// TIA Portal project "MSE_Mubea_AsitYikama" (V15.1)

(* hardware
DEVICE "S7-1200 station_1"  S7-1200 Station
   slot 0: "Rack_0"  S7-1200 Rack  Rack  V1.0
   slot 1: "PLC_1"  CPU 1215C DC/DC/DC  6ES7 215-1AG40-0XB0  V4.1
   slot 2: "DI16/DQ16 x 24VDC"  6ES7 223-1BL32-0XB0  V2.0
DEVICE "HMI_1"  KTP400 Basic color PN
   slot 0: "HMI_1"  KTP400 Basic color PN  6AV6 647-0AK11-3AX0  12.0.0.0
   slot 1: "HMI_RT_1"  KTP400 Basic color PN  6AV6 647-0AK11-3AX0  12.0.0.0
   slot 5: "HMI_1.IE_CP_1"  PROFINET Interface  12.0.0.0
      slot 1: "PROFINET Interface_1"  PROFINET Interface
         slot 1: "Port_1"  Port
*)

// ===== PLC "PLC_1"  CPU 1215C DC/DC/DC =====

VAR_GLOBAL   // PLC tag table "Default tag table"
   "Clock_Byte" AT %MB0 : Byte;
   "Clock_10Hz" AT %M0.0 : Bool;
   "Clock_5Hz" AT %M0.1 : Bool;
   "Clock_2.5Hz" AT %M0.2 : Bool;
   "Clock_2Hz" AT %M0.3 : Bool;
   "Clock_1.25Hz" AT %M0.4 : Bool;
   "Clock_1Hz" AT %M0.5 : Bool;
   "Clock_0.625Hz" AT %M0.6 : Bool;
   "Clock_0.5Hz" AT %M0.7 : Bool;
   "HmiSirkVana_Ac_Mem" AT %M1.0 : Bool;   // Sirkulasyon vanasini ac
   "HmiSirkVana_Kapat_Mem" AT %M1.1 : Bool;
   "HmiDolumVana_Ac_Mem" AT %M1.2 : Bool;
   "HmiDolumVana_Kapat_Mem" AT %M1.3 : Bool;
   "HmiAsitTahVana_Ac_Mem" AT %M1.4 : Bool;
   "HmiAsitTahVana_Kapat_Mem" AT %M1.5 : Bool;
   "HmiUcYolluVana_Ac_Mem" AT %M1.6 : Bool;
   "HmiUcYolluVana_Kapat_Mem" AT %M1.7 : Bool;
   "HmiKuyuVana_Ac_Mem" AT %M2.0 : Bool;
   "HmiKuyuVana_Kapat_Mem" AT %M2.1 : Bool;
   "HmiIBCVana_Ac_Mem" AT %M2.2 : Bool;
   "HmiIBCVana_Kapat_Mem" AT %M2.3 : Bool;
   "HmiAnaPompa_Run" AT %M2.4 : Bool;
   "HmiIBCPopmpa_Run" AT %M2.5 : Bool;
   "AsitDoldur_Started" AT %M2.6 : Bool;
   "AsitDoldurSeq_UcYolVana_Ac" AT %M2.7 : Bool;
   "AsitDoldurSeq_DolumVana_Ac" AT %M3.0 : Bool;
   "AsitDoldurSeq_SirVana_Kapat" AT %M3.1 : Bool;
   "AsitDoldurSeq_TahVana_Kapat" AT %M3.2 : Bool;
   "AsitDoldurSeq_KuyuVana_Kapat" AT %M3.3 : Bool;
   "AsitDoldurSeq_IBCVana_Kapat" AT %M3.4 : Bool;
   "AsitDoldurSeq_AnaPompa_Run" AT %M3.5 : Bool;
   "AsitSirkulas_Started" AT %M3.6 : Bool;
   "AsitSirkulas_SirkVana_Ac" AT %M3.7 : Bool;
   "AsitSirkulas_DolumVana_Kapat" AT %M4.0 : Bool;
   "AsitSirkulas_TahVana_Kapat" AT %M4.1 : Bool;
   "AsitSirkulas_UcYolVana_Kapat" AT %M4.2 : Bool;
   "AsitSirkulas_KuyuVana_Kapat" AT %M4.3 : Bool;
   "AsitSirkulas_IBCVana_Kapat" AT %M4.4 : Bool;
   "AsitSirkulas_AnaPompa_Run" AT %M4.5 : Bool;
   "AsitSirkTimerReset_Mem" AT %M4.6 : Bool;
   "AsitTahliyesi_Started" AT %M4.7 : Bool;
   "AsitTahliyesi_SirkVana_Kapat" AT %M5.0 : Bool;
   "AsitTahliyesi_DolumVana_Kapat" AT %M5.1 : Bool;
   "AsitTahliyesi_TahVana_Ac" AT %M5.2 : Bool;
   "AsitTahliyesi_UcYolVana_Kapat" AT %M5.3 : Bool;
   "AsitTahliyesi_KuyuTahVana_Kapat" AT %M5.4 : Bool;
   "AsitTahliyesi_IBCVana_Kapat" AT %M5.5 : Bool;
   "AsitTahliyesi_Pompa_Run" AT %M5.6 : Bool;
   "SuSirkulasyon_Started" AT %M5.7 : Bool;
   "SuSirkulasyonTimer_Reset" AT %M6.0 : Bool;
   "SuSirkulasyon_SirkVana_Ac" AT %M6.1 : Bool;
   "SuSirkulasyon_DolumVana_Kapat" AT %M6.2 : Bool;
   "SuSirkulasyon_TahVana_Kapat" AT %M6.3 : Bool;
   "SuSirkulasyon_UcYolluVana_Kapat" AT %M6.4 : Bool;
   "SuSirkulasyon_KuyuTah_Kapat" AT %M6.5 : Bool;
   "SuSirkulasyon_IBCVana_Kapat" AT %M6.6 : Bool;
   "SuSirkulasyon_Pompa_Run" AT %M6.7 : Bool;
   "SuTahliyesi_Started" AT %M7.0 : Bool;
   "SuTahliyesi_SirkVana_Kapat" AT %M7.1 : Bool;
   "SuTahliyesi_DolumVana_Kapat" AT %M7.2 : Bool;
   "SuTahliyesi_AsitTahVana_Kapat" AT %M7.3 : Bool;
   "SuTahliyesi_UcYolluVana_Kapat" AT %M7.4 : Bool;
   "SuTahliyesi_KuyuTahVana_Ac" AT %M7.5 : Bool;
   "SuTahliyesi_IBCVana_Kapat" AT %M7.6 : Bool;
   "SuTahliyesi_Pompa_Run" AT %M7.7 : Bool;
   "IBCTahliye_Started" AT %M8.0 : Bool;
   "IBCTahliye_SirkVana_Kapat" AT %M8.1 : Bool;
   "IBCTahliye_DolumVana_Kapat" AT %M8.2 : Bool;
   "IBCTahliye_AsitTahVana_Kapat" AT %M8.3 : Bool;
   "IBCTahliye_UcYolluVana_Kapat" AT %M8.4 : Bool;
   "IBCTahliye_kuyuTahVana_Kapat" AT %M8.5 : Bool;
   "IBCTahliye_IBCVana_Ac" AT %M8.6 : Bool;
   "tempPompaRun" AT %M8.7 : Bool;
   "IBCTahliye_IBCpompa_Run" AT %M9.0 : Bool;
   "AsitDoldur_Siren" AT %M9.1 : Bool;
   "AsitDoldur_IslemBitti" AT %M9.2 : Bool;
   "AsitSirkulas_Siren" AT %M9.3 : Bool;
   "AsitSirkulas_IslemBitti" AT %M9.4 : Bool;
   "AsitTahliyesi_Siren" AT %M9.5 : Bool;
   "AsitTahliyesi_IslemBitti" AT %M9.6 : Bool;
   "SuSirkulasyon_Siren" AT %M9.7 : Bool;
   "SuSirkulasyon_IslemBitti" AT %M10.0 : Bool;
   "SuTahliyesi_Siren" AT %M10.1 : Bool;
   "SuTahliyesi_IslemBitti" AT %M10.2 : Bool;
   "IBCTahliye_Siren" AT %M10.3 : Bool;
   "IBCTahliye_IslemBitti" AT %M10.4 : Bool;
   "HmiKorKuyuPompa_Run" AT %M10.5 : Bool;
   "I0.0" AT %I0.0 : Bool;   // Acil Stop 1
   "I0.1" AT %I0.1 : Bool;   // Acil Stop 2
   "I0.2" AT %I0.2 : Bool;   // Yikama tanki alt seviye sen.
   "I0.3" AT %I0.3 : Bool;   // Yikama tanki ust limit sen.
   "I0.4" AT %I0.4 : Bool;   // Asti tanki alt limit sen.
   "I0.5" AT %I0.5 : Bool;
   "I0.6" AT %I0.6 : Bool;   // Yikama tank kapi sw 1
   "I1.0" AT %I1.0 : Bool;   // Asit tanki kapi sw
   "I1.1" AT %I1.1 : Bool;   // tERMİK HATA
   "I1.2" AT %I1.2 : Bool;   // Sirkulasyon vanasi kapali
   "I1.3" AT %I1.3 : Bool;   // Sirkulasyon vanasi acik
   "I1.4" AT %I1.4 : Bool;   // Dolum vanasi kapali
   "I1.5" AT %I1.5 : Bool;   // Dolum vanasi acik
   "I2.0" AT %I2.0 : Bool;   // Asit tahliye vanasi kapali
   "I2.1" AT %I2.1 : Bool;   // Asit tahliye vanasi acik
   "I2.2" AT %I2.2 : Bool;   // Uc yollu vana kapali
   "I2.3" AT %I2.3 : Bool;   // Uc yollu vana acik
   "I2.4" AT %I2.4 : Bool;   // Kuyu tahliye vanasi kapali
   "I2.5" AT %I2.5 : Bool;   // Kuyu tahliye vanasi acik
   "I2.6" AT %I2.6 : Bool;   // IBC Akis vanasi kapali
   "I2.7" AT %I2.7 : Bool;   // IBC akis vanasi acik
   "AsitDoldurSeq_DolumVana_Kapat" AT %M10.6 : Bool;
   "AsitDoldurSeq_AnaPompa_Run_2" AT %M10.7 : Bool;
   "AsitSirkulas_SirkVana_Kapat" AT %M11.0 : Bool;
   "AsitSirkulas_AnaPompa_Run_2" AT %M11.1 : Bool;
   "AsitTahliyesi_TahVana_Kapat" AT %M11.2 : Bool;
   "AsitTahliyesi_Pompa_Run_2" AT %M11.3 : Bool;
   "SuDolumSeq_SirkVana_Kapat" AT %M11.4 : Bool;
   "SuDolumSeq_DolumVana_Kapat" AT %M11.5 : Bool;
   "SuDolumSeq_AsitTahVana_Kapat" AT %M11.6 : Bool;
   "SuDolumSeq_UcYolluVana_Kapat" AT %M11.7 : Bool;
   "SuDolumSeq_KuyuTahVana_Kapat" AT %M12.0 : Bool;
   "SuDolumSeq_IBCVana_Kapat" AT %M12.1 : Bool;
   "SuDolumSeq_SuyuAc" AT %M12.2 : Bool;
   "SuDolumSeq_IslemBitti" AT %M12.3 : Bool;
   "I0.7" AT %I0.7 : Bool;   // Yikama tanki orta seviye sensoru
   "Always_On" AT %M12.4 : Bool;
   "SuSirkulasyon_SirkVana_Kapat" AT %M12.5 : Bool;
   "SuSirkulasyon_Pompa_Run2" AT %M12.6 : Bool;
   "SuTahliyesi_KuyuTahVana_Kapat" AT %M12.7 : Bool;
   "SuTahliyesi_Popmpa_Run2" AT %M13.0 : Bool;
   "IBCTahliye_IBCVana_Kapat" AT %M13.1 : Bool;
   "IBCTahliye_IBCpompa_Run2" AT %M13.2 : Bool;
   "AsitDoldurSeq_UcyolluVana_Kapat" AT %M13.3 : Bool;
   "HmiSuDolumVana" AT %M13.4 : Bool;
   "SuDolumVanasi" AT %Q3.0 : Bool;
END_VAR

VAR_GLOBAL   // PLC tag table "Output"
   "YesilLamba" AT %Q0.0 : Bool;
   "KirmiziLamba" AT %Q0.1 : Bool;
   "Siren" AT %Q0.2 : Bool;
   "SirkulasyonVanaKapat" AT %Q0.3 : Bool;
   "SirkulasyonVanaAc" AT %Q0.4 : Bool;
   "DolumVanaKapat" AT %Q0.5 : Bool;
   "DolumVanaAc" AT %Q0.6 : Bool;
   "AsitTahliyeVanaKapat" AT %Q0.7 : Bool;
   "AsitTahliyeVanaAc" AT %Q1.0 : Bool;
   "UcYolluVanaKapat" AT %Q1.1 : Bool;
   "UcYolluVanaAc" AT %Q2.0 : Bool;
   "KuyuTahliyeVanaKapat" AT %Q2.1 : Bool;
   "KuyuTahliyeVanaAc" AT %Q2.2 : Bool;
   "IBCVanaKapat" AT %Q2.3 : Bool;
   "IBCVanaAc" AT %Q2.4 : Bool;
   "AnaPompa" AT %Q2.5 : Bool;
   "IBC_DiyaframPompa" AT %Q2.6 : Bool;
   "KorKuyuPompasi" AT %Q2.7 : Bool;
END_VAR

// folder: DataBlocks

DATA_BLOCK "FB_Manuel_DB"   // DB4
{ S7_Optimized_Access := 'TRUE' }
VERSION : 0.1
// stored: InstanceOfName FB_Manuel
"FB_Manuel"
BEGIN
END_DATA_BLOCK

DATA_BLOCK "21_Alarm_DB"   // DB17
{ S7_Optimized_Access := 'TRUE' }
VERSION : 0.1
// stored: InstanceOfName 21_Alarm
"21_Alarm"
BEGIN
END_DATA_BLOCK

DATA_BLOCK "01_Out_DB"   // DB18
{ S7_Optimized_Access := 'TRUE' }
VERSION : 0.1
// stored: InstanceOfName 01_Out
"01_Out"
BEGIN
END_DATA_BLOCK

// folder: System blocks/Program resources

DATA_BLOCK "AsitSirkTimer_DB"   // DB5
{ S7_Optimized_Access := 'TRUE' }
AUTHOR : Simatic
FAMILY : IEC
NAME : IEC_TMR
VERSION : 1.0
// stored: InstanceOfName IEC_TIMER
"IEC_TIMER"
BEGIN
END_DATA_BLOCK

DATA_BLOCK "SuSirkTimer_DB"   // DB7
{ S7_Optimized_Access := 'TRUE' }
AUTHOR : Simatic
FAMILY : IEC
NAME : IEC_TMR
VERSION : 1.0
// stored: InstanceOfName IEC_TIMER
"IEC_TIMER"
BEGIN
END_DATA_BLOCK

// folder: SystemData

DATA_BLOCK "01_System"   // DB1
{ S7_Optimized_Access := 'TRUE' }
VERSION : 0.1
   VAR
      SystemInfo : String[50] := 'Asit sirkulasyonu yapiliyor';   // Sistem durumları
      Alarms : Word;
      Process : Struct
         Manuel_Normal : Bool;
      END_STRUCT;
      State : Struct
         AsitDolum : Byte;
         AsitSirkulasyon : Byte;
         AsitTahliye : Byte;
         SuDolum : Byte;
         SuSirkulasyon : Byte;
         SuTahliye : Byte;
         IBCTahliye : Byte;
      END_STRUCT;
      AlwaysOn : Bool;
      ConvertTimeToDint : DInt;   // Hmi ekranı icin cevrim
      Timers : Struct
         AsitDolum_TimerAdim3 : IEC_TIMER;
         AsitDolum_TimerAdim3_Pom : IEC_TIMER;
         Manuel : Struct
            SirkVana_Ac : IEC_TIMER;
            SirkVana_Kapat : IEC_TIMER;
            DolumVana_Ac : IEC_TIMER;
            DolumVana_Kapat : IEC_TIMER;
            AsitTahVana_Ac : IEC_TIMER;
            AsitTahVana_Kapat : IEC_TIMER;
            UcYolluVana_Ac : IEC_TIMER;
            UcYolluVana_Kapat : IEC_TIMER;
            KuyuTahVana_Ac : IEC_TIMER;
            KuyuTahVana_Kapat : IEC_TIMER;
            IBCVana_Ac : IEC_TIMER;
            IBCVana_Kapat : IEC_TIMER;
         END_STRUCT;
         Sequence : Struct
            AsitSir_TimerAdim3 : IEC_TIMER;
            AsitSir_TimerAdim3_Pom : IEC_TIMER;
            AsitTah_TimerAdim3 : IEC_TIMER;
            AsitTah_TimerAdim3_Pom : IEC_TIMER;
            SuSir_TimerAdim2_Pom : IEC_TIMER;
            SuSir_TimerAdim2 : IEC_TIMER;
            SuTah_TimerAdim2 : IEC_TIMER;
            SuTah_TimerAdim2_Pom : IEC_TIMER;
            IBCTah_TimerAdim2 : IEC_TIMER;
            IBCTah_TimerAdim2_Pom : IEC_TIMER;
         END_STRUCT;
      END_STRUCT;
   END_VAR
BEGIN
END_DATA_BLOCK

DATA_BLOCK "02_Peripheral"   // DB2
{ S7_Optimized_Access := 'TRUE' }
VERSION : 0.1
   VAR
      IN : Struct
         AcilStop : Bool;
         YikamaTanki : Struct
            UstSeviyeSen : Bool;   // Yikama tanki ust seviye sensoru
            AltSeviyeSen : Bool;   // Yikama tanki alt seviye sensoru
            CriticalSeviyeSen : Bool;   // Yikama tanki kritik seviye sensoru
            KapiSwitch1 : Bool;   // Yikama tanki kapi sw 1
            KapiSwitch2 : Bool;   // Yikama tanki kapi sw 2
         END_STRUCT;
         AsitTanki : Struct
            UstSeviyeSen : Bool;
            AltSeviyeSen : Bool;
            KapiSwitch : Bool;
         END_STRUCT;
         SirkulasyonVanasi : Struct   // 1 numaralı vana
            Opened : Bool;
            Closed : Bool;
         END_STRUCT;
         DolumVanasi : Struct   // 2 numaralı vana
            Opened : Bool;
            Closed : Bool;
         END_STRUCT;
         AsitTahliyeVanasi : Struct   // 3 numaralı vana
            Opened : Bool;
            Closed : Bool;
         END_STRUCT;
         UcYolluVana : Struct   // 4 numaralı vana
            Opened : Bool;
            Closed : Bool;
         END_STRUCT;
         KuyuTahVanasi : Struct   // 5 numaralı vana
            Opened : Bool;
            Closed : Bool;
         END_STRUCT;
         IBC : Struct
            AkisValfi : Struct
               Opened : Bool;   // IBC vanasi acildi
               Closed : Bool;   // IBC vanasi kapandi
            END_STRUCT;
         END_STRUCT;
         TermikAnaPompa : Bool;
      END_STRUCT;
      OUT : Struct
         IBC : Struct
            PompaDiyafram : Bool;   // Diyafram pompasi
            AkisValfi : Struct   // 6 numaralı akis valfi
               Open : Bool;
               Close : Bool;
            END_STRUCT;
         END_STRUCT;
         SirkulasyonVanasi : Struct   // 1 numaralı vana
            Open : Bool;
            Close : Bool;
         END_STRUCT;
         DolumVanasi : Struct   // 2 numaralı vana
            Open : Bool;
            Close : Bool;
         END_STRUCT;
         AsitTahliyeVanasi : Struct   // 3 numaralı vana
            Open : Bool;
            Close : Bool;
         END_STRUCT;
         UcYolluVana : Struct   // 4 numaralı vana
            Open : Bool;
            Close : Bool;
         END_STRUCT;
         KuyuAktVanasi : Struct   // 5 numaralı vana
            Open : Bool;
            Close : Bool;
         END_STRUCT;
         AnaPompa : Bool;   // Ana doldurma ve sirkulasyon pompasi
         KorKuyuPompasi : Bool;   // Kör kuyu pompası
         SuDolumVanasi : Bool;   // Su dolumu yapmak icin
      END_STRUCT;
      Lamba : Struct
         Yesil : Bool;
         Sari : Bool;
         Kirmizi : Bool;
         Siren : Bool;
      END_STRUCT;
   END_VAR
BEGIN
END_DATA_BLOCK

DATA_BLOCK "03_HmiData"   // DB3
{ S7_Optimized_Access := 'TRUE' }
VERSION : 0.1
   VAR
      SurkilasyonVanasi_Ac : Bool;
      SurkilasyonVanasi_Kapat : Bool;
      DolumVanasi_Ac : Bool;
      DolumVanasi_Kapat : Bool;
      AsitTahliyeVanasi_Ac : Bool;
      AsitTahliyeVanasi_Kapat : Bool;
      UcYolluVana_Ac : Bool;
      UcYolluVana_Kapat : Bool;
      KuyuAktarimVanasi_Ac : Bool;
      KuyuAktarimVanasi_Kapat : Bool;
      IBCVanasi_Ac : Bool;
      IBCVanasi_Kapat : Bool;
      AnaPompa_Run : Bool;
      AnaPompa_Stop : Bool;
      IBC_DiyaframPompa_Run : Bool;
      IBC_DiyaframPompa_Stop : Bool;
      KorKuyuPompası_Run : Bool;
      KorKuyuPompası_Stop : Bool;
      SuDolumVanasi_Ac : Bool;
      SuDolumVanasi_Kapat : Bool;
   END_VAR
   VAR RETAIN
      TimerInterval : Struct
         AsitSirkulasyon : Time := T#1m;   // Asit sirkulasyon set degeri
         SuSirkulasyon : Time := T#1m;   // Su sirkulasyon set degeri
      END_STRUCT;
   END_VAR
   VAR
      Timer_ET : Struct
         AsitSirkulasyon : Time;
         SuSirkulasyon : Time;
      END_STRUCT;
      Started : Struct
         AsitDolum : Bool;
         AsitSirkulasyon : Bool;
         AsitTahliye : Bool;
         TemizSuDolum : Bool;
         TemizSuSirkulasyon : Bool;
         TemizSuTahliye : Bool;
         IBCTahliye : Bool;
      END_STRUCT;
      System : Struct
         Stop : Bool;   // ,
         AsitDoldurBaslat : Bool;   // Asit doldurma sekansı
         AsitSirkulasyonBaslat : Bool;   // Asit sirkulasyon sekansı
         AsitTahliyesiBaslat : Bool;
         TemizSuDolumuBaslat : Bool;
         TemizSuSirkulasyonuBaslat : Bool;
         TemizSuTahliyesiBaslat : Bool;
         IBCTahliyesiBaslat : Bool;
         WarningReset : Bool;
      END_STRUCT;
      Visualization : Struct
         TimerVisible : Bool;
         ActTimerMin : DInt;
         ActTimerSec : DInt;
         Visibility : Struct
            AsitDolum : Bool;
            AsitSirkulasyon : Bool;
            AsitTahliyesi : Bool;
            TemizSuDolum : Bool;
            TemizSuSirkulasyon : Bool;
            TemizSuTahliye : Bool;
            IBCTaliye : Bool;
            Manuel : Struct
               SirkulasyonVanaAc : Bool;
               SirkulasyonVanaKapat : Bool;
               DolumVanaAc : Bool;
               DolumVanaKapat : Bool;
               AsitTahVanaAc : Bool;
               AsitTahVanaKapat : Bool;
               UcYolluVanaAc : Bool;
               UcYolluVanaKapat : Bool;
               KuyuTahVanaAc : Bool;
               KuyuTahVanaKapat : Bool;
               IBCVanaAc : Bool;
               IBCVanaKapat : Bool;
            END_STRUCT;
         END_STRUCT;
         nMode : Int;
      END_STRUCT;
   END_VAR
BEGIN
END_DATA_BLOCK

// folder: (top level)

FUNCTION_BLOCK "01_Out"   // FB1, LAD
{ S7_Optimized_Access := 'TRUE' }
VERSION : 0.1
BEGIN

REGION Network 1: Sirkulasyon vanası ac
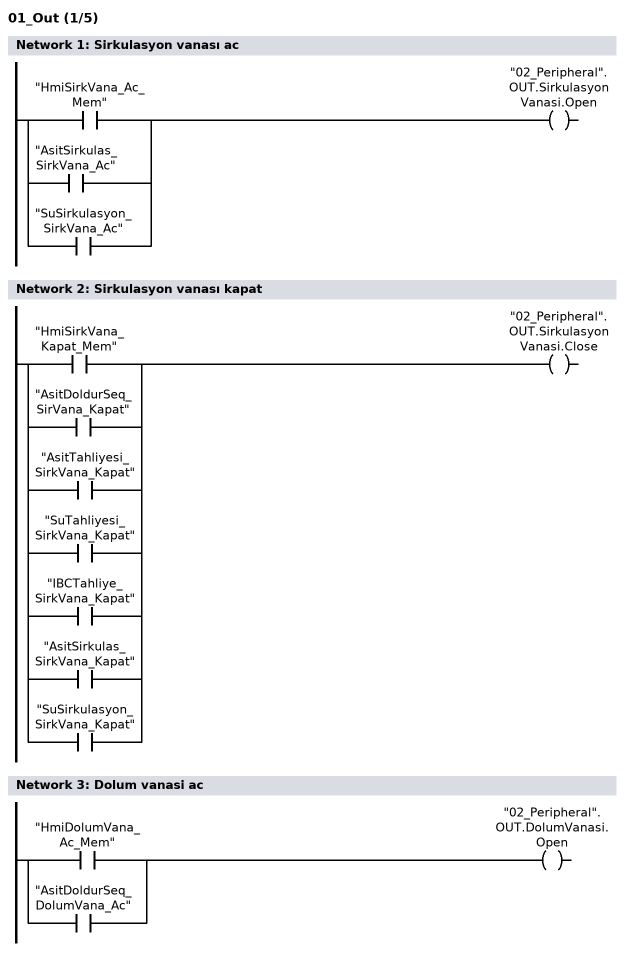
   RUNG wire#powerrail
      Contact( "HmiSirkVana_Ac_Mem" )
      wire#w1
      Coil( "02_Peripheral".OUT.SirkulasyonVanasi.Open )
   END_RUNG
   RUNG wire#powerrail
      Contact( "AsitSirkulas_SirkVana_Ac" )
   END_RUNG wire#w1
   RUNG wire#powerrail
      Contact( "SuSirkulasyon_SirkVana_Ac" )
   END_RUNG wire#w1
   // the same network as SCL:
   "02_Peripheral".OUT.SirkulasyonVanasi.Open := "HmiSirkVana_Ac_Mem" OR "AsitSirkulas_SirkVana_Ac" OR "SuSirkulasyon_SirkVana_Ac";
END_REGION

REGION Network 2: Sirkulasyon vanası kapat
   RUNG wire#powerrail
      Contact( "HmiSirkVana_Kapat_Mem" )
      wire#w1
      Coil( "02_Peripheral".OUT.SirkulasyonVanasi.Close )
   END_RUNG
   RUNG wire#powerrail
      Contact( "AsitDoldurSeq_SirVana_Kapat" )
   END_RUNG wire#w1
   RUNG wire#powerrail
      Contact( "AsitTahliyesi_SirkVana_Kapat" )
   END_RUNG wire#w1
   RUNG wire#powerrail
      Contact( "SuTahliyesi_SirkVana_Kapat" )
   END_RUNG wire#w1
   RUNG wire#powerrail
      Contact( "IBCTahliye_SirkVana_Kapat" )
   END_RUNG wire#w1
   RUNG wire#powerrail
      Contact( "AsitSirkulas_SirkVana_Kapat" )
   END_RUNG wire#w1
   RUNG wire#powerrail
      Contact( "SuSirkulasyon_SirkVana_Kapat" )
   END_RUNG wire#w1
   // the same network as SCL:
   "02_Peripheral".OUT.SirkulasyonVanasi.Close := "HmiSirkVana_Kapat_Mem" OR "AsitDoldurSeq_SirVana_Kapat" OR "AsitTahliyesi_SirkVana_Kapat" OR "SuTahliyesi_SirkVana_Kapat" OR "IBCTahliye_SirkVana_Kapat" OR "AsitSirkulas_SirkVana_Kapat" OR "SuSirkulasyon_SirkVana_Kapat";
END_REGION

REGION Network 3: Dolum vanasi ac
   RUNG wire#powerrail
      Contact( "HmiDolumVana_Ac_Mem" )
      wire#w1
      Coil( "02_Peripheral".OUT.DolumVanasi.Open )
   END_RUNG
   RUNG wire#powerrail
      Contact( "AsitDoldurSeq_DolumVana_Ac" )
   END_RUNG wire#w1
   // the same network as SCL:
   "02_Peripheral".OUT.DolumVanasi.Open := "HmiDolumVana_Ac_Mem" OR "AsitDoldurSeq_DolumVana_Ac";
END_REGION

REGION Network 4: Dolum vanasi kapat
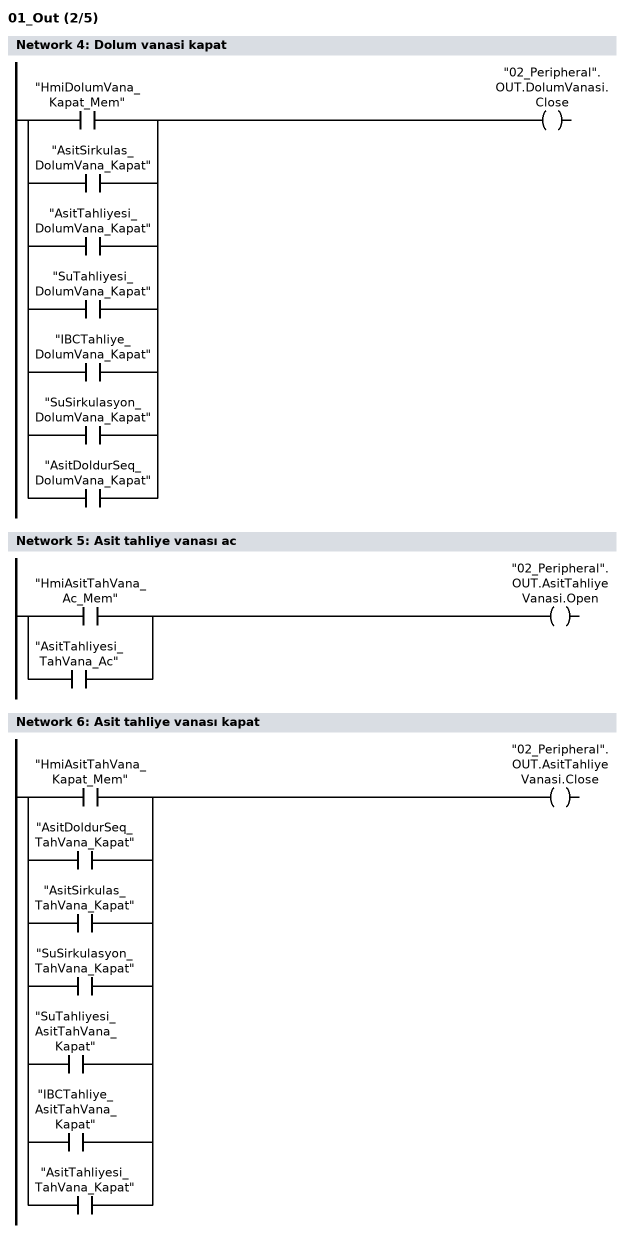
   RUNG wire#powerrail
      Contact( "HmiDolumVana_Kapat_Mem" )
      wire#w1
      Coil( "02_Peripheral".OUT.DolumVanasi.Close )
   END_RUNG
   RUNG wire#powerrail
      Contact( "AsitSirkulas_DolumVana_Kapat" )
   END_RUNG wire#w1
   RUNG wire#powerrail
      Contact( "AsitTahliyesi_DolumVana_Kapat" )
   END_RUNG wire#w1
   RUNG wire#powerrail
      Contact( "SuTahliyesi_DolumVana_Kapat" )
   END_RUNG wire#w1
   RUNG wire#powerrail
      Contact( "IBCTahliye_DolumVana_Kapat" )
   END_RUNG wire#w1
   RUNG wire#powerrail
      Contact( "SuSirkulasyon_DolumVana_Kapat" )
   END_RUNG wire#w1
   RUNG wire#powerrail
      Contact( "AsitDoldurSeq_DolumVana_Kapat" )
   END_RUNG wire#w1
   // the same network as SCL:
   "02_Peripheral".OUT.DolumVanasi.Close := "HmiDolumVana_Kapat_Mem" OR "AsitSirkulas_DolumVana_Kapat" OR "AsitTahliyesi_DolumVana_Kapat" OR "SuTahliyesi_DolumVana_Kapat" OR "IBCTahliye_DolumVana_Kapat" OR "SuSirkulasyon_DolumVana_Kapat" OR "AsitDoldurSeq_DolumVana_Kapat";
END_REGION

REGION Network 5: Asit tahliye vanası ac
   RUNG wire#powerrail
      Contact( "HmiAsitTahVana_Ac_Mem" )
      wire#w1
      Coil( "02_Peripheral".OUT.AsitTahliyeVanasi.Open )
   END_RUNG
   RUNG wire#powerrail
      Contact( "AsitTahliyesi_TahVana_Ac" )
   END_RUNG wire#w1
   // the same network as SCL:
   "02_Peripheral".OUT.AsitTahliyeVanasi.Open := "HmiAsitTahVana_Ac_Mem" OR "AsitTahliyesi_TahVana_Ac";
END_REGION

REGION Network 6: Asit tahliye vanası kapat
   RUNG wire#powerrail
      Contact( "HmiAsitTahVana_Kapat_Mem" )
      wire#w1
      Coil( "02_Peripheral".OUT.AsitTahliyeVanasi.Close )
   END_RUNG
   RUNG wire#powerrail
      Contact( "AsitDoldurSeq_TahVana_Kapat" )
   END_RUNG wire#w1
   RUNG wire#powerrail
      Contact( "AsitSirkulas_TahVana_Kapat" )
   END_RUNG wire#w1
   RUNG wire#powerrail
      Contact( "SuSirkulasyon_TahVana_Kapat" )
   END_RUNG wire#w1
   RUNG wire#powerrail
      Contact( "SuTahliyesi_AsitTahVana_Kapat" )
   END_RUNG wire#w1
   RUNG wire#powerrail
      Contact( "IBCTahliye_AsitTahVana_Kapat" )
   END_RUNG wire#w1
   RUNG wire#powerrail
      Contact( "AsitTahliyesi_TahVana_Kapat" )
   END_RUNG wire#w1
   // the same network as SCL:
   "02_Peripheral".OUT.AsitTahliyeVanasi.Close := "HmiAsitTahVana_Kapat_Mem" OR "AsitDoldurSeq_TahVana_Kapat" OR "AsitSirkulas_TahVana_Kapat" OR "SuSirkulasyon_TahVana_Kapat" OR "SuTahliyesi_AsitTahVana_Kapat" OR "IBCTahliye_AsitTahVana_Kapat" OR "AsitTahliyesi_TahVana_Kapat";
END_REGION

REGION Network 7: Uc yollu vana ac
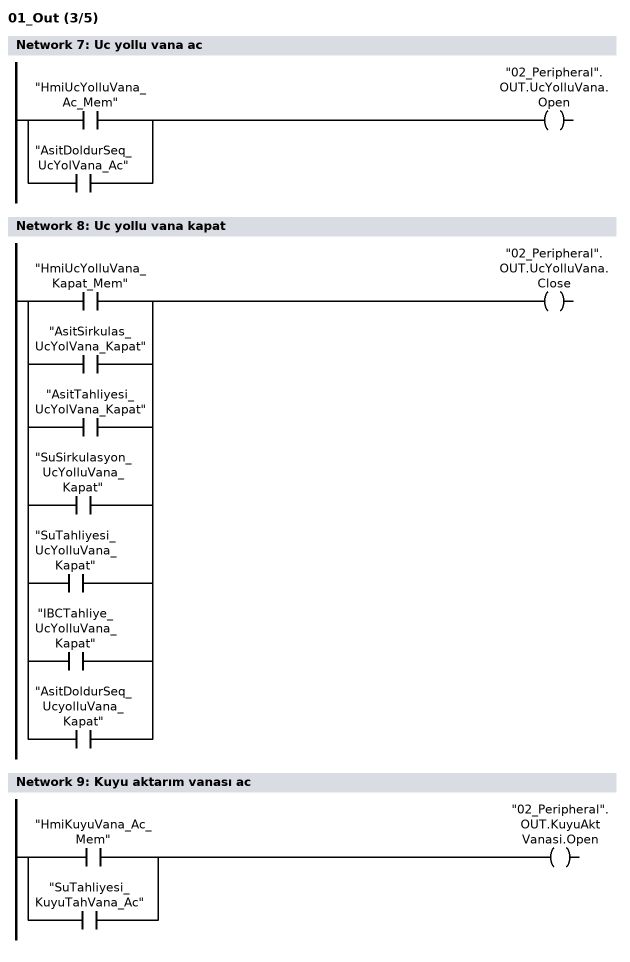
   RUNG wire#powerrail
      Contact( "HmiUcYolluVana_Ac_Mem" )
      wire#w1
      Coil( "02_Peripheral".OUT.UcYolluVana.Open )
   END_RUNG
   RUNG wire#powerrail
      Contact( "AsitDoldurSeq_UcYolVana_Ac" )
   END_RUNG wire#w1
   // the same network as SCL:
   "02_Peripheral".OUT.UcYolluVana.Open := "HmiUcYolluVana_Ac_Mem" OR "AsitDoldurSeq_UcYolVana_Ac";
END_REGION

REGION Network 8: Uc yollu vana kapat
   RUNG wire#powerrail
      Contact( "HmiUcYolluVana_Kapat_Mem" )
      wire#w1
      Coil( "02_Peripheral".OUT.UcYolluVana.Close )
   END_RUNG
   RUNG wire#powerrail
      Contact( "AsitSirkulas_UcYolVana_Kapat" )
   END_RUNG wire#w1
   RUNG wire#powerrail
      Contact( "AsitTahliyesi_UcYolVana_Kapat" )
   END_RUNG wire#w1
   RUNG wire#powerrail
      Contact( "SuSirkulasyon_UcYolluVana_Kapat" )
   END_RUNG wire#w1
   RUNG wire#powerrail
      Contact( "SuTahliyesi_UcYolluVana_Kapat" )
   END_RUNG wire#w1
   RUNG wire#powerrail
      Contact( "IBCTahliye_UcYolluVana_Kapat" )
   END_RUNG wire#w1
   RUNG wire#powerrail
      Contact( "AsitDoldurSeq_UcyolluVana_Kapat" )
   END_RUNG wire#w1
   // the same network as SCL:
   "02_Peripheral".OUT.UcYolluVana.Close := "HmiUcYolluVana_Kapat_Mem" OR "AsitSirkulas_UcYolVana_Kapat" OR "AsitTahliyesi_UcYolVana_Kapat" OR "SuSirkulasyon_UcYolluVana_Kapat" OR "SuTahliyesi_UcYolluVana_Kapat" OR "IBCTahliye_UcYolluVana_Kapat" OR "AsitDoldurSeq_UcyolluVana_Kapat";
END_REGION

REGION Network 9: Kuyu aktarım vanası ac
   RUNG wire#powerrail
      Contact( "HmiKuyuVana_Ac_Mem" )
      wire#w1
      Coil( "02_Peripheral".OUT.KuyuAktVanasi.Open )
   END_RUNG
   RUNG wire#powerrail
      Contact( "SuTahliyesi_KuyuTahVana_Ac" )
   END_RUNG wire#w1
   // the same network as SCL:
   "02_Peripheral".OUT.KuyuAktVanasi.Open := "HmiKuyuVana_Ac_Mem" OR "SuTahliyesi_KuyuTahVana_Ac";
END_REGION

REGION Network 10: Kuyu aktarım vanası kapat
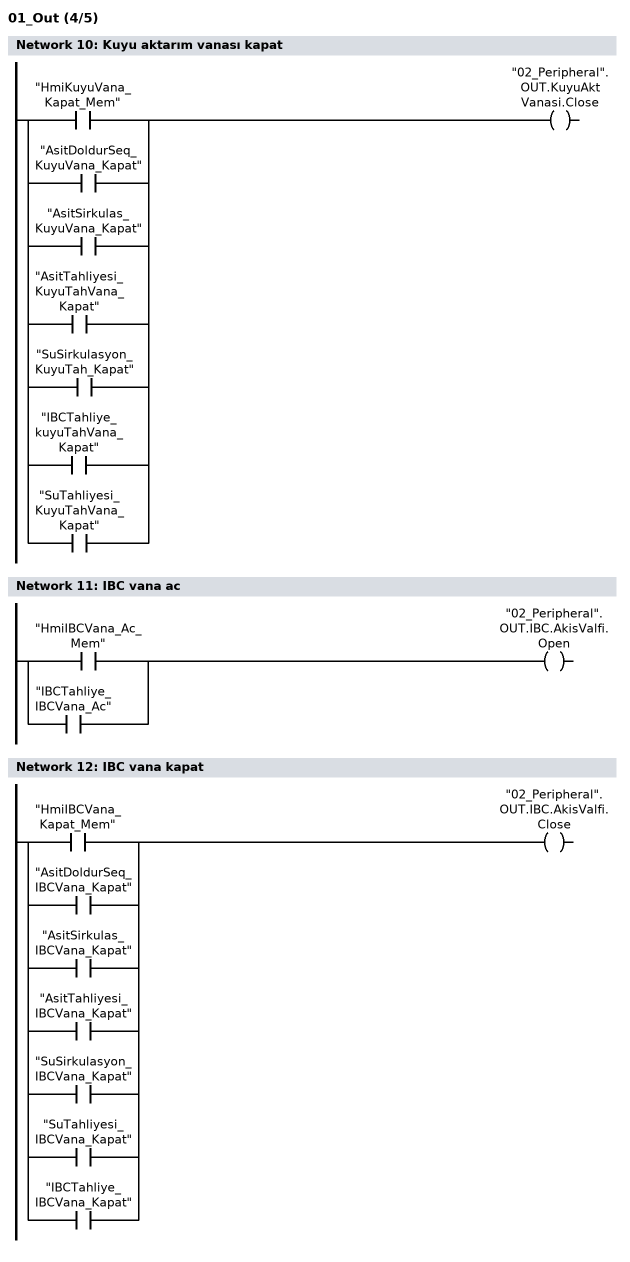
   RUNG wire#powerrail
      Contact( "HmiKuyuVana_Kapat_Mem" )
      wire#w1
      Coil( "02_Peripheral".OUT.KuyuAktVanasi.Close )
   END_RUNG
   RUNG wire#powerrail
      Contact( "AsitDoldurSeq_KuyuVana_Kapat" )
   END_RUNG wire#w1
   RUNG wire#powerrail
      Contact( "AsitSirkulas_KuyuVana_Kapat" )
   END_RUNG wire#w1
   RUNG wire#powerrail
      Contact( "AsitTahliyesi_KuyuTahVana_Kapat" )
   END_RUNG wire#w1
   RUNG wire#powerrail
      Contact( "SuSirkulasyon_KuyuTah_Kapat" )
   END_RUNG wire#w1
   RUNG wire#powerrail
      Contact( "IBCTahliye_kuyuTahVana_Kapat" )
   END_RUNG wire#w1
   RUNG wire#powerrail
      Contact( "SuTahliyesi_KuyuTahVana_Kapat" )
   END_RUNG wire#w1
   // the same network as SCL:
   "02_Peripheral".OUT.KuyuAktVanasi.Close := "HmiKuyuVana_Kapat_Mem" OR "AsitDoldurSeq_KuyuVana_Kapat" OR "AsitSirkulas_KuyuVana_Kapat" OR "AsitTahliyesi_KuyuTahVana_Kapat" OR "SuSirkulasyon_KuyuTah_Kapat" OR "IBCTahliye_kuyuTahVana_Kapat" OR "SuTahliyesi_KuyuTahVana_Kapat";
END_REGION

REGION Network 11: IBC vana ac
   RUNG wire#powerrail
      Contact( "HmiIBCVana_Ac_Mem" )
      wire#w1
      Coil( "02_Peripheral".OUT.IBC.AkisValfi.Open )
   END_RUNG
   RUNG wire#powerrail
      Contact( "IBCTahliye_IBCVana_Ac" )
   END_RUNG wire#w1
   // the same network as SCL:
   "02_Peripheral".OUT.IBC.AkisValfi.Open := "HmiIBCVana_Ac_Mem" OR "IBCTahliye_IBCVana_Ac";
END_REGION

REGION Network 12: IBC vana kapat
   RUNG wire#powerrail
      Contact( "HmiIBCVana_Kapat_Mem" )
      wire#w1
      Coil( "02_Peripheral".OUT.IBC.AkisValfi.Close )
   END_RUNG
   RUNG wire#powerrail
      Contact( "AsitDoldurSeq_IBCVana_Kapat" )
   END_RUNG wire#w1
   RUNG wire#powerrail
      Contact( "AsitSirkulas_IBCVana_Kapat" )
   END_RUNG wire#w1
   RUNG wire#powerrail
      Contact( "AsitTahliyesi_IBCVana_Kapat" )
   END_RUNG wire#w1
   RUNG wire#powerrail
      Contact( "SuSirkulasyon_IBCVana_Kapat" )
   END_RUNG wire#w1
   RUNG wire#powerrail
      Contact( "SuTahliyesi_IBCVana_Kapat" )
   END_RUNG wire#w1
   RUNG wire#powerrail
      Contact( "IBCTahliye_IBCVana_Kapat" )
   END_RUNG wire#w1
   // the same network as SCL:
   "02_Peripheral".OUT.IBC.AkisValfi.Close := "HmiIBCVana_Kapat_Mem" OR "AsitDoldurSeq_IBCVana_Kapat" OR "AsitSirkulas_IBCVana_Kapat" OR "AsitTahliyesi_IBCVana_Kapat" OR "SuSirkulasyon_IBCVana_Kapat" OR "SuTahliyesi_IBCVana_Kapat" OR "IBCTahliye_IBCVana_Kapat";
END_REGION

REGION Network 13: Ana pompa run/stop
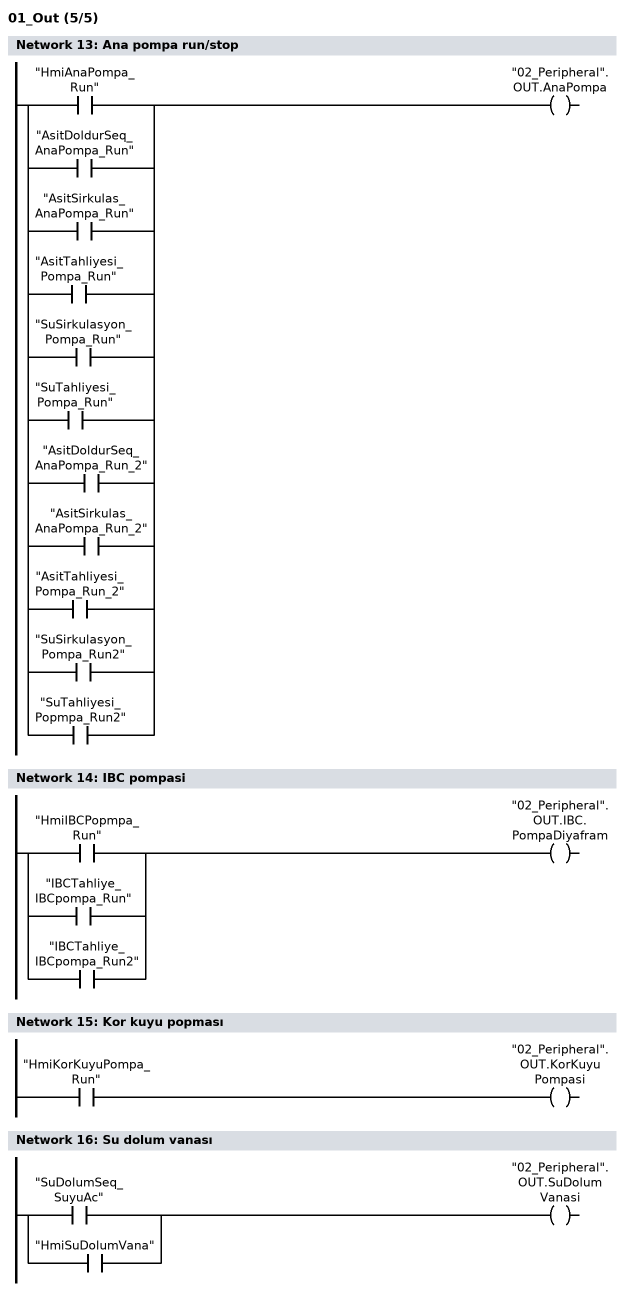
   RUNG wire#powerrail
      Contact( "HmiAnaPompa_Run" )
      wire#w1
      Coil( "02_Peripheral".OUT.AnaPompa )
   END_RUNG
   RUNG wire#powerrail
      Contact( "AsitDoldurSeq_AnaPompa_Run" )
   END_RUNG wire#w1
   RUNG wire#powerrail
      Contact( "AsitSirkulas_AnaPompa_Run" )
   END_RUNG wire#w1
   RUNG wire#powerrail
      Contact( "AsitTahliyesi_Pompa_Run" )
   END_RUNG wire#w1
   RUNG wire#powerrail
      Contact( "SuSirkulasyon_Pompa_Run" )
   END_RUNG wire#w1
   RUNG wire#powerrail
      Contact( "SuTahliyesi_Pompa_Run" )
   END_RUNG wire#w1
   RUNG wire#powerrail
      Contact( "AsitDoldurSeq_AnaPompa_Run_2" )
   END_RUNG wire#w1
   RUNG wire#powerrail
      Contact( "AsitSirkulas_AnaPompa_Run_2" )
   END_RUNG wire#w1
   RUNG wire#powerrail
      Contact( "AsitTahliyesi_Pompa_Run_2" )
   END_RUNG wire#w1
   RUNG wire#powerrail
      Contact( "SuSirkulasyon_Pompa_Run2" )
   END_RUNG wire#w1
   RUNG wire#powerrail
      Contact( "SuTahliyesi_Popmpa_Run2" )
   END_RUNG wire#w1
   // the same network as SCL:
   "02_Peripheral".OUT.AnaPompa := "HmiAnaPompa_Run" OR "AsitDoldurSeq_AnaPompa_Run" OR "AsitSirkulas_AnaPompa_Run" OR "AsitTahliyesi_Pompa_Run" OR "SuSirkulasyon_Pompa_Run" OR "SuTahliyesi_Pompa_Run" OR "AsitDoldurSeq_AnaPompa_Run_2" OR "AsitSirkulas_AnaPompa_Run_2" OR "AsitTahliyesi_Pompa_Run_2" OR "SuSirkulasyon_Pompa_Run2" OR "SuTahliyesi_Popmpa_Run2";
END_REGION

REGION Network 14: IBC pompasi
   RUNG wire#powerrail
      Contact( "HmiIBCPopmpa_Run" )
      wire#w1
      Coil( "02_Peripheral".OUT.IBC.PompaDiyafram )
   END_RUNG
   RUNG wire#powerrail
      Contact( "IBCTahliye_IBCpompa_Run" )
   END_RUNG wire#w1
   RUNG wire#powerrail
      Contact( "IBCTahliye_IBCpompa_Run2" )
   END_RUNG wire#w1
   // the same network as SCL:
   "02_Peripheral".OUT.IBC.PompaDiyafram := "HmiIBCPopmpa_Run" OR "IBCTahliye_IBCpompa_Run" OR "IBCTahliye_IBCpompa_Run2";
END_REGION

REGION Network 15: Kor kuyu popması
   RUNG wire#powerrail
      Contact( "HmiKorKuyuPompa_Run" )
      Coil( "02_Peripheral".OUT.KorKuyuPompasi )
   END_RUNG
   // the same network as SCL:
   "02_Peripheral".OUT.KorKuyuPompasi := "HmiKorKuyuPompa_Run";
END_REGION

REGION Network 16: Su dolum vanası
   RUNG wire#powerrail
      Contact( "SuDolumSeq_SuyuAc" )
      wire#w1
      Coil( "02_Peripheral".OUT.SuDolumVanasi )
   END_RUNG
   RUNG wire#powerrail
      Contact( "HmiSuDolumVana" )
   END_RUNG wire#w1
   // the same network as SCL:
   "02_Peripheral".OUT.SuDolumVanasi := "SuDolumSeq_SuyuAc" OR "HmiSuDolumVana";
END_REGION
END_FUNCTION_BLOCK

FUNCTION_BLOCK "FB_Manuel"   // FB2, LAD
{ S7_Optimized_Access := 'TRUE' }
VERSION : 0.1
   VAR_TEMP
      tTimerInterval : Time;
      bEmpty : Bool;
   END_VAR
   VAR_TEMP   // added for the SCL form of the ladder/FBD networks
      _w1 : Bool;
   END_VAR
BEGIN

REGION Network 1: Timer set degeri
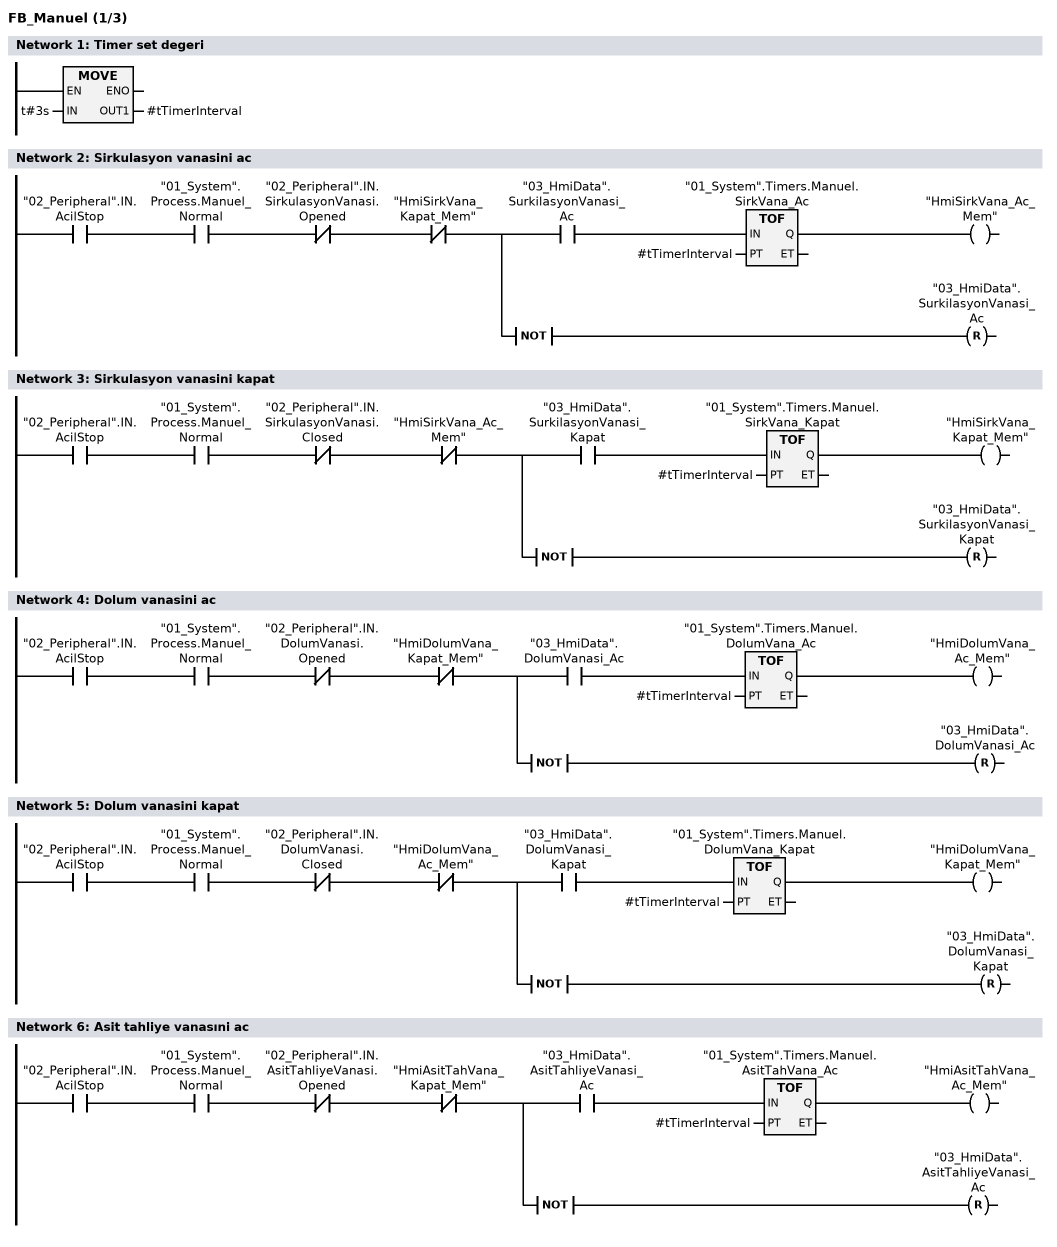
   RUNG wire#powerrail
      Move(in := t#3s, out1 => #tTimerInterval)
   END_RUNG
   // the same network as SCL:
   #tTimerInterval := t#3s;
END_REGION

REGION Network 2: Sirkulasyon vanasini ac
   #_w1 := "02_Peripheral".IN.AcilStop AND "01_System".Process.Manuel_Normal AND NOT "02_Peripheral".IN.SirkulasyonVanasi.Opened AND NOT "HmiSirkVana_Kapat_Mem";
   "01_System".Timers.Manuel.SirkVana_Ac.TOF(IN := #_w1 AND "03_HmiData".SurkilasyonVanasi_Ac,
                           PT := #tTimerInterval);
   "HmiSirkVana_Ac_Mem" := "01_System".Timers.Manuel.SirkVana_Ac.Q;
   IF NOT #_w1 THEN "03_HmiData".SurkilasyonVanasi_Ac := FALSE; END_IF;
END_REGION

REGION Network 3: Sirkulasyon vanasini kapat
   #_w1 := "02_Peripheral".IN.AcilStop AND "01_System".Process.Manuel_Normal AND NOT "02_Peripheral".IN.SirkulasyonVanasi.Closed AND NOT "HmiSirkVana_Ac_Mem";
   "01_System".Timers.Manuel.SirkVana_Kapat.TOF(IN := #_w1 AND "03_HmiData".SurkilasyonVanasi_Kapat,
                           PT := #tTimerInterval);
   "HmiSirkVana_Kapat_Mem" := "01_System".Timers.Manuel.SirkVana_Kapat.Q;
   IF NOT #_w1 THEN "03_HmiData".SurkilasyonVanasi_Kapat := FALSE; END_IF;
END_REGION

REGION Network 4: Dolum vanasini ac
   #_w1 := "02_Peripheral".IN.AcilStop AND "01_System".Process.Manuel_Normal AND NOT "02_Peripheral".IN.DolumVanasi.Opened AND NOT "HmiDolumVana_Kapat_Mem";
   "01_System".Timers.Manuel.DolumVana_Ac.TOF(IN := #_w1 AND "03_HmiData".DolumVanasi_Ac, PT := #tTimerInterval);
   "HmiDolumVana_Ac_Mem" := "01_System".Timers.Manuel.DolumVana_Ac.Q;
   IF NOT #_w1 THEN "03_HmiData".DolumVanasi_Ac := FALSE; END_IF;
END_REGION

REGION Network 5: Dolum vanasini kapat
   #_w1 := "02_Peripheral".IN.AcilStop AND "01_System".Process.Manuel_Normal AND NOT "02_Peripheral".IN.DolumVanasi.Closed AND NOT "HmiDolumVana_Ac_Mem";
   "01_System".Timers.Manuel.DolumVana_Kapat.TOF(IN := #_w1 AND "03_HmiData".DolumVanasi_Kapat,
                           PT := #tTimerInterval);
   "HmiDolumVana_Kapat_Mem" := "01_System".Timers.Manuel.DolumVana_Kapat.Q;
   IF NOT #_w1 THEN "03_HmiData".DolumVanasi_Kapat := FALSE; END_IF;
END_REGION

REGION Network 6: Asit tahliye vanasıni ac
   #_w1 := "02_Peripheral".IN.AcilStop AND "01_System".Process.Manuel_Normal AND NOT "02_Peripheral".IN.AsitTahliyeVanasi.Opened AND NOT "HmiAsitTahVana_Kapat_Mem";
   "01_System".Timers.Manuel.AsitTahVana_Ac.TOF(IN := #_w1 AND "03_HmiData".AsitTahliyeVanasi_Ac,
                           PT := #tTimerInterval);
   "HmiAsitTahVana_Ac_Mem" := "01_System".Timers.Manuel.AsitTahVana_Ac.Q;
   IF NOT #_w1 THEN "03_HmiData".AsitTahliyeVanasi_Ac := FALSE; END_IF;
END_REGION

REGION Network 7: Asit tahliye vanasıni kapat
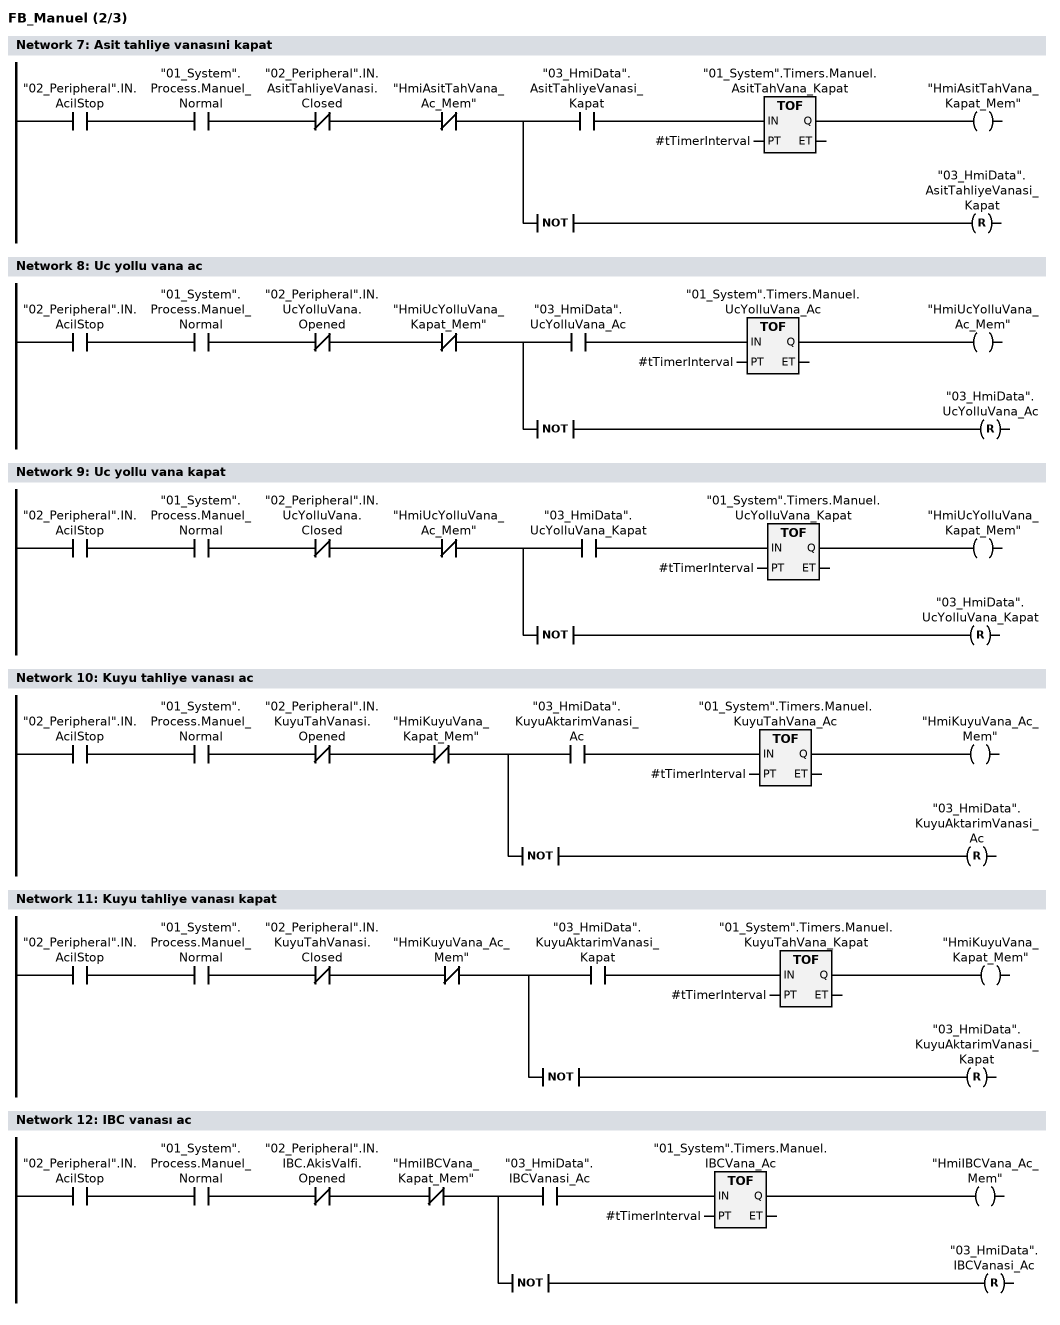
   #_w1 := "02_Peripheral".IN.AcilStop AND "01_System".Process.Manuel_Normal AND NOT "02_Peripheral".IN.AsitTahliyeVanasi.Closed AND NOT "HmiAsitTahVana_Ac_Mem";
   "01_System".Timers.Manuel.AsitTahVana_Kapat.TOF(IN := #_w1 AND "03_HmiData".AsitTahliyeVanasi_Kapat,
                           PT := #tTimerInterval);
   "HmiAsitTahVana_Kapat_Mem" := "01_System".Timers.Manuel.AsitTahVana_Kapat.Q;
   IF NOT #_w1 THEN "03_HmiData".AsitTahliyeVanasi_Kapat := FALSE; END_IF;
END_REGION

REGION Network 8: Uc yollu vana ac
   #_w1 := "02_Peripheral".IN.AcilStop AND "01_System".Process.Manuel_Normal AND NOT "02_Peripheral".IN.UcYolluVana.Opened AND NOT "HmiUcYolluVana_Kapat_Mem";
   "01_System".Timers.Manuel.UcYolluVana_Ac.TOF(IN := #_w1 AND "03_HmiData".UcYolluVana_Ac,
                           PT := #tTimerInterval);
   "HmiUcYolluVana_Ac_Mem" := "01_System".Timers.Manuel.UcYolluVana_Ac.Q;
   IF NOT #_w1 THEN "03_HmiData".UcYolluVana_Ac := FALSE; END_IF;
END_REGION

REGION Network 9: Uc yollu vana kapat
   #_w1 := "02_Peripheral".IN.AcilStop AND "01_System".Process.Manuel_Normal AND NOT "02_Peripheral".IN.UcYolluVana.Closed AND NOT "HmiUcYolluVana_Ac_Mem";
   "01_System".Timers.Manuel.UcYolluVana_Kapat.TOF(IN := #_w1 AND "03_HmiData".UcYolluVana_Kapat,
                           PT := #tTimerInterval);
   "HmiUcYolluVana_Kapat_Mem" := "01_System".Timers.Manuel.UcYolluVana_Kapat.Q;
   IF NOT #_w1 THEN "03_HmiData".UcYolluVana_Kapat := FALSE; END_IF;
END_REGION

REGION Network 10: Kuyu tahliye vanası ac
   #_w1 := "02_Peripheral".IN.AcilStop AND "01_System".Process.Manuel_Normal AND NOT "02_Peripheral".IN.KuyuTahVanasi.Opened AND NOT "HmiKuyuVana_Kapat_Mem";
   "01_System".Timers.Manuel.KuyuTahVana_Ac.TOF(IN := #_w1 AND "03_HmiData".KuyuAktarimVanasi_Ac,
                           PT := #tTimerInterval);
   "HmiKuyuVana_Ac_Mem" := "01_System".Timers.Manuel.KuyuTahVana_Ac.Q;
   IF NOT #_w1 THEN "03_HmiData".KuyuAktarimVanasi_Ac := FALSE; END_IF;
END_REGION

REGION Network 11: Kuyu tahliye vanası kapat
   #_w1 := "02_Peripheral".IN.AcilStop AND "01_System".Process.Manuel_Normal AND NOT "02_Peripheral".IN.KuyuTahVanasi.Closed AND NOT "HmiKuyuVana_Ac_Mem";
   "01_System".Timers.Manuel.KuyuTahVana_Kapat.TOF(IN := #_w1 AND "03_HmiData".KuyuAktarimVanasi_Kapat,
                           PT := #tTimerInterval);
   "HmiKuyuVana_Kapat_Mem" := "01_System".Timers.Manuel.KuyuTahVana_Kapat.Q;
   IF NOT #_w1 THEN "03_HmiData".KuyuAktarimVanasi_Kapat := FALSE; END_IF;
END_REGION

REGION Network 12: IBC vanası ac
   #_w1 := "02_Peripheral".IN.AcilStop AND "01_System".Process.Manuel_Normal AND NOT "02_Peripheral".IN.IBC.AkisValfi.Opened AND NOT "HmiIBCVana_Kapat_Mem";
   "01_System".Timers.Manuel.IBCVana_Ac.TOF(IN := #_w1 AND "03_HmiData".IBCVanasi_Ac, PT := #tTimerInterval);
   "HmiIBCVana_Ac_Mem" := "01_System".Timers.Manuel.IBCVana_Ac.Q;
   IF NOT #_w1 THEN "03_HmiData".IBCVanasi_Ac := FALSE; END_IF;
END_REGION

REGION Network 13: IBC vanası kapat
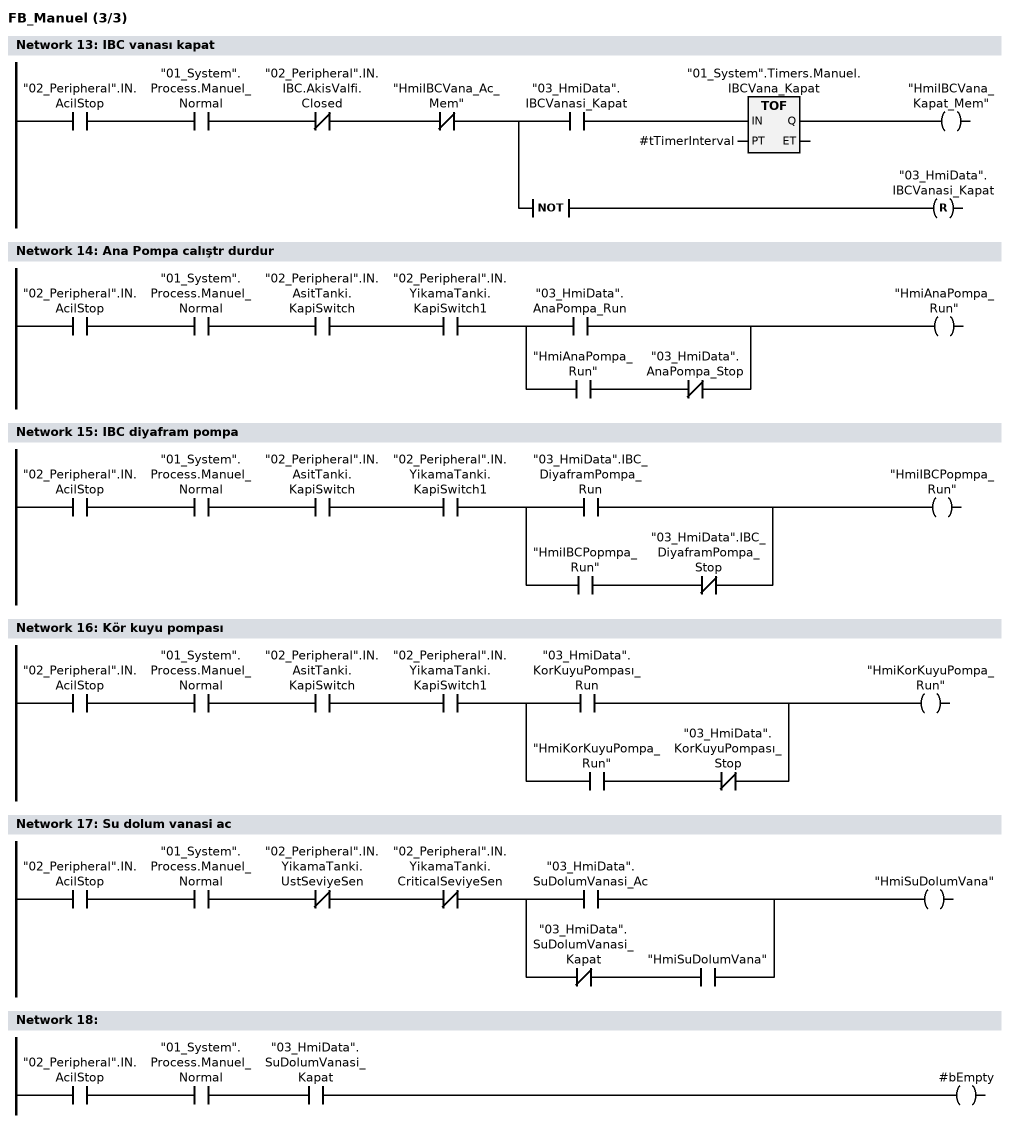
   #_w1 := "02_Peripheral".IN.AcilStop AND "01_System".Process.Manuel_Normal AND NOT "02_Peripheral".IN.IBC.AkisValfi.Closed AND NOT "HmiIBCVana_Ac_Mem";
   "01_System".Timers.Manuel.IBCVana_Kapat.TOF(IN := #_w1 AND "03_HmiData".IBCVanasi_Kapat,
                           PT := #tTimerInterval);
   "HmiIBCVana_Kapat_Mem" := "01_System".Timers.Manuel.IBCVana_Kapat.Q;
   IF NOT #_w1 THEN "03_HmiData".IBCVanasi_Kapat := FALSE; END_IF;
END_REGION

REGION Network 14: Ana Pompa calıştr durdur
   RUNG wire#powerrail
      Contact( "02_Peripheral".IN.AcilStop )
      Contact( "01_System".Process.Manuel_Normal )
      Contact( "02_Peripheral".IN.AsitTanki.KapiSwitch )
      Contact( "02_Peripheral".IN.YikamaTanki.KapiSwitch1 )
      wire#w1
      Contact( "03_HmiData".AnaPompa_Run )
      wire#w2
      Coil( "HmiAnaPompa_Run" )
   END_RUNG
   RUNG wire#w1
      Contact( "HmiAnaPompa_Run" )
      I_Contact( "03_HmiData".AnaPompa_Stop )
   END_RUNG wire#w2
   // the same network as SCL:
   "HmiAnaPompa_Run" := "02_Peripheral".IN.AcilStop AND "01_System".Process.Manuel_Normal AND "02_Peripheral".IN.AsitTanki.KapiSwitch AND "02_Peripheral".IN.YikamaTanki.KapiSwitch1 AND ("03_HmiData".AnaPompa_Run OR ("HmiAnaPompa_Run" AND NOT "03_HmiData".AnaPompa_Stop));
END_REGION

REGION Network 15: IBC diyafram pompa
   RUNG wire#powerrail
      Contact( "02_Peripheral".IN.AcilStop )
      Contact( "01_System".Process.Manuel_Normal )
      Contact( "02_Peripheral".IN.AsitTanki.KapiSwitch )
      Contact( "02_Peripheral".IN.YikamaTanki.KapiSwitch1 )
      wire#w1
      Contact( "03_HmiData".IBC_DiyaframPompa_Run )
      wire#w2
      Coil( "HmiIBCPopmpa_Run" )
   END_RUNG
   RUNG wire#w1
      Contact( "HmiIBCPopmpa_Run" )
      I_Contact( "03_HmiData".IBC_DiyaframPompa_Stop )
   END_RUNG wire#w2
   // the same network as SCL:
   "HmiIBCPopmpa_Run" := "02_Peripheral".IN.AcilStop AND "01_System".Process.Manuel_Normal AND "02_Peripheral".IN.AsitTanki.KapiSwitch AND "02_Peripheral".IN.YikamaTanki.KapiSwitch1 AND ("03_HmiData".IBC_DiyaframPompa_Run OR ("HmiIBCPopmpa_Run" AND NOT "03_HmiData".IBC_DiyaframPompa_Stop));
END_REGION

REGION Network 16: Kör kuyu pompası
   RUNG wire#powerrail
      Contact( "02_Peripheral".IN.AcilStop )
      Contact( "01_System".Process.Manuel_Normal )
      Contact( "02_Peripheral".IN.AsitTanki.KapiSwitch )
      Contact( "02_Peripheral".IN.YikamaTanki.KapiSwitch1 )
      wire#w1
      Contact( "03_HmiData".KorKuyuPompası_Run )
      wire#w2
      Coil( "HmiKorKuyuPompa_Run" )
   END_RUNG
   RUNG wire#w1
      Contact( "HmiKorKuyuPompa_Run" )
      I_Contact( "03_HmiData".KorKuyuPompası_Stop )
   END_RUNG wire#w2
   // the same network as SCL:
   "HmiKorKuyuPompa_Run" := "02_Peripheral".IN.AcilStop AND "01_System".Process.Manuel_Normal AND "02_Peripheral".IN.AsitTanki.KapiSwitch AND "02_Peripheral".IN.YikamaTanki.KapiSwitch1 AND ("03_HmiData".KorKuyuPompası_Run OR ("HmiKorKuyuPompa_Run" AND NOT "03_HmiData".KorKuyuPompası_Stop));
END_REGION

REGION Network 17: Su dolum vanasi ac
   RUNG wire#powerrail
      Contact( "02_Peripheral".IN.AcilStop )
      Contact( "01_System".Process.Manuel_Normal )
      I_Contact( "02_Peripheral".IN.YikamaTanki.UstSeviyeSen )
      I_Contact( "02_Peripheral".IN.YikamaTanki.CriticalSeviyeSen )
      wire#w1
      Contact( "03_HmiData".SuDolumVanasi_Ac )
      wire#w2
      Coil( "HmiSuDolumVana" )
   END_RUNG
   RUNG wire#w1
      I_Contact( "03_HmiData".SuDolumVanasi_Kapat )
      Contact( "HmiSuDolumVana" )
   END_RUNG wire#w2
   // the same network as SCL:
   "HmiSuDolumVana" := "02_Peripheral".IN.AcilStop AND "01_System".Process.Manuel_Normal AND NOT "02_Peripheral".IN.YikamaTanki.UstSeviyeSen AND NOT "02_Peripheral".IN.YikamaTanki.CriticalSeviyeSen AND ("03_HmiData".SuDolumVanasi_Ac OR (NOT "03_HmiData".SuDolumVanasi_Kapat AND "HmiSuDolumVana"));
END_REGION

REGION Network 18
   RUNG wire#powerrail
      Contact( "02_Peripheral".IN.AcilStop )
      Contact( "01_System".Process.Manuel_Normal )
      Contact( "03_HmiData".SuDolumVanasi_Kapat )
      Coil( #bEmpty )
   END_RUNG
   // the same network as SCL:
   #bEmpty := "02_Peripheral".IN.AcilStop AND "01_System".Process.Manuel_Normal AND "03_HmiData".SuDolumVanasi_Kapat;
END_REGION
END_FUNCTION_BLOCK

FUNCTION_BLOCK "21_Alarm"   // FB10, LAD
{ S7_Optimized_Access := 'TRUE' }
VERSION : 0.1
   VAR
      SirkulasyonVanaKapat : TON_TIME;
      SirkulasyonVanaAc : TON_TIME;
      DolumVanasiAc : TON_TIME;
      DolumVanasiKapat : TON_TIME;
      AsitTahliyeVanasiAc : TON_TIME;
      AsitTahliyeVanasiKapat : TON_TIME;
      UcYolluVanaAc : TON_TIME;
      UcYolluVanaKapat : TON_TIME;
      KuyuTahliyeVanaAc : TON_TIME;
      KuyuTahliyeVanaKapat : TON_TIME;
      IBCTahliyeVanaAc : TON_TIME;
      IBCTahliyeVanaKapat : TON_TIME;
   END_VAR
   VAR_TEMP
      tWatchdogInterval : Time;
   END_VAR
BEGIN

REGION Network 1
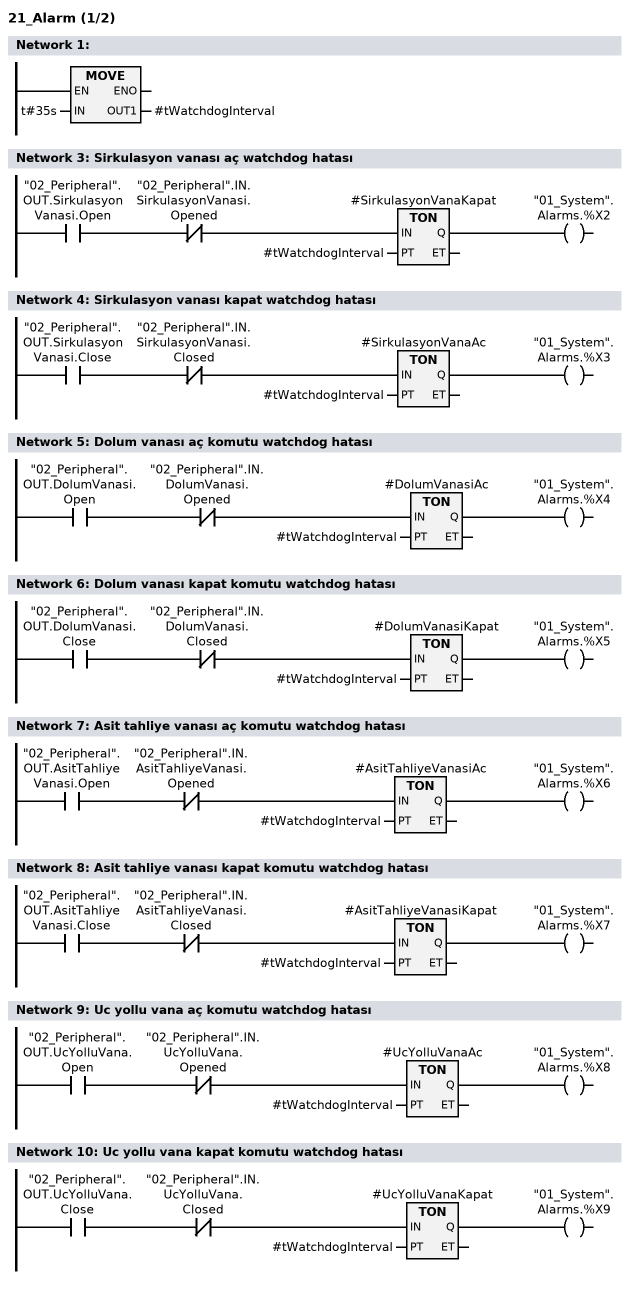
   RUNG wire#powerrail
      Move(in := t#35s, out1 => #tWatchdogInterval)
   END_RUNG
   // the same network as SCL:
   #tWatchdogInterval := t#35s;
END_REGION

REGION Network 2 (SCL): aCİL STOP ve TERMİK HATA
   "01_System".Alarms.%X0 := NOT "02_Peripheral".IN.AcilStop;
   "01_System".Alarms.%X1 := "02_Peripheral".IN.TermikAnaPompa;
END_REGION

REGION Network 3: Sirkulasyon vanası aç watchdog hatası
   #SirkulasyonVanaKapat(IN := "02_Peripheral".OUT.SirkulasyonVanasi.Open AND NOT "02_Peripheral".IN.SirkulasyonVanasi.Opened,   // TON
                         PT := #tWatchdogInterval);
   "01_System".Alarms.%X2 := #SirkulasyonVanaKapat.Q;
END_REGION

REGION Network 4: Sirkulasyon vanası kapat watchdog hatası
   #SirkulasyonVanaAc(IN := "02_Peripheral".OUT.SirkulasyonVanasi.Close AND NOT "02_Peripheral".IN.SirkulasyonVanasi.Closed,   // TON
                      PT := #tWatchdogInterval);
   "01_System".Alarms.%X3 := #SirkulasyonVanaAc.Q;
END_REGION

REGION Network 5: Dolum vanası aç komutu watchdog hatası
   #DolumVanasiAc(IN := "02_Peripheral".OUT.DolumVanasi.Open AND NOT "02_Peripheral".IN.DolumVanasi.Opened,   // TON
                  PT := #tWatchdogInterval);
   "01_System".Alarms.%X4 := #DolumVanasiAc.Q;
END_REGION

REGION Network 6: Dolum vanası kapat komutu watchdog hatası
   #DolumVanasiKapat(IN := "02_Peripheral".OUT.DolumVanasi.Close AND NOT "02_Peripheral".IN.DolumVanasi.Closed,   // TON
                     PT := #tWatchdogInterval);
   "01_System".Alarms.%X5 := #DolumVanasiKapat.Q;
END_REGION

REGION Network 7: Asit tahliye vanası aç komutu watchdog hatası
   #AsitTahliyeVanasiAc(IN := "02_Peripheral".OUT.AsitTahliyeVanasi.Open AND NOT "02_Peripheral".IN.AsitTahliyeVanasi.Opened,   // TON
                        PT := #tWatchdogInterval);
   "01_System".Alarms.%X6 := #AsitTahliyeVanasiAc.Q;
END_REGION

REGION Network 8: Asit tahliye vanası kapat komutu watchdog hatası
   #AsitTahliyeVanasiKapat(IN := "02_Peripheral".OUT.AsitTahliyeVanasi.Close AND NOT "02_Peripheral".IN.AsitTahliyeVanasi.Closed,   // TON
                           PT := #tWatchdogInterval);
   "01_System".Alarms.%X7 := #AsitTahliyeVanasiKapat.Q;
END_REGION

REGION Network 9: Uc yollu vana aç komutu watchdog hatası
   #UcYolluVanaAc(IN := "02_Peripheral".OUT.UcYolluVana.Open AND NOT "02_Peripheral".IN.UcYolluVana.Opened,   // TON
                  PT := #tWatchdogInterval);
   "01_System".Alarms.%X8 := #UcYolluVanaAc.Q;
END_REGION

REGION Network 10: Uc yollu vana kapat komutu watchdog hatası
   #UcYolluVanaKapat(IN := "02_Peripheral".OUT.UcYolluVana.Close AND NOT "02_Peripheral".IN.UcYolluVana.Closed,   // TON
                     PT := #tWatchdogInterval);
   "01_System".Alarms.%X9 := #UcYolluVanaKapat.Q;
END_REGION

REGION Network 11: Kuyu aktarım vanası aç komutu watchdog hatası
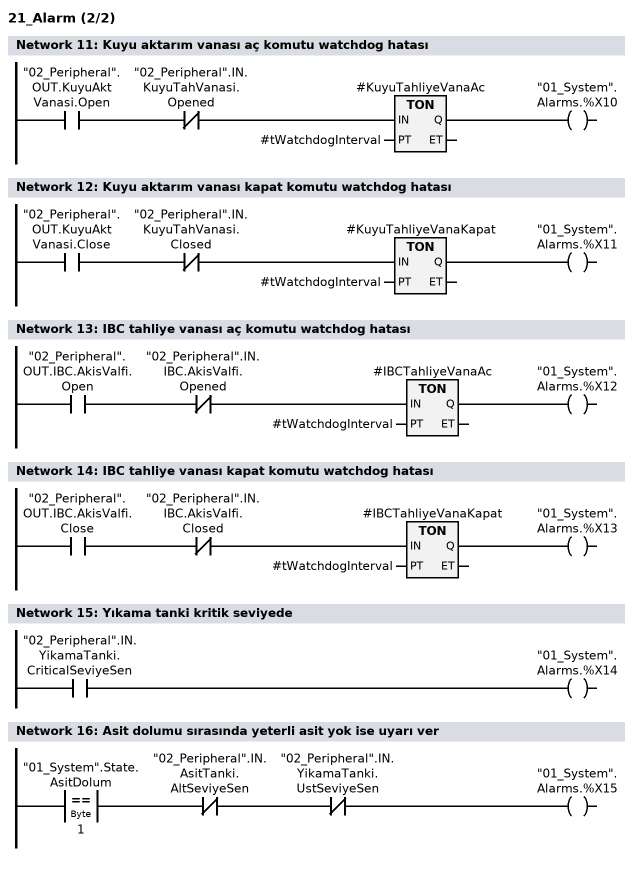
   #KuyuTahliyeVanaAc(IN := "02_Peripheral".OUT.KuyuAktVanasi.Open AND NOT "02_Peripheral".IN.KuyuTahVanasi.Opened,   // TON
                      PT := #tWatchdogInterval);
   "01_System".Alarms.%X10 := #KuyuTahliyeVanaAc.Q;
END_REGION

REGION Network 12: Kuyu aktarım vanası kapat komutu watchdog hatası
   #KuyuTahliyeVanaKapat(IN := "02_Peripheral".OUT.KuyuAktVanasi.Close AND NOT "02_Peripheral".IN.KuyuTahVanasi.Closed,   // TON
                         PT := #tWatchdogInterval);
   "01_System".Alarms.%X11 := #KuyuTahliyeVanaKapat.Q;
END_REGION

REGION Network 13: IBC tahliye vanası aç komutu watchdog hatası
   #IBCTahliyeVanaAc(IN := "02_Peripheral".OUT.IBC.AkisValfi.Open AND NOT "02_Peripheral".IN.IBC.AkisValfi.Opened,   // TON
                     PT := #tWatchdogInterval);
   "01_System".Alarms.%X12 := #IBCTahliyeVanaAc.Q;
END_REGION

REGION Network 14: IBC tahliye vanası kapat komutu watchdog hatası
   #IBCTahliyeVanaKapat(IN := "02_Peripheral".OUT.IBC.AkisValfi.Close AND NOT "02_Peripheral".IN.IBC.AkisValfi.Closed,   // TON
                        PT := #tWatchdogInterval);
   "01_System".Alarms.%X13 := #IBCTahliyeVanaKapat.Q;
END_REGION

REGION Network 15: Yıkama tanki kritik seviyede
   RUNG wire#powerrail
      Contact( "02_Peripheral".IN.YikamaTanki.CriticalSeviyeSen )
      Coil( "01_System".Alarms.%X14 )
   END_RUNG
   // the same network as SCL:
   "01_System".Alarms.%X14 := "02_Peripheral".IN.YikamaTanki.CriticalSeviyeSen;
END_REGION

REGION Network 16: Asit dolumu sırasında yeterli asit yok ise uyarı ver
   RUNG wire#powerrail
      { S7_Templates := "SrcType := Byte" } EQ_Contact(in1 := "01_System".State.AsitDolum, in2 := 1)
      I_Contact( "02_Peripheral".IN.AsitTanki.AltSeviyeSen )
      I_Contact( "02_Peripheral".IN.YikamaTanki.UstSeviyeSen )
      Coil( "01_System".Alarms.%X15 )
   END_RUNG
   // the same network as SCL:
   "01_System".Alarms.%X15 := ("01_System".State.AsitDolum = 1) AND NOT "02_Peripheral".IN.AsitTanki.AltSeviyeSen AND NOT "02_Peripheral".IN.YikamaTanki.UstSeviyeSen;
END_REGION
END_FUNCTION_BLOCK

FUNCTION "20_Visualization" : Void   // FC1, SCL
{ S7_Optimized_Access := 'TRUE' }
VERSION : 0.1
   VAR_INPUT
      bAsitDolumStarted : Bool;
      bAsitSirkulasyonStarted : Bool;
      bAsitTahliyeStarted : Bool;
      bTemizSuDolumStarted : Bool;
      bTemizSuSirStarted : Bool;
      bTemizSuTahliyeStarted : Bool;
      IBCTahStarted : Bool;
   END_VAR
   VAR_TEMP
      dnAsitSirTimeToDint : DInt;
      dnAsitSitCalculateMin : DInt;
      dnAsitSitCalculateSec : DInt;
      dnSuSirTimeToDint : DInt;
      dnSuSitCalculateMin : DInt;
      dnSuSitCalculateSec : DInt;
   END_VAR
BEGIN
   REGION "Info mesajı"

       IF NOT "02_Peripheral".IN.AcilStop THEN
           "01_System".SystemInfo := 'ACIL STOP BASILI !!!';

       ELSIF NOT "02_Peripheral".IN.AsitTanki.KapiSwitch THEN
           "01_System".SystemInfo := 'Asit tanki kapisi acik...';
       ELSIF NOT "02_Peripheral".IN.YikamaTanki.KapiSwitch1 THEN
           "01_System".SystemInfo := 'Yikama tanki kapisi acik...';

       ELSIF #bAsitDolumStarted THEN  // Asit dolumu
           IF NOT "02_Peripheral".IN.AsitTanki.AltSeviyeSen
               AND NOT "02_Peripheral".IN.YikamaTanki.UstSeviyeSen THEN
               "01_System".SystemInfo := 'Asit dolumu yapilamadi';
           ELSIF NOT "AsitDoldurSeq_AnaPompa_Run" THEN
               "01_System".SystemInfo := 'Vanalar bekleniyor...';
           ELSE
               "01_System".SystemInfo := 'Asit dolumu yapiliyor';
           END_IF;

       ELSIF #bAsitSirkulasyonStarted THEN //Asit sirkulasyonu
           IF NOT "02_Peripheral".IN.AsitTanki.KapiSwitch
               OR NOT "02_Peripheral".IN.YikamaTanki.KapiSwitch1
           THEN
               "01_System".SystemInfo := 'Kapilar acik';
           ELSIF NOT "AsitSirkulas_AnaPompa_Run" THEN
                   "01_System".SystemInfo := 'Vanalar bekleniyor...';
           ELSE
                   "01_System".SystemInfo := 'Asit sirkulasyonu yapiliyor';
           END_IF;

       ELSIF #bAsitTahliyeStarted THEN //Asit tahliyesi
           IF NOT "AsitTahliyesi_Pompa_Run" THEN
               "01_System".SystemInfo := 'Vanalar bekleniyor...';
           ELSE
               "01_System".SystemInfo := 'Asit tahliyesi yapiliyor';
           END_IF;

       ELSIF #bTemizSuDolumStarted THEN    // Temiz su dolumu
           IF NOT "AsitTahliyesi_Pompa_Run" THEN
               "01_System".SystemInfo := 'Vanalar bekleniyor...';
           ELSE
               "01_System".SystemInfo := 'Asit tahliyesi yapiliyor';
           END_IF;

       ELSIF #bTemizSuSirStarted THEN  //Temiz su sirkulasyonu
           IF NOT "02_Peripheral".IN.AsitTanki.KapiSwitch
               OR NOT "02_Peripheral".IN.YikamaTanki.KapiSwitch1
           THEN
               "01_System".SystemInfo := 'Kapilar acik';
           ELSIF NOT "SuSirkulasyon_Pompa_Run" THEN
               "01_System".SystemInfo := 'Vanalar bekleniyor...';
           ELSE
               "01_System".SystemInfo := 'Su sirkulasyonu yapiliyor';
           END_IF;

       ELSIF #bTemizSuTahliyeStarted THEN  //Temiz su tahliyesi
           IF NOT "SuTahliyesi_Pompa_Run" THEN
               "01_System".SystemInfo := 'Vanalar bekleniyor...';
           ELSE
               "01_System".SystemInfo := 'Su tahliyesi yapiliyor';
           END_IF;

       ELSIF #IBCTahStarted THEN   // IBC tahliyesi
           IF NOT "IBCTahliye_IBCpompa_Run" THEN
               "01_System".SystemInfo := 'Vanalar bekleniyor...';
           ELSE
               "01_System".SystemInfo := 'IBC pompa calisiyor...';
           END_IF;

       ELSE
           "01_System".SystemInfo := 'Sistem bosta!!!';

       END_IF;

   END_REGION

   REGION "Ana ekran buton visibility - IPTAL" 

       IF "03_HmiData".Started.AsitDolum THEN
           "03_HmiData".Visualization.nMode := 1;
       ELSIF "03_HmiData".Started.AsitSirkulasyon THEN
           "03_HmiData".Visualization.nMode := 2;
       ELSIF "03_HmiData".Started.AsitTahliye THEN
           "03_HmiData".Visualization.nMode := 3;
       ELSIF "03_HmiData".Started.TemizSuSirkulasyon THEN
           "03_HmiData".Visualization.nMode := 4;
       ELSIF "03_HmiData".Started.TemizSuTahliye THEN
           "03_HmiData".Visualization.nMode := 5;
       ELSIF "03_HmiData".Started.IBCTahliye THEN
           "03_HmiData".Visualization.nMode := 6;
       ELSE
           "03_HmiData".Visualization.nMode := 0;
       END_IF;

       CASE "03_HmiData".Visualization.nMode OF

           0:
               "03_HmiData".Visualization.Visibility.AsitDolum := false;
               "03_HmiData".Visualization.Visibility.AsitSirkulasyon := false;
               "03_HmiData".Visualization.Visibility.AsitTahliyesi := false;
               "03_HmiData".Visualization.Visibility.TemizSuSirkulasyon := false;
               "03_HmiData".Visualization.Visibility.TemizSuTahliye := false;
               "03_HmiData".Visualization.Visibility.IBCTaliye := false;
           1:
               "03_HmiData".Visualization.Visibility.AsitDolum := false;
               "03_HmiData".Visualization.Visibility.AsitSirkulasyon := true;
               "03_HmiData".Visualization.Visibility.AsitTahliyesi := true;
               "03_HmiData".Visualization.Visibility.TemizSuSirkulasyon := true;
               "03_HmiData".Visualization.Visibility.TemizSuTahliye := true;
               "03_HmiData".Visualization.Visibility.IBCTaliye := true;
           2:
               "03_HmiData".Visualization.Visibility.AsitDolum := true;
               "03_HmiData".Visualization.Visibility.AsitSirkulasyon := false;
               "03_HmiData".Visualization.Visibility.AsitTahliyesi := true;
               "03_HmiData".Visualization.Visibility.TemizSuSirkulasyon := true;
               "03_HmiData".Visualization.Visibility.TemizSuTahliye := true;
               "03_HmiData".Visualization.Visibility.IBCTaliye := true;
           3:
               "03_HmiData".Visualization.Visibility.AsitDolum := true;
               "03_HmiData".Visualization.Visibility.AsitSirkulasyon := true;
               "03_HmiData".Visualization.Visibility.AsitTahliyesi := false;
               "03_HmiData".Visualization.Visibility.TemizSuSirkulasyon := true;
               "03_HmiData".Visualization.Visibility.TemizSuTahliye := true;
               "03_HmiData".Visualization.Visibility.IBCTaliye := true;
           4:
               "03_HmiData".Visualization.Visibility.AsitDolum := true;
               "03_HmiData".Visualization.Visibility.AsitSirkulasyon := true;
               "03_HmiData".Visualization.Visibility.AsitTahliyesi := true;
               "03_HmiData".Visualization.Visibility.TemizSuSirkulasyon := false;
               "03_HmiData".Visualization.Visibility.TemizSuTahliye := true;
               "03_HmiData".Visualization.Visibility.IBCTaliye := true;
           5:
               "03_HmiData".Visualization.Visibility.AsitDolum := true;
               "03_HmiData".Visualization.Visibility.AsitSirkulasyon := true;
               "03_HmiData".Visualization.Visibility.AsitTahliyesi := true;
               "03_HmiData".Visualization.Visibility.TemizSuSirkulasyon := true;
               "03_HmiData".Visualization.Visibility.TemizSuTahliye := false;
               "03_HmiData".Visualization.Visibility.IBCTaliye := true;
           6:
               "03_HmiData".Visualization.Visibility.AsitDolum := true;
               "03_HmiData".Visualization.Visibility.AsitSirkulasyon := true;
               "03_HmiData".Visualization.Visibility.AsitTahliyesi := true;
               "03_HmiData".Visualization.Visibility.TemizSuSirkulasyon := true;
               "03_HmiData".Visualization.Visibility.TemizSuTahliye := true;
               "03_HmiData".Visualization.Visibility.IBCTaliye := false;
           ELSE
               "03_HmiData".Visualization.Visibility.AsitDolum := false;
               "03_HmiData".Visualization.Visibility.AsitSirkulasyon := false;
               "03_HmiData".Visualization.Visibility.AsitTahliyesi := false;
               "03_HmiData".Visualization.Visibility.TemizSuSirkulasyon := false;
               "03_HmiData".Visualization.Visibility.TemizSuTahliye := false;
               "03_HmiData".Visualization.Visibility.IBCTaliye := false;
       END_CASE;

   END_REGION

   REGION "Manuel ekran buton visibility - IPTAL"

       "03_HmiData".Visualization.Visibility.Manuel.SirkulasyonVanaKapat := "HmiSirkVana_Ac_Mem";
       "03_HmiData".Visualization.Visibility.Manuel.SirkulasyonVanaAc := "HmiSirkVana_Kapat_Mem";

       "03_HmiData".Visualization.Visibility.Manuel.DolumVanaKapat := "HmiDolumVana_Ac_Mem";
       "03_HmiData".Visualization.Visibility.Manuel.DolumVanaAc := "HmiDolumVana_Kapat_Mem";

       "03_HmiData".Visualization.Visibility.Manuel.AsitTahVanaKapat := "HmiAsitTahVana_Ac_Mem";
       "03_HmiData".Visualization.Visibility.Manuel.AsitTahVanaAc := "HmiAsitTahVana_Kapat_Mem";

       "03_HmiData".Visualization.Visibility.Manuel.UcYolluVanaKapat := "HmiUcYolluVana_Ac_Mem";
       "03_HmiData".Visualization.Visibility.Manuel.UcYolluVanaAc := "HmiUcYolluVana_Kapat_Mem";

       "03_HmiData".Visualization.Visibility.Manuel.KuyuTahVanaKapat := "HmiKuyuVana_Ac_Mem";
       "03_HmiData".Visualization.Visibility.Manuel.KuyuTahVanaAc := "HmiKuyuVana_Kapat_Mem";

       "03_HmiData".Visualization.Visibility.Manuel.IBCVanaKapat := "HmiIBCVana_Ac_Mem";
       "03_HmiData".Visualization.Visibility.Manuel.IBCVanaAc := "HmiIBCVana_Kapat_Mem";

   END_REGION

   REGION "HMI için timer çevrimi"

       #dnAsitSirTimeToDint := TIME_TO_DINT(IN := "AsitSirkTimer_DB".ET);
       #dnAsitSitCalculateMin := (#dnAsitSirTimeToDint / 60000);
       #dnAsitSitCalculateSec := (#dnAsitSirTimeToDint MOD 60000) / 1000;

       #dnSuSirTimeToDint := TIME_TO_DINT(IN := "SuSirkTimer_DB".ET);
       #dnSuSitCalculateMin := (#dnSuSirTimeToDint / 60000);
       #dnSuSitCalculateSec := (#dnSuSirTimeToDint MOD 60000) / 1000;

       IF "03_HmiData".Started.AsitSirkulasyon THEN
           "03_HmiData".Visualization.ActTimerMin := #dnAsitSitCalculateMin;
           "03_HmiData".Visualization.ActTimerSec := #dnAsitSitCalculateSec;
       ELSIF "03_HmiData".Started.TemizSuSirkulasyon THEN
   //        "01_System".ConvertTimeToDint := TIME_TO_DINT(IN := "SuSirkTimer_DB".ET);
           "03_HmiData".Visualization.ActTimerMin := #dnSuSitCalculateMin;
           "03_HmiData".Visualization.ActTimerSec := #dnSuSitCalculateSec;
       ELSE
           "03_HmiData".Visualization.ActTimerMin := 0;
           "03_HmiData".Visualization.ActTimerSec := 0;
       END_IF;

   END_REGION
END_FUNCTION

FUNCTION "12_AsitSirkulasyonSeq" : Void   // FC2, LAD
{ S7_Optimized_Access := 'TRUE' }
VERSION : 0.1
   VAR_TEMP   // added for the SCL form of the ladder/FBD networks
      _w1 : Bool;
      _w2 : Bool;
   END_VAR
BEGIN

REGION Network 1
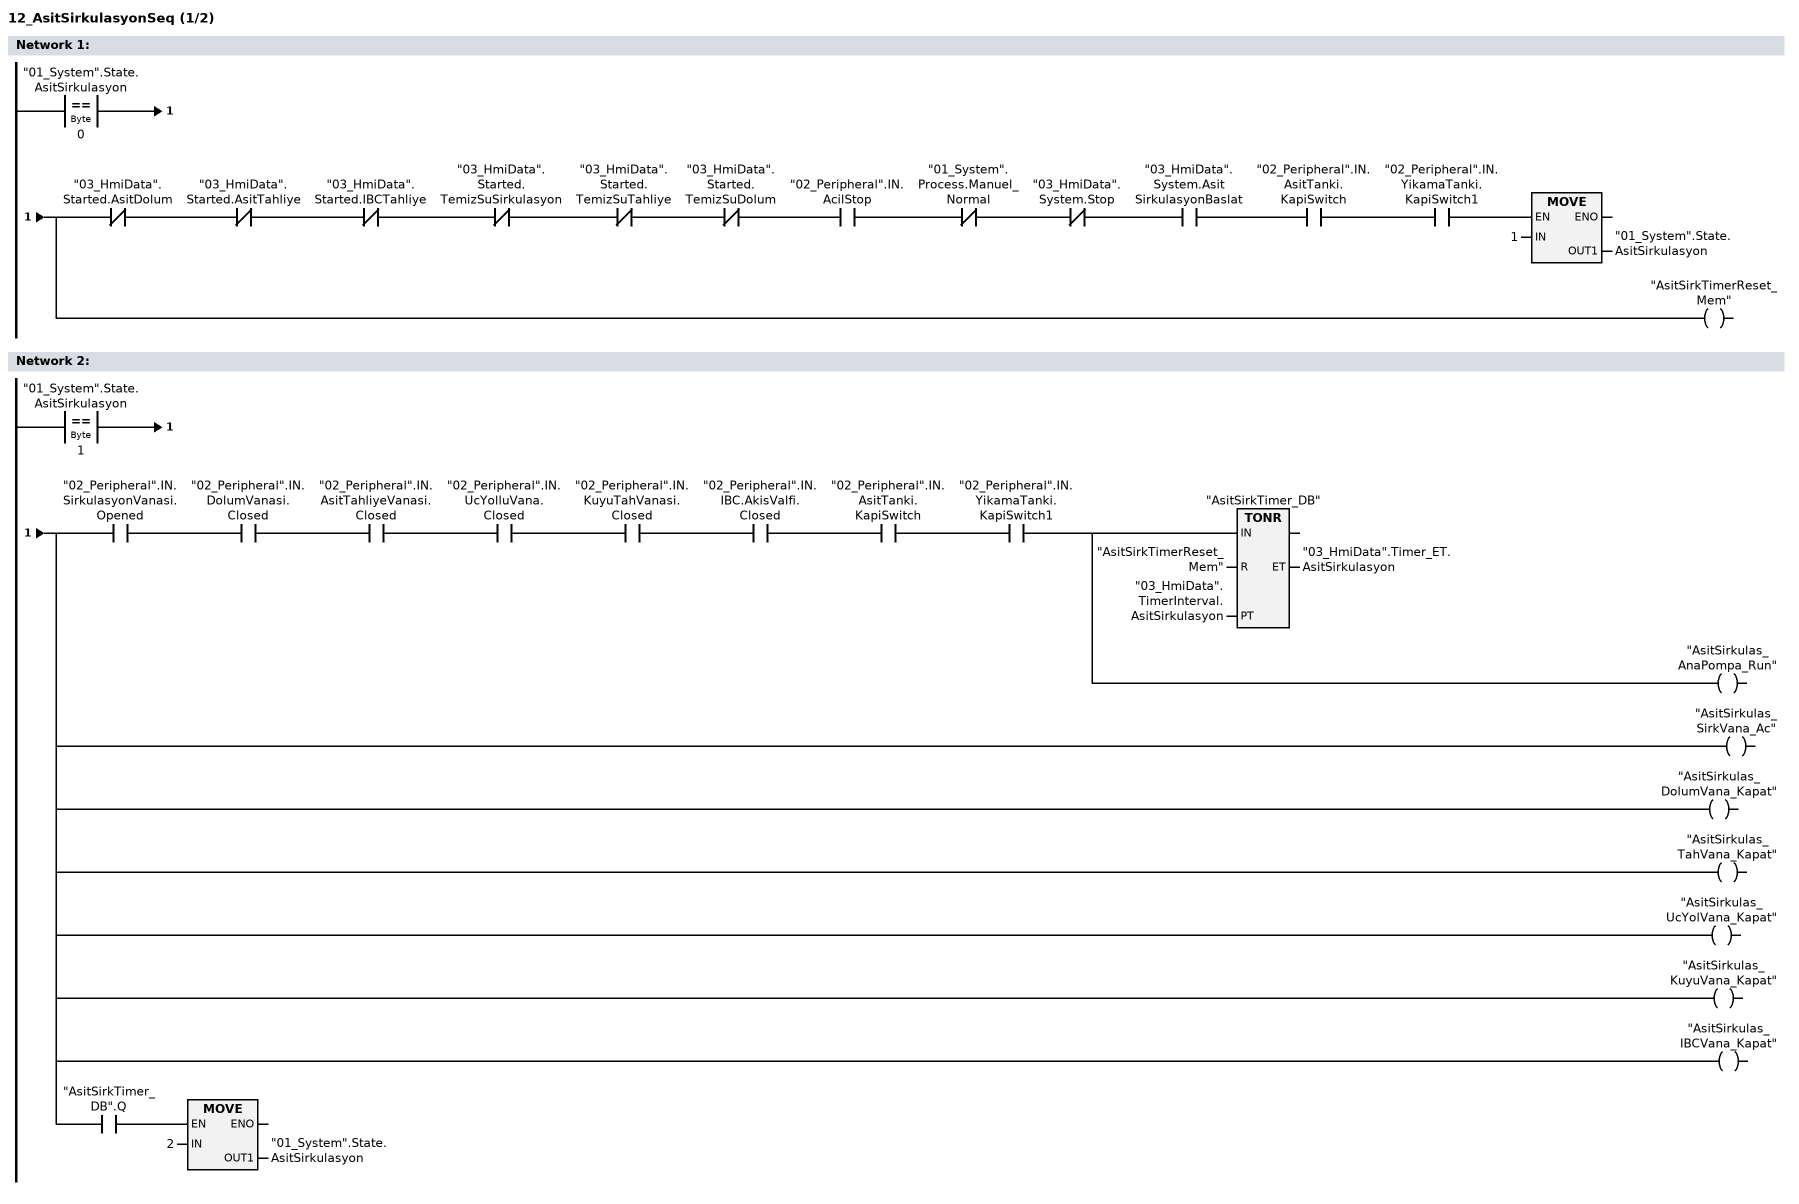
   RUNG wire#powerrail
      { S7_Templates := "SrcType := Byte" } EQ_Contact(in1 := "01_System".State.AsitSirkulasyon, in2 := 0)
      wire#w1
      I_Contact( "03_HmiData".Started.AsitDolum )
      I_Contact( "03_HmiData".Started.AsitTahliye )
      I_Contact( "03_HmiData".Started.IBCTahliye )
      I_Contact( "03_HmiData".Started.TemizSuSirkulasyon )
      I_Contact( "03_HmiData".Started.TemizSuTahliye )
      I_Contact( "03_HmiData".Started.TemizSuDolum )
      Contact( "02_Peripheral".IN.AcilStop )
      I_Contact( "01_System".Process.Manuel_Normal )
      I_Contact( "03_HmiData".System.Stop )
      Contact( "03_HmiData".System.AsitSirkulasyonBaslat )
      Contact( "02_Peripheral".IN.AsitTanki.KapiSwitch )
      Contact( "02_Peripheral".IN.YikamaTanki.KapiSwitch1 )
      Move(in := 1, out1 => "01_System".State.AsitSirkulasyon)
   END_RUNG
   RUNG wire#w1
      Coil( "AsitSirkTimerReset_Mem" )
   END_RUNG
   // the same network as SCL:
   #_w1 := "01_System".State.AsitSirkulasyon = 0;
   IF #_w1 AND NOT "03_HmiData".Started.AsitDolum AND NOT "03_HmiData".Started.AsitTahliye AND NOT "03_HmiData".Started.IBCTahliye AND NOT "03_HmiData".Started.TemizSuSirkulasyon AND NOT "03_HmiData".Started.TemizSuTahliye AND NOT "03_HmiData".Started.TemizSuDolum AND "02_Peripheral".IN.AcilStop AND NOT "01_System".Process.Manuel_Normal AND NOT "03_HmiData".System.Stop AND "03_HmiData".System.AsitSirkulasyonBaslat AND "02_Peripheral".IN.AsitTanki.KapiSwitch AND "02_Peripheral".IN.YikamaTanki.KapiSwitch1 THEN
       "01_System".State.AsitSirkulasyon := 1;
   END_IF;
   "AsitSirkTimerReset_Mem" := #_w1;
END_REGION

REGION Network 2
   #_w1 := "01_System".State.AsitSirkulasyon = 1;
   #_w2 := #_w1 AND "02_Peripheral".IN.SirkulasyonVanasi.Opened AND "02_Peripheral".IN.DolumVanasi.Closed AND "02_Peripheral".IN.AsitTahliyeVanasi.Closed AND "02_Peripheral".IN.UcYolluVana.Closed AND "02_Peripheral".IN.KuyuTahVanasi.Closed AND "02_Peripheral".IN.IBC.AkisValfi.Closed AND "02_Peripheral".IN.AsitTanki.KapiSwitch AND "02_Peripheral".IN.YikamaTanki.KapiSwitch1;
   "AsitSirkTimer_DB".TONR(IN := #_w2,
                           R := "AsitSirkTimerReset_Mem",
                           PT := "03_HmiData".TimerInterval.AsitSirkulasyon,
                           ET => "03_HmiData".Timer_ET.AsitSirkulasyon);
   "AsitSirkulas_AnaPompa_Run" := #_w2;
   "AsitSirkulas_SirkVana_Ac" := #_w1;
   "AsitSirkulas_DolumVana_Kapat" := #_w1;
   "AsitSirkulas_TahVana_Kapat" := #_w1;
   "AsitSirkulas_UcYolVana_Kapat" := #_w1;
   "AsitSirkulas_KuyuVana_Kapat" := #_w1;
   "AsitSirkulas_IBCVana_Kapat" := #_w1;
   IF #_w1 AND "AsitSirkTimer_DB".Q THEN "01_System".State.AsitSirkulasyon := 2; END_IF;
END_REGION

REGION Network 3
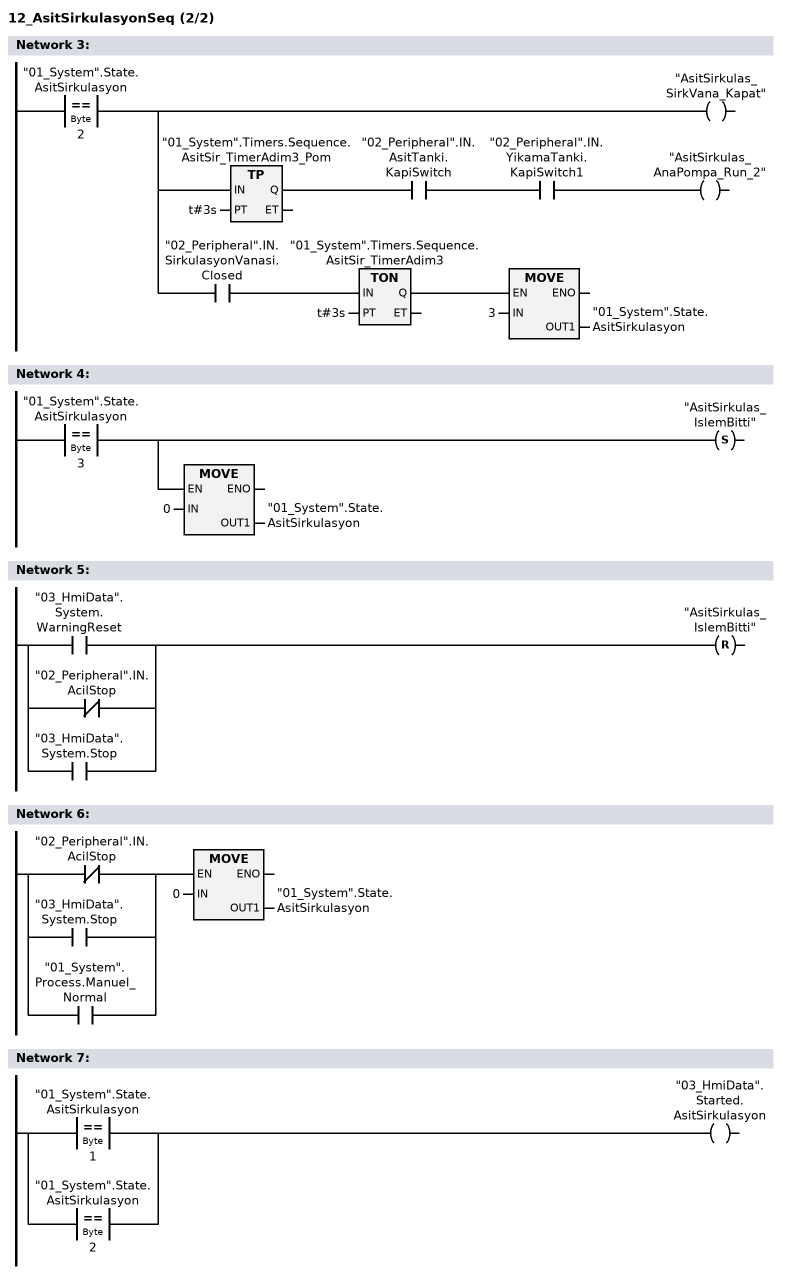
   "AsitSirkulas_SirkVana_Kapat" := "01_System".State.AsitSirkulasyon = 2;
   "01_System".Timers.Sequence.AsitSir_TimerAdim3_Pom.TP(IN := "AsitSirkulas_SirkVana_Kapat", PT := t#3s);
   "AsitSirkulas_AnaPompa_Run_2" := "01_System".Timers.Sequence.AsitSir_TimerAdim3_Pom.Q AND "02_Peripheral".IN.AsitTanki.KapiSwitch AND "02_Peripheral".IN.YikamaTanki.KapiSwitch1;
   "01_System".Timers.Sequence.AsitSir_TimerAdim3.TON(IN := "AsitSirkulas_SirkVana_Kapat" AND "02_Peripheral".IN.SirkulasyonVanasi.Closed,
                           PT := t#3s);
   IF "01_System".Timers.Sequence.AsitSir_TimerAdim3.Q THEN "01_System".State.AsitSirkulasyon := 3; END_IF;
END_REGION

REGION Network 4
   RUNG wire#powerrail
      { S7_Templates := "SrcType := Byte" } EQ_Contact(in1 := "01_System".State.AsitSirkulasyon, in2 := 3)
      wire#w1
      S_Coil( "AsitSirkulas_IslemBitti" )
   END_RUNG
   RUNG wire#w1
      Move(in := 0, out1 => "01_System".State.AsitSirkulasyon)
   END_RUNG
   // the same network as SCL:
   IF "01_System".State.AsitSirkulasyon = 3 THEN
       "AsitSirkulas_IslemBitti" := TRUE;
       "01_System".State.AsitSirkulasyon := 0;
   END_IF;
END_REGION

REGION Network 5
   RUNG wire#powerrail
      Contact( "03_HmiData".System.WarningReset )
      wire#w1
      R_Coil( "AsitSirkulas_IslemBitti" )
   END_RUNG
   RUNG wire#powerrail
      I_Contact( "02_Peripheral".IN.AcilStop )
   END_RUNG wire#w1
   RUNG wire#powerrail
      Contact( "03_HmiData".System.Stop )
   END_RUNG wire#w1
   // the same network as SCL:
   IF "03_HmiData".System.WarningReset OR NOT "02_Peripheral".IN.AcilStop OR "03_HmiData".System.Stop THEN
       "AsitSirkulas_IslemBitti" := FALSE;
   END_IF;
END_REGION

REGION Network 6
   RUNG wire#powerrail
      I_Contact( "02_Peripheral".IN.AcilStop )
      wire#w1
      Move(in := 0, out1 => "01_System".State.AsitSirkulasyon)
   END_RUNG
   RUNG wire#powerrail
      Contact( "03_HmiData".System.Stop )
   END_RUNG wire#w1
   RUNG wire#powerrail
      Contact( "01_System".Process.Manuel_Normal )
   END_RUNG wire#w1
   // the same network as SCL:
   IF NOT "02_Peripheral".IN.AcilStop OR "03_HmiData".System.Stop OR "01_System".Process.Manuel_Normal THEN
       "01_System".State.AsitSirkulasyon := 0;
   END_IF;
END_REGION

REGION Network 7
   RUNG wire#powerrail
      { S7_Templates := "SrcType := Byte" } EQ_Contact(in1 := "01_System".State.AsitSirkulasyon, in2 := 1)
      wire#w1
      Coil( "03_HmiData".Started.AsitSirkulasyon )
   END_RUNG
   RUNG wire#powerrail
      { S7_Templates := "SrcType := Byte" } EQ_Contact(in1 := "01_System".State.AsitSirkulasyon, in2 := 2)
   END_RUNG wire#w1
   // the same network as SCL:
   "03_HmiData".Started.AsitSirkulasyon := ("01_System".State.AsitSirkulasyon = 1) OR ("01_System".State.AsitSirkulasyon = 2);
END_REGION
END_FUNCTION

FUNCTION "22_Peripheral" : Void   // FC3, SCL
{ S7_Optimized_Access := 'TRUE' }
VERSION : 0.1
BEGIN
   // ==================INPUT=============================
   "02_Peripheral".IN.AcilStop := "I0.0"
                                   AND "I0.1";

   "02_Peripheral".IN.YikamaTanki.AltSeviyeSen         := "I0.2";
   //"02_Peripheral".IN.YikamaTanki.UstSeviyeSen         := "I0.3";
   //"02_Peripheral".IN.YikamaTanki.CriticalSeviyeSen    := "I0.7";
   "02_Peripheral".IN.YikamaTanki.UstSeviyeSen := "I0.7";
   "02_Peripheral".IN.YikamaTanki.CriticalSeviyeSen := "I0.3";

   "02_Peripheral".IN.AsitTanki.AltSeviyeSen           := "I0.4";
   "02_Peripheral".IN.AsitTanki.UstSeviyeSen           := "I0.5";
   "02_Peripheral".IN.YikamaTanki.KapiSwitch1          :=  "I0.6";

   "02_Peripheral".IN.AsitTanki.KapiSwitch :=      "I1.0";
   //"02_Peripheral".IN.TermikAnaPompa :=            "I1.1";
   "02_Peripheral".IN.SirkulasyonVanasi.Closed :=  "I1.2";
   "02_Peripheral".IN.SirkulasyonVanasi.Opened :=  "I1.3";
   "02_Peripheral".IN.DolumVanasi.Closed :=        "I1.4";
   "02_Peripheral".IN.DolumVanasi.Opened :=        "I1.5";
   "02_Peripheral".IN.AsitTahliyeVanasi.Closed :=  "I2.0";
   "02_Peripheral".IN.AsitTahliyeVanasi.Opened :=  "I2.1";
   "02_Peripheral".IN.UcYolluVana.Closed :=        "I2.2";
   "02_Peripheral".IN.UcYolluVana.Opened :=        "I2.3";
   "02_Peripheral".IN.KuyuTahVanasi.Closed :=      "I2.4";
   "02_Peripheral".IN.KuyuTahVanasi.Opened :=      "I2.5";
   "02_Peripheral".IN.IBC.AkisValfi.Closed :=      "I2.6";
   "02_Peripheral".IN.IBC.AkisValfi.Opened :=      "I2.7";
   // ====================END INPUT==============================


   //=================OUTPUT===========================
   "YesilLamba" :=             "02_Peripheral".Lamba.Yesil;
   "KirmiziLamba" :=           "02_Peripheral".Lamba.Kirmizi;
   "Siren" :=                  "02_Peripheral".Lamba.Siren;
   "SirkulasyonVanaKapat" :=   "02_Peripheral".OUT.SirkulasyonVanasi.Close;
   "SirkulasyonVanaAc" :=      "02_Peripheral".OUT.SirkulasyonVanasi.Open;
   "DolumVanaKapat" :=         "02_Peripheral".OUT.DolumVanasi.Close;
   "DolumVanaAc" :=            "02_Peripheral".OUT.DolumVanasi.Open;
   "AsitTahliyeVanaKapat" :=   "02_Peripheral".OUT.AsitTahliyeVanasi.Close;
   "AsitTahliyeVanaAc" :=      "02_Peripheral".OUT.AsitTahliyeVanasi.Open;
   "UcYolluVanaKapat" :=       "02_Peripheral".OUT.UcYolluVana.Close;
   "UcYolluVanaAc" :=          "02_Peripheral".OUT.UcYolluVana.Open;
   "KuyuTahliyeVanaKapat" :=   "02_Peripheral".OUT.KuyuAktVanasi.Close;
   "KuyuTahliyeVanaAc" :=      "02_Peripheral".OUT.KuyuAktVanasi.Open;
   "IBCVanaKapat" :=           "02_Peripheral".OUT.IBC.AkisValfi.Close;
   "IBCVanaAc" :=              "02_Peripheral".OUT.IBC.AkisValfi.Open;

   "AnaPompa" :=               "02_Peripheral".OUT.AnaPompa;
   "IBC_DiyaframPompa" :=      "02_Peripheral".OUT.IBC.PompaDiyafram;
   "KorKuyuPompasi" :=         "02_Peripheral".OUT.KorKuyuPompasi;
   "SuDolumVanasi" :=          "02_Peripheral".OUT.SuDolumVanasi;
   // ===============END OUTPUT==============================
END_FUNCTION

FUNCTION "11_AsitDolumSeq" : Void   // FC4, LAD
{ S7_Optimized_Access := 'TRUE' }
VERSION : 0.1
BEGIN

REGION Network 1
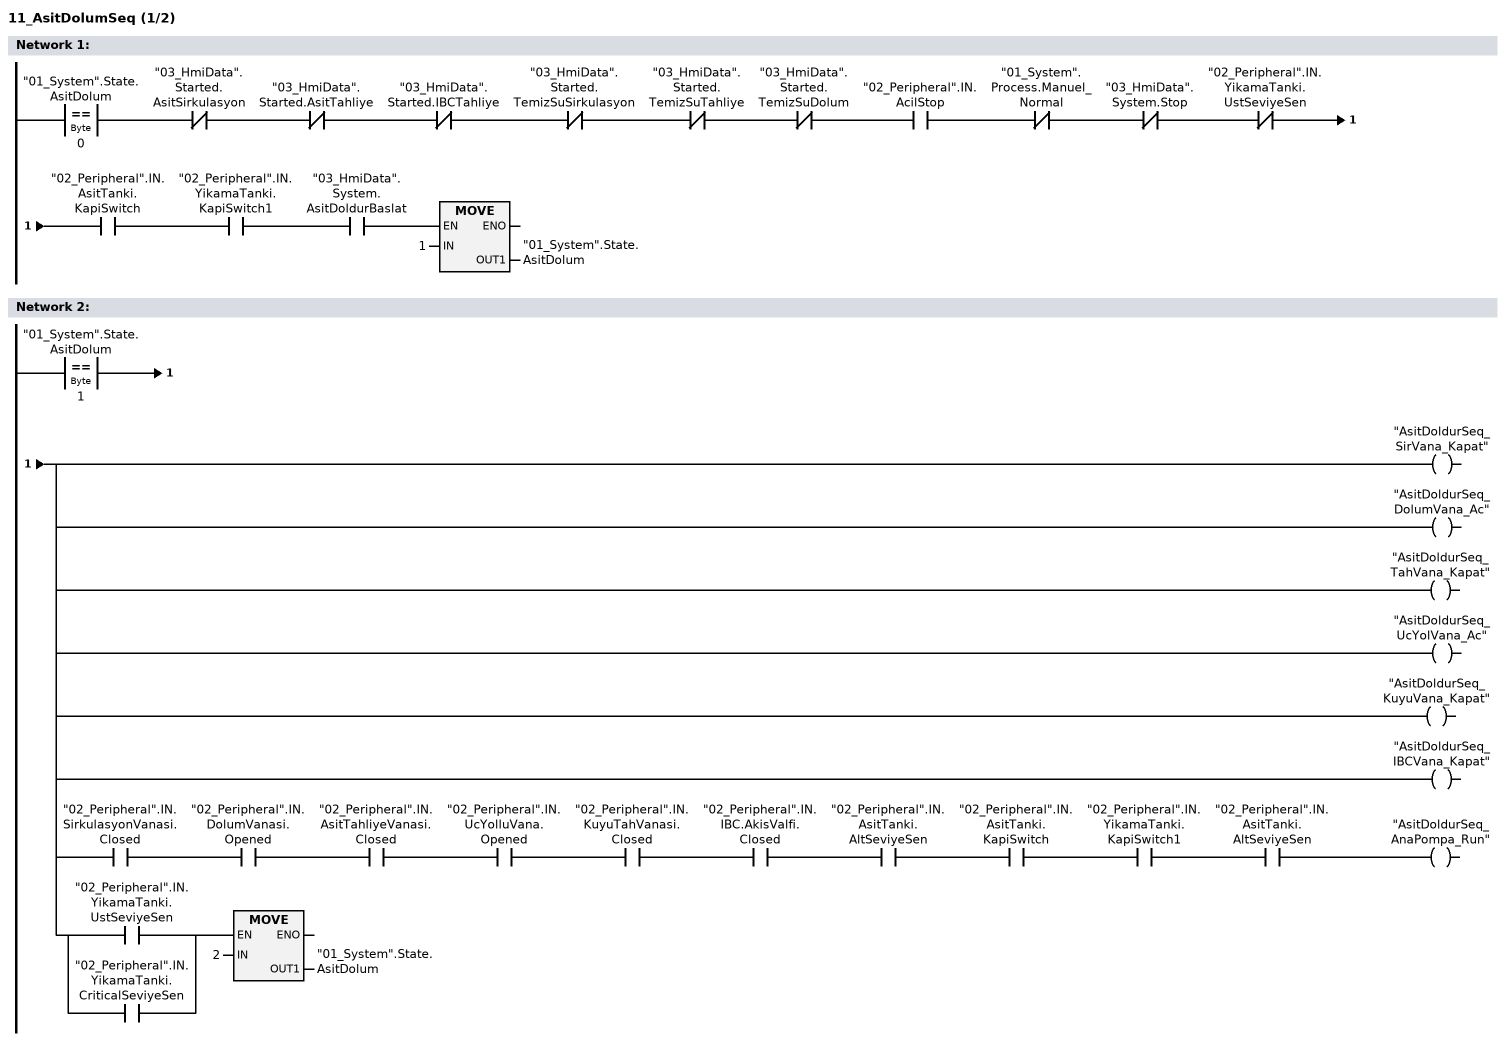
   RUNG wire#powerrail
      { S7_Templates := "SrcType := Byte" } EQ_Contact(in1 := "01_System".State.AsitDolum, in2 := 0)
      I_Contact( "03_HmiData".Started.AsitSirkulasyon )
      I_Contact( "03_HmiData".Started.AsitTahliye )
      I_Contact( "03_HmiData".Started.IBCTahliye )
      I_Contact( "03_HmiData".Started.TemizSuSirkulasyon )
      I_Contact( "03_HmiData".Started.TemizSuTahliye )
      I_Contact( "03_HmiData".Started.TemizSuDolum )
      Contact( "02_Peripheral".IN.AcilStop )
      I_Contact( "01_System".Process.Manuel_Normal )
      I_Contact( "03_HmiData".System.Stop )
      I_Contact( "02_Peripheral".IN.YikamaTanki.UstSeviyeSen )
      Contact( "02_Peripheral".IN.AsitTanki.KapiSwitch )
      Contact( "02_Peripheral".IN.YikamaTanki.KapiSwitch1 )
      Contact( "03_HmiData".System.AsitDoldurBaslat )
      Move(in := 1, out1 => "01_System".State.AsitDolum)
   END_RUNG
   // the same network as SCL:
   IF ("01_System".State.AsitDolum = 0) AND NOT "03_HmiData".Started.AsitSirkulasyon AND NOT "03_HmiData".Started.AsitTahliye AND NOT "03_HmiData".Started.IBCTahliye AND NOT "03_HmiData".Started.TemizSuSirkulasyon AND NOT "03_HmiData".Started.TemizSuTahliye AND NOT "03_HmiData".Started.TemizSuDolum AND "02_Peripheral".IN.AcilStop AND NOT "01_System".Process.Manuel_Normal AND NOT "03_HmiData".System.Stop AND NOT "02_Peripheral".IN.YikamaTanki.UstSeviyeSen AND "02_Peripheral".IN.AsitTanki.KapiSwitch AND "02_Peripheral".IN.YikamaTanki.KapiSwitch1 AND "03_HmiData".System.AsitDoldurBaslat THEN
       "01_System".State.AsitDolum := 1;
   END_IF;
END_REGION

REGION Network 2
   RUNG wire#powerrail
      { S7_Templates := "SrcType := Byte" } EQ_Contact(in1 := "01_System".State.AsitDolum, in2 := 1)
      wire#w1
      Coil( "AsitDoldurSeq_SirVana_Kapat" )
   END_RUNG
   RUNG wire#w1
      Coil( "AsitDoldurSeq_DolumVana_Ac" )
   END_RUNG
   RUNG wire#w1
      Coil( "AsitDoldurSeq_TahVana_Kapat" )
   END_RUNG
   RUNG wire#w1
      Coil( "AsitDoldurSeq_UcYolVana_Ac" )
   END_RUNG
   RUNG wire#w1
      Coil( "AsitDoldurSeq_KuyuVana_Kapat" )
   END_RUNG
   RUNG wire#w1
      Coil( "AsitDoldurSeq_IBCVana_Kapat" )
   END_RUNG
   RUNG wire#w1
      Contact( "02_Peripheral".IN.SirkulasyonVanasi.Closed )
      Contact( "02_Peripheral".IN.DolumVanasi.Opened )
      Contact( "02_Peripheral".IN.AsitTahliyeVanasi.Closed )
      Contact( "02_Peripheral".IN.UcYolluVana.Opened )
      Contact( "02_Peripheral".IN.KuyuTahVanasi.Closed )
      Contact( "02_Peripheral".IN.IBC.AkisValfi.Closed )
      Contact( "02_Peripheral".IN.AsitTanki.AltSeviyeSen )
      Contact( "02_Peripheral".IN.AsitTanki.KapiSwitch )
      Contact( "02_Peripheral".IN.YikamaTanki.KapiSwitch1 )
      Contact( "02_Peripheral".IN.AsitTanki.AltSeviyeSen )
      Coil( "AsitDoldurSeq_AnaPompa_Run" )
   END_RUNG
   RUNG wire#w1
      Contact( "02_Peripheral".IN.YikamaTanki.UstSeviyeSen )
      wire#w2
      Move(in := 2, out1 => "01_System".State.AsitDolum)
   END_RUNG
   RUNG wire#w1
      Contact( "02_Peripheral".IN.YikamaTanki.CriticalSeviyeSen )
   END_RUNG wire#w2
   // the same network as SCL:
   "AsitDoldurSeq_SirVana_Kapat" := "01_System".State.AsitDolum = 1;
   "AsitDoldurSeq_DolumVana_Ac" := "AsitDoldurSeq_SirVana_Kapat";
   "AsitDoldurSeq_TahVana_Kapat" := "AsitDoldurSeq_SirVana_Kapat";
   "AsitDoldurSeq_UcYolVana_Ac" := "AsitDoldurSeq_SirVana_Kapat";
   "AsitDoldurSeq_KuyuVana_Kapat" := "AsitDoldurSeq_SirVana_Kapat";
   "AsitDoldurSeq_IBCVana_Kapat" := "AsitDoldurSeq_SirVana_Kapat";
   "AsitDoldurSeq_AnaPompa_Run" := "AsitDoldurSeq_SirVana_Kapat" AND "02_Peripheral".IN.SirkulasyonVanasi.Closed AND "02_Peripheral".IN.DolumVanasi.Opened AND "02_Peripheral".IN.AsitTahliyeVanasi.Closed AND "02_Peripheral".IN.UcYolluVana.Opened AND "02_Peripheral".IN.KuyuTahVanasi.Closed AND "02_Peripheral".IN.IBC.AkisValfi.Closed AND "02_Peripheral".IN.AsitTanki.AltSeviyeSen AND "02_Peripheral".IN.AsitTanki.KapiSwitch AND "02_Peripheral".IN.YikamaTanki.KapiSwitch1 AND "02_Peripheral".IN.AsitTanki.AltSeviyeSen;
   IF "AsitDoldurSeq_SirVana_Kapat" AND ("02_Peripheral".IN.YikamaTanki.UstSeviyeSen OR "02_Peripheral".IN.YikamaTanki.CriticalSeviyeSen) THEN
       "01_System".State.AsitDolum := 2;
   END_IF;
END_REGION

REGION Network 3: İşlem bittikten sonra dolum vanasini kapat
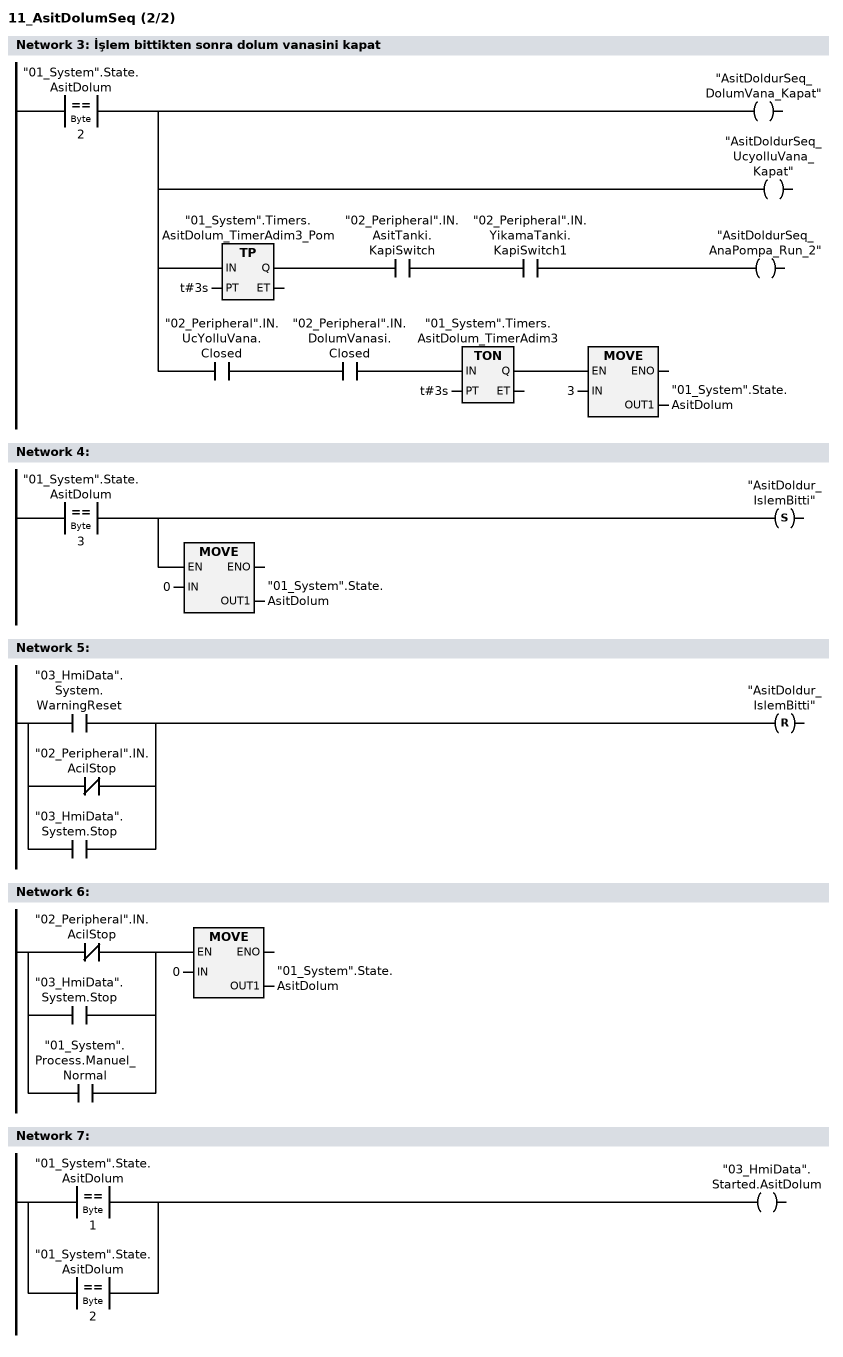
   "AsitDoldurSeq_DolumVana_Kapat" := "01_System".State.AsitDolum = 2;
   "AsitDoldurSeq_UcyolluVana_Kapat" := "AsitDoldurSeq_DolumVana_Kapat";
   "01_System".Timers.AsitDolum_TimerAdim3_Pom.TP(IN := "AsitDoldurSeq_DolumVana_Kapat", PT := t#3s);
   "AsitDoldurSeq_AnaPompa_Run_2" := "01_System".Timers.AsitDolum_TimerAdim3_Pom.Q AND "02_Peripheral".IN.AsitTanki.KapiSwitch AND "02_Peripheral".IN.YikamaTanki.KapiSwitch1;
   "01_System".Timers.AsitDolum_TimerAdim3.TON(IN := "AsitDoldurSeq_DolumVana_Kapat" AND "02_Peripheral".IN.UcYolluVana.Closed AND "02_Peripheral".IN.DolumVanasi.Closed,
                           PT := t#3s);
   IF "01_System".Timers.AsitDolum_TimerAdim3.Q THEN "01_System".State.AsitDolum := 3; END_IF;
END_REGION

REGION Network 4
   RUNG wire#powerrail
      { S7_Templates := "SrcType := Byte" } EQ_Contact(in1 := "01_System".State.AsitDolum, in2 := 3)
      wire#w1
      S_Coil( "AsitDoldur_IslemBitti" )
   END_RUNG
   RUNG wire#w1
      Move(in := 0, out1 => "01_System".State.AsitDolum)
   END_RUNG
   // the same network as SCL:
   IF "01_System".State.AsitDolum = 3 THEN
       "AsitDoldur_IslemBitti" := TRUE;
       "01_System".State.AsitDolum := 0;
   END_IF;
END_REGION

REGION Network 5
   RUNG wire#powerrail
      Contact( "03_HmiData".System.WarningReset )
      wire#w1
      R_Coil( "AsitDoldur_IslemBitti" )
   END_RUNG
   RUNG wire#powerrail
      I_Contact( "02_Peripheral".IN.AcilStop )
   END_RUNG wire#w1
   RUNG wire#powerrail
      Contact( "03_HmiData".System.Stop )
   END_RUNG wire#w1
   // the same network as SCL:
   IF "03_HmiData".System.WarningReset OR NOT "02_Peripheral".IN.AcilStop OR "03_HmiData".System.Stop THEN
       "AsitDoldur_IslemBitti" := FALSE;
   END_IF;
END_REGION

REGION Network 6
   RUNG wire#powerrail
      I_Contact( "02_Peripheral".IN.AcilStop )
      wire#w1
      Move(in := 0, out1 => "01_System".State.AsitDolum)
   END_RUNG
   RUNG wire#powerrail
      Contact( "03_HmiData".System.Stop )
   END_RUNG wire#w1
   RUNG wire#powerrail
      Contact( "01_System".Process.Manuel_Normal )
   END_RUNG wire#w1
   // the same network as SCL:
   IF NOT "02_Peripheral".IN.AcilStop OR "03_HmiData".System.Stop OR "01_System".Process.Manuel_Normal THEN
       "01_System".State.AsitDolum := 0;
   END_IF;
END_REGION

REGION Network 7
   RUNG wire#powerrail
      { S7_Templates := "SrcType := Byte" } EQ_Contact(in1 := "01_System".State.AsitDolum, in2 := 1)
      wire#w1
      Coil( "03_HmiData".Started.AsitDolum )
   END_RUNG
   RUNG wire#powerrail
      { S7_Templates := "SrcType := Byte" } EQ_Contact(in1 := "01_System".State.AsitDolum, in2 := 2)
   END_RUNG wire#w1
   // the same network as SCL:
   "03_HmiData".Started.AsitDolum := ("01_System".State.AsitDolum = 1) OR ("01_System".State.AsitDolum = 2);
END_REGION
END_FUNCTION

FUNCTION "13_AsitTahliyeSeq" : Void   // FC5, LAD
{ S7_Optimized_Access := 'TRUE' }
VERSION : 0.1
BEGIN

REGION Network 1
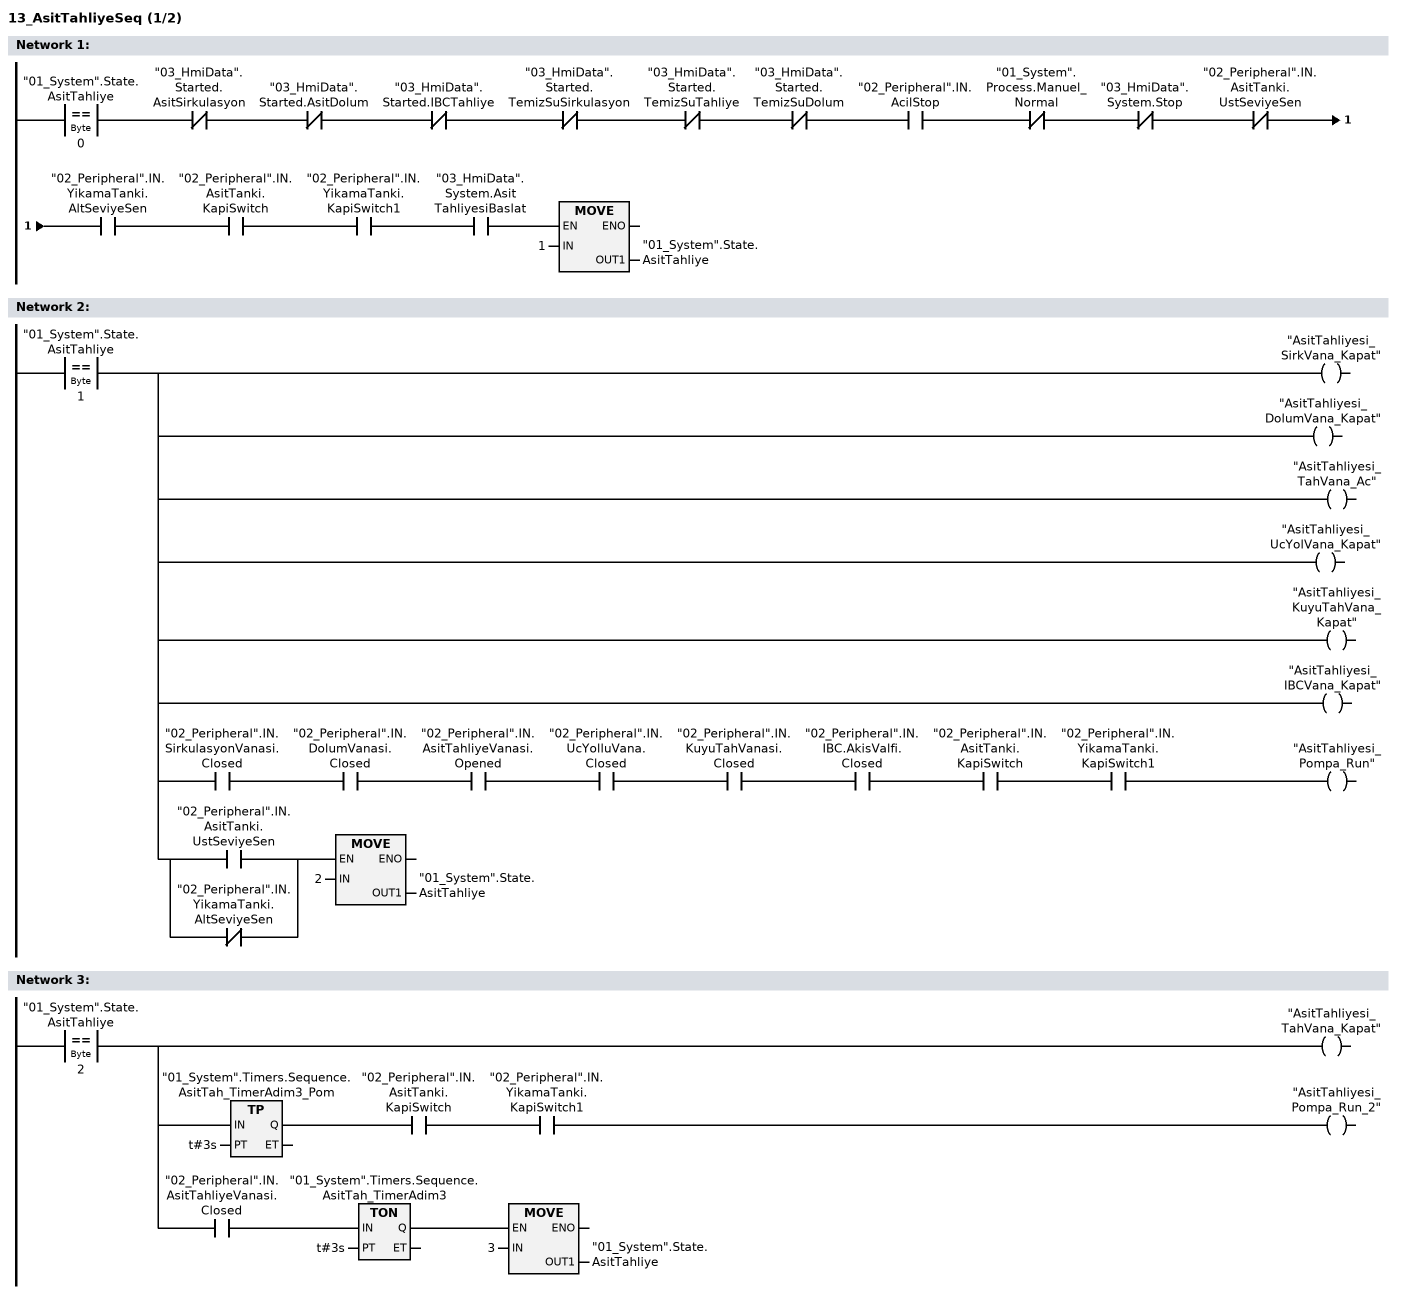
   RUNG wire#powerrail
      { S7_Templates := "SrcType := Byte" } EQ_Contact(in1 := "01_System".State.AsitTahliye, in2 := 0)
      I_Contact( "03_HmiData".Started.AsitSirkulasyon )
      I_Contact( "03_HmiData".Started.AsitDolum )
      I_Contact( "03_HmiData".Started.IBCTahliye )
      I_Contact( "03_HmiData".Started.TemizSuSirkulasyon )
      I_Contact( "03_HmiData".Started.TemizSuTahliye )
      I_Contact( "03_HmiData".Started.TemizSuDolum )
      Contact( "02_Peripheral".IN.AcilStop )
      I_Contact( "01_System".Process.Manuel_Normal )
      I_Contact( "03_HmiData".System.Stop )
      I_Contact( "02_Peripheral".IN.AsitTanki.UstSeviyeSen )
      Contact( "02_Peripheral".IN.YikamaTanki.AltSeviyeSen )
      Contact( "02_Peripheral".IN.AsitTanki.KapiSwitch )
      Contact( "02_Peripheral".IN.YikamaTanki.KapiSwitch1 )
      Contact( "03_HmiData".System.AsitTahliyesiBaslat )
      Move(in := 1, out1 => "01_System".State.AsitTahliye)
   END_RUNG
   // the same network as SCL:
   IF ("01_System".State.AsitTahliye = 0) AND NOT "03_HmiData".Started.AsitSirkulasyon AND NOT "03_HmiData".Started.AsitDolum AND NOT "03_HmiData".Started.IBCTahliye AND NOT "03_HmiData".Started.TemizSuSirkulasyon AND NOT "03_HmiData".Started.TemizSuTahliye AND NOT "03_HmiData".Started.TemizSuDolum AND "02_Peripheral".IN.AcilStop AND NOT "01_System".Process.Manuel_Normal AND NOT "03_HmiData".System.Stop AND NOT "02_Peripheral".IN.AsitTanki.UstSeviyeSen AND "02_Peripheral".IN.YikamaTanki.AltSeviyeSen AND "02_Peripheral".IN.AsitTanki.KapiSwitch AND "02_Peripheral".IN.YikamaTanki.KapiSwitch1 AND "03_HmiData".System.AsitTahliyesiBaslat THEN
       "01_System".State.AsitTahliye := 1;
   END_IF;
END_REGION

REGION Network 2
   RUNG wire#powerrail
      { S7_Templates := "SrcType := Byte" } EQ_Contact(in1 := "01_System".State.AsitTahliye, in2 := 1)
      wire#w1
      Coil( "AsitTahliyesi_SirkVana_Kapat" )
   END_RUNG
   RUNG wire#w1
      Coil( "AsitTahliyesi_DolumVana_Kapat" )
   END_RUNG
   RUNG wire#w1
      Coil( "AsitTahliyesi_TahVana_Ac" )
   END_RUNG
   RUNG wire#w1
      Coil( "AsitTahliyesi_UcYolVana_Kapat" )
   END_RUNG
   RUNG wire#w1
      Coil( "AsitTahliyesi_KuyuTahVana_Kapat" )
   END_RUNG
   RUNG wire#w1
      Coil( "AsitTahliyesi_IBCVana_Kapat" )
   END_RUNG
   RUNG wire#w1
      Contact( "02_Peripheral".IN.SirkulasyonVanasi.Closed )
      Contact( "02_Peripheral".IN.DolumVanasi.Closed )
      Contact( "02_Peripheral".IN.AsitTahliyeVanasi.Opened )
      Contact( "02_Peripheral".IN.UcYolluVana.Closed )
      Contact( "02_Peripheral".IN.KuyuTahVanasi.Closed )
      Contact( "02_Peripheral".IN.IBC.AkisValfi.Closed )
      Contact( "02_Peripheral".IN.AsitTanki.KapiSwitch )
      Contact( "02_Peripheral".IN.YikamaTanki.KapiSwitch1 )
      Coil( "AsitTahliyesi_Pompa_Run" )
   END_RUNG
   RUNG wire#w1
      Contact( "02_Peripheral".IN.AsitTanki.UstSeviyeSen )
      wire#w2
      Move(in := 2, out1 => "01_System".State.AsitTahliye)
   END_RUNG
   RUNG wire#w1
      I_Contact( "02_Peripheral".IN.YikamaTanki.AltSeviyeSen )
   END_RUNG wire#w2
   // the same network as SCL:
   "AsitTahliyesi_SirkVana_Kapat" := "01_System".State.AsitTahliye = 1;
   "AsitTahliyesi_DolumVana_Kapat" := "AsitTahliyesi_SirkVana_Kapat";
   "AsitTahliyesi_TahVana_Ac" := "AsitTahliyesi_SirkVana_Kapat";
   "AsitTahliyesi_UcYolVana_Kapat" := "AsitTahliyesi_SirkVana_Kapat";
   "AsitTahliyesi_KuyuTahVana_Kapat" := "AsitTahliyesi_SirkVana_Kapat";
   "AsitTahliyesi_IBCVana_Kapat" := "AsitTahliyesi_SirkVana_Kapat";
   "AsitTahliyesi_Pompa_Run" := "AsitTahliyesi_SirkVana_Kapat" AND "02_Peripheral".IN.SirkulasyonVanasi.Closed AND "02_Peripheral".IN.DolumVanasi.Closed AND "02_Peripheral".IN.AsitTahliyeVanasi.Opened AND "02_Peripheral".IN.UcYolluVana.Closed AND "02_Peripheral".IN.KuyuTahVanasi.Closed AND "02_Peripheral".IN.IBC.AkisValfi.Closed AND "02_Peripheral".IN.AsitTanki.KapiSwitch AND "02_Peripheral".IN.YikamaTanki.KapiSwitch1;
   IF "AsitTahliyesi_SirkVana_Kapat" AND ("02_Peripheral".IN.AsitTanki.UstSeviyeSen OR NOT "02_Peripheral".IN.YikamaTanki.AltSeviyeSen) THEN
       "01_System".State.AsitTahliye := 2;
   END_IF;
END_REGION

REGION Network 3
   "AsitTahliyesi_TahVana_Kapat" := "01_System".State.AsitTahliye = 2;
   "01_System".Timers.Sequence.AsitTah_TimerAdim3_Pom.TP(IN := "AsitTahliyesi_TahVana_Kapat", PT := t#3s);
   "AsitTahliyesi_Pompa_Run_2" := "01_System".Timers.Sequence.AsitTah_TimerAdim3_Pom.Q AND "02_Peripheral".IN.AsitTanki.KapiSwitch AND "02_Peripheral".IN.YikamaTanki.KapiSwitch1;
   "01_System".Timers.Sequence.AsitTah_TimerAdim3.TON(IN := "AsitTahliyesi_TahVana_Kapat" AND "02_Peripheral".IN.AsitTahliyeVanasi.Closed,
                           PT := t#3s);
   IF "01_System".Timers.Sequence.AsitTah_TimerAdim3.Q THEN "01_System".State.AsitTahliye := 3; END_IF;
END_REGION

REGION Network 4
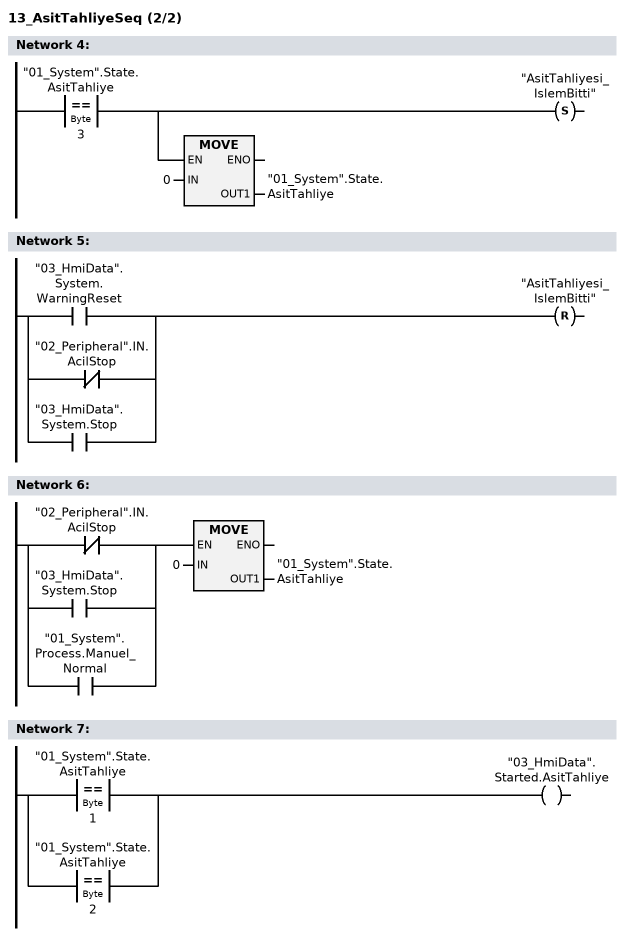
   RUNG wire#powerrail
      { S7_Templates := "SrcType := Byte" } EQ_Contact(in1 := "01_System".State.AsitTahliye, in2 := 3)
      wire#w1
      S_Coil( "AsitTahliyesi_IslemBitti" )
   END_RUNG
   RUNG wire#w1
      Move(in := 0, out1 => "01_System".State.AsitTahliye)
   END_RUNG
   // the same network as SCL:
   IF "01_System".State.AsitTahliye = 3 THEN
       "AsitTahliyesi_IslemBitti" := TRUE;
       "01_System".State.AsitTahliye := 0;
   END_IF;
END_REGION

REGION Network 5
   RUNG wire#powerrail
      Contact( "03_HmiData".System.WarningReset )
      wire#w1
      R_Coil( "AsitTahliyesi_IslemBitti" )
   END_RUNG
   RUNG wire#powerrail
      I_Contact( "02_Peripheral".IN.AcilStop )
   END_RUNG wire#w1
   RUNG wire#powerrail
      Contact( "03_HmiData".System.Stop )
   END_RUNG wire#w1
   // the same network as SCL:
   IF "03_HmiData".System.WarningReset OR NOT "02_Peripheral".IN.AcilStop OR "03_HmiData".System.Stop THEN
       "AsitTahliyesi_IslemBitti" := FALSE;
   END_IF;
END_REGION

REGION Network 6
   RUNG wire#powerrail
      I_Contact( "02_Peripheral".IN.AcilStop )
      wire#w1
      Move(in := 0, out1 => "01_System".State.AsitTahliye)
   END_RUNG
   RUNG wire#powerrail
      Contact( "03_HmiData".System.Stop )
   END_RUNG wire#w1
   RUNG wire#powerrail
      Contact( "01_System".Process.Manuel_Normal )
   END_RUNG wire#w1
   // the same network as SCL:
   IF NOT "02_Peripheral".IN.AcilStop OR "03_HmiData".System.Stop OR "01_System".Process.Manuel_Normal THEN
       "01_System".State.AsitTahliye := 0;
   END_IF;
END_REGION

REGION Network 7
   RUNG wire#powerrail
      { S7_Templates := "SrcType := Byte" } EQ_Contact(in1 := "01_System".State.AsitTahliye, in2 := 1)
      wire#w1
      Coil( "03_HmiData".Started.AsitTahliye )
   END_RUNG
   RUNG wire#powerrail
      { S7_Templates := "SrcType := Byte" } EQ_Contact(in1 := "01_System".State.AsitTahliye, in2 := 2)
   END_RUNG wire#w1
   // the same network as SCL:
   "03_HmiData".Started.AsitTahliye := ("01_System".State.AsitTahliye = 1) OR ("01_System".State.AsitTahliye = 2);
END_REGION
END_FUNCTION

FUNCTION "15_SuSirkulasyonSeq" : Void   // FC6, LAD
{ S7_Optimized_Access := 'TRUE' }
VERSION : 0.1
   VAR_TEMP   // added for the SCL form of the ladder/FBD networks
      _w1 : Bool;
   END_VAR
BEGIN

REGION Network 1
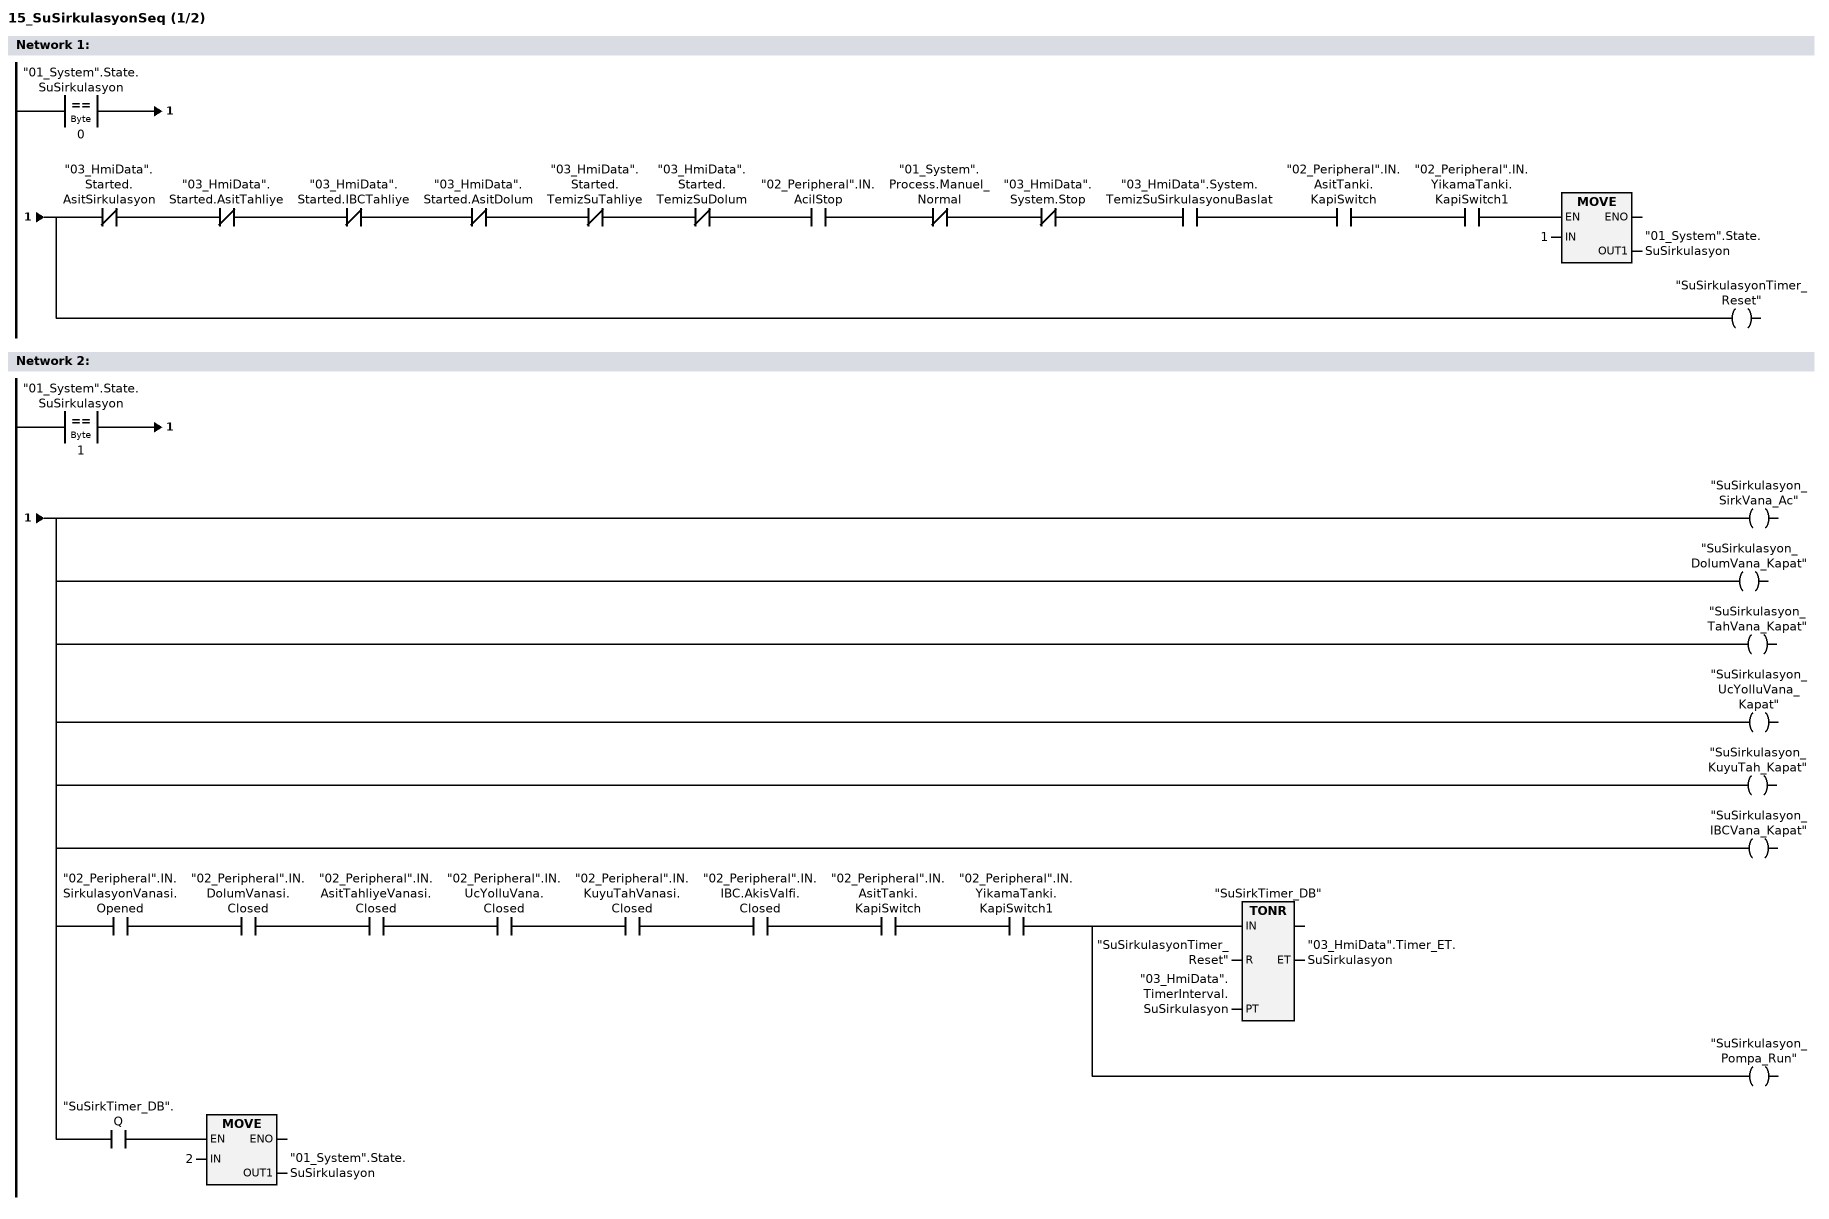
   RUNG wire#powerrail
      { S7_Templates := "SrcType := Byte" } EQ_Contact(in1 := "01_System".State.SuSirkulasyon, in2 := 0)
      wire#w1
      I_Contact( "03_HmiData".Started.AsitSirkulasyon )
      I_Contact( "03_HmiData".Started.AsitTahliye )
      I_Contact( "03_HmiData".Started.IBCTahliye )
      I_Contact( "03_HmiData".Started.AsitDolum )
      I_Contact( "03_HmiData".Started.TemizSuTahliye )
      I_Contact( "03_HmiData".Started.TemizSuDolum )
      Contact( "02_Peripheral".IN.AcilStop )
      I_Contact( "01_System".Process.Manuel_Normal )
      I_Contact( "03_HmiData".System.Stop )
      Contact( "03_HmiData".System.TemizSuSirkulasyonuBaslat )
      Contact( "02_Peripheral".IN.AsitTanki.KapiSwitch )
      Contact( "02_Peripheral".IN.YikamaTanki.KapiSwitch1 )
      Move(in := 1, out1 => "01_System".State.SuSirkulasyon)
   END_RUNG
   RUNG wire#w1
      Coil( "SuSirkulasyonTimer_Reset" )
   END_RUNG
   // the same network as SCL:
   #_w1 := "01_System".State.SuSirkulasyon = 0;
   IF #_w1 AND NOT "03_HmiData".Started.AsitSirkulasyon AND NOT "03_HmiData".Started.AsitTahliye AND NOT "03_HmiData".Started.IBCTahliye AND NOT "03_HmiData".Started.AsitDolum AND NOT "03_HmiData".Started.TemizSuTahliye AND NOT "03_HmiData".Started.TemizSuDolum AND "02_Peripheral".IN.AcilStop AND NOT "01_System".Process.Manuel_Normal AND NOT "03_HmiData".System.Stop AND "03_HmiData".System.TemizSuSirkulasyonuBaslat AND "02_Peripheral".IN.AsitTanki.KapiSwitch AND "02_Peripheral".IN.YikamaTanki.KapiSwitch1 THEN
       "01_System".State.SuSirkulasyon := 1;
   END_IF;
   "SuSirkulasyonTimer_Reset" := #_w1;
END_REGION

REGION Network 2
   "SuSirkulasyon_SirkVana_Ac" := "01_System".State.SuSirkulasyon = 1;
   "SuSirkulasyon_DolumVana_Kapat" := "SuSirkulasyon_SirkVana_Ac";
   "SuSirkulasyon_TahVana_Kapat" := "SuSirkulasyon_SirkVana_Ac";
   "SuSirkulasyon_UcYolluVana_Kapat" := "SuSirkulasyon_SirkVana_Ac";
   "SuSirkulasyon_KuyuTah_Kapat" := "SuSirkulasyon_SirkVana_Ac";
   "SuSirkulasyon_IBCVana_Kapat" := "SuSirkulasyon_SirkVana_Ac";
   #_w1 := "SuSirkulasyon_SirkVana_Ac" AND "02_Peripheral".IN.SirkulasyonVanasi.Opened AND "02_Peripheral".IN.DolumVanasi.Closed AND "02_Peripheral".IN.AsitTahliyeVanasi.Closed AND "02_Peripheral".IN.UcYolluVana.Closed AND "02_Peripheral".IN.KuyuTahVanasi.Closed AND "02_Peripheral".IN.IBC.AkisValfi.Closed AND "02_Peripheral".IN.AsitTanki.KapiSwitch AND "02_Peripheral".IN.YikamaTanki.KapiSwitch1;
   "SuSirkTimer_DB".TONR(IN := #_w1,
                         R := "SuSirkulasyonTimer_Reset",
                         PT := "03_HmiData".TimerInterval.SuSirkulasyon,
                         ET => "03_HmiData".Timer_ET.SuSirkulasyon);
   "SuSirkulasyon_Pompa_Run" := #_w1;
   IF "SuSirkulasyon_SirkVana_Ac" AND "SuSirkTimer_DB".Q THEN "01_System".State.SuSirkulasyon := 2; END_IF;
END_REGION

REGION Network 3
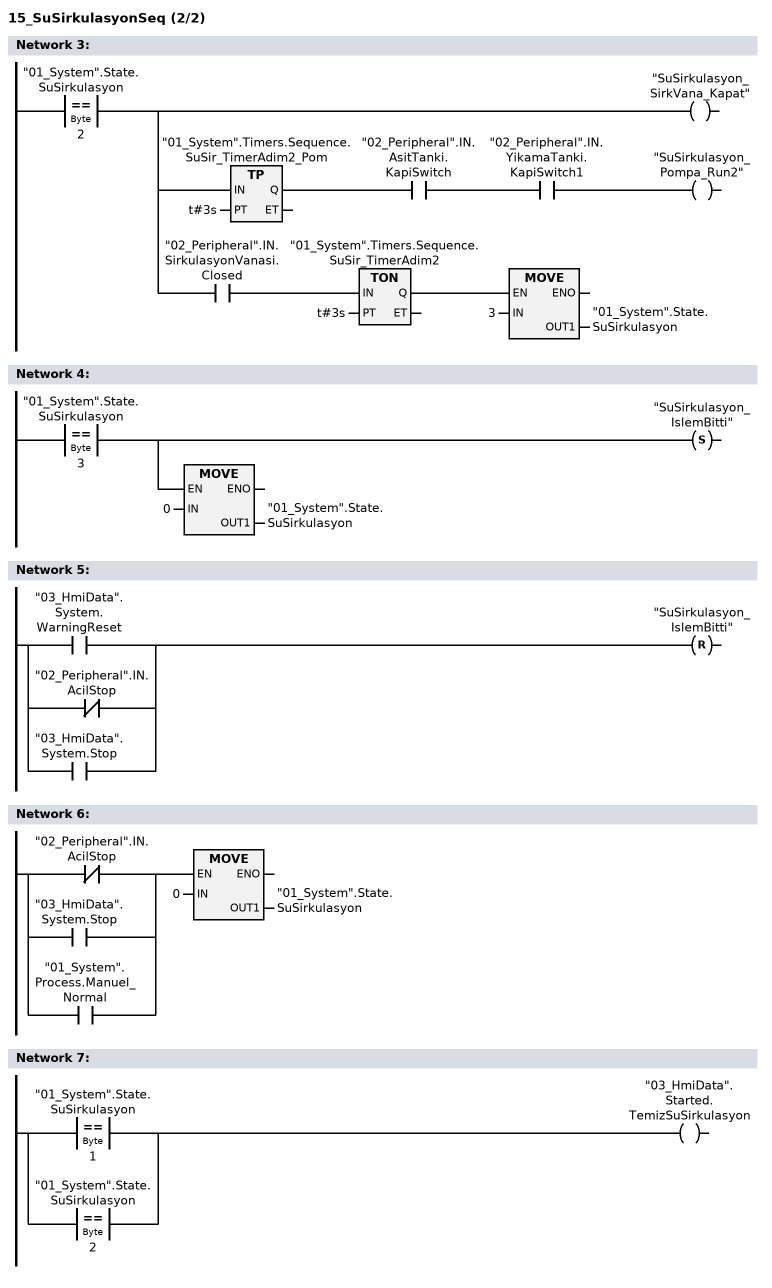
   "SuSirkulasyon_SirkVana_Kapat" := "01_System".State.SuSirkulasyon = 2;
   "01_System".Timers.Sequence.SuSir_TimerAdim2_Pom.TP(IN := "SuSirkulasyon_SirkVana_Kapat", PT := t#3s);
   "SuSirkulasyon_Pompa_Run2" := "01_System".Timers.Sequence.SuSir_TimerAdim2_Pom.Q AND "02_Peripheral".IN.AsitTanki.KapiSwitch AND "02_Peripheral".IN.YikamaTanki.KapiSwitch1;
   "01_System".Timers.Sequence.SuSir_TimerAdim2.TON(IN := "SuSirkulasyon_SirkVana_Kapat" AND "02_Peripheral".IN.SirkulasyonVanasi.Closed,
                           PT := t#3s);
   IF "01_System".Timers.Sequence.SuSir_TimerAdim2.Q THEN "01_System".State.SuSirkulasyon := 3; END_IF;
END_REGION

REGION Network 4
   RUNG wire#powerrail
      { S7_Templates := "SrcType := Byte" } EQ_Contact(in1 := "01_System".State.SuSirkulasyon, in2 := 3)
      wire#w1
      S_Coil( "SuSirkulasyon_IslemBitti" )
   END_RUNG
   RUNG wire#w1
      Move(in := 0, out1 => "01_System".State.SuSirkulasyon)
   END_RUNG
   // the same network as SCL:
   IF "01_System".State.SuSirkulasyon = 3 THEN
       "SuSirkulasyon_IslemBitti" := TRUE;
       "01_System".State.SuSirkulasyon := 0;
   END_IF;
END_REGION

REGION Network 5
   RUNG wire#powerrail
      Contact( "03_HmiData".System.WarningReset )
      wire#w1
      R_Coil( "SuSirkulasyon_IslemBitti" )
   END_RUNG
   RUNG wire#powerrail
      I_Contact( "02_Peripheral".IN.AcilStop )
   END_RUNG wire#w1
   RUNG wire#powerrail
      Contact( "03_HmiData".System.Stop )
   END_RUNG wire#w1
   // the same network as SCL:
   IF "03_HmiData".System.WarningReset OR NOT "02_Peripheral".IN.AcilStop OR "03_HmiData".System.Stop THEN
       "SuSirkulasyon_IslemBitti" := FALSE;
   END_IF;
END_REGION

REGION Network 6
   RUNG wire#powerrail
      I_Contact( "02_Peripheral".IN.AcilStop )
      wire#w1
      Move(in := 0, out1 => "01_System".State.SuSirkulasyon)
   END_RUNG
   RUNG wire#powerrail
      Contact( "03_HmiData".System.Stop )
   END_RUNG wire#w1
   RUNG wire#powerrail
      Contact( "01_System".Process.Manuel_Normal )
   END_RUNG wire#w1
   // the same network as SCL:
   IF NOT "02_Peripheral".IN.AcilStop OR "03_HmiData".System.Stop OR "01_System".Process.Manuel_Normal THEN
       "01_System".State.SuSirkulasyon := 0;
   END_IF;
END_REGION

REGION Network 7
   RUNG wire#powerrail
      { S7_Templates := "SrcType := Byte" } EQ_Contact(in1 := "01_System".State.SuSirkulasyon, in2 := 1)
      wire#w1
      Coil( "03_HmiData".Started.TemizSuSirkulasyon )
   END_RUNG
   RUNG wire#powerrail
      { S7_Templates := "SrcType := Byte" } EQ_Contact(in1 := "01_System".State.SuSirkulasyon, in2 := 2)
   END_RUNG wire#w1
   // the same network as SCL:
   "03_HmiData".Started.TemizSuSirkulasyon := ("01_System".State.SuSirkulasyon = 1) OR ("01_System".State.SuSirkulasyon = 2);
END_REGION
END_FUNCTION

FUNCTION "16_SuTahliyeSeq" : Void   // FC7, LAD
{ S7_Optimized_Access := 'TRUE' }
VERSION : 0.1
BEGIN

REGION Network 1
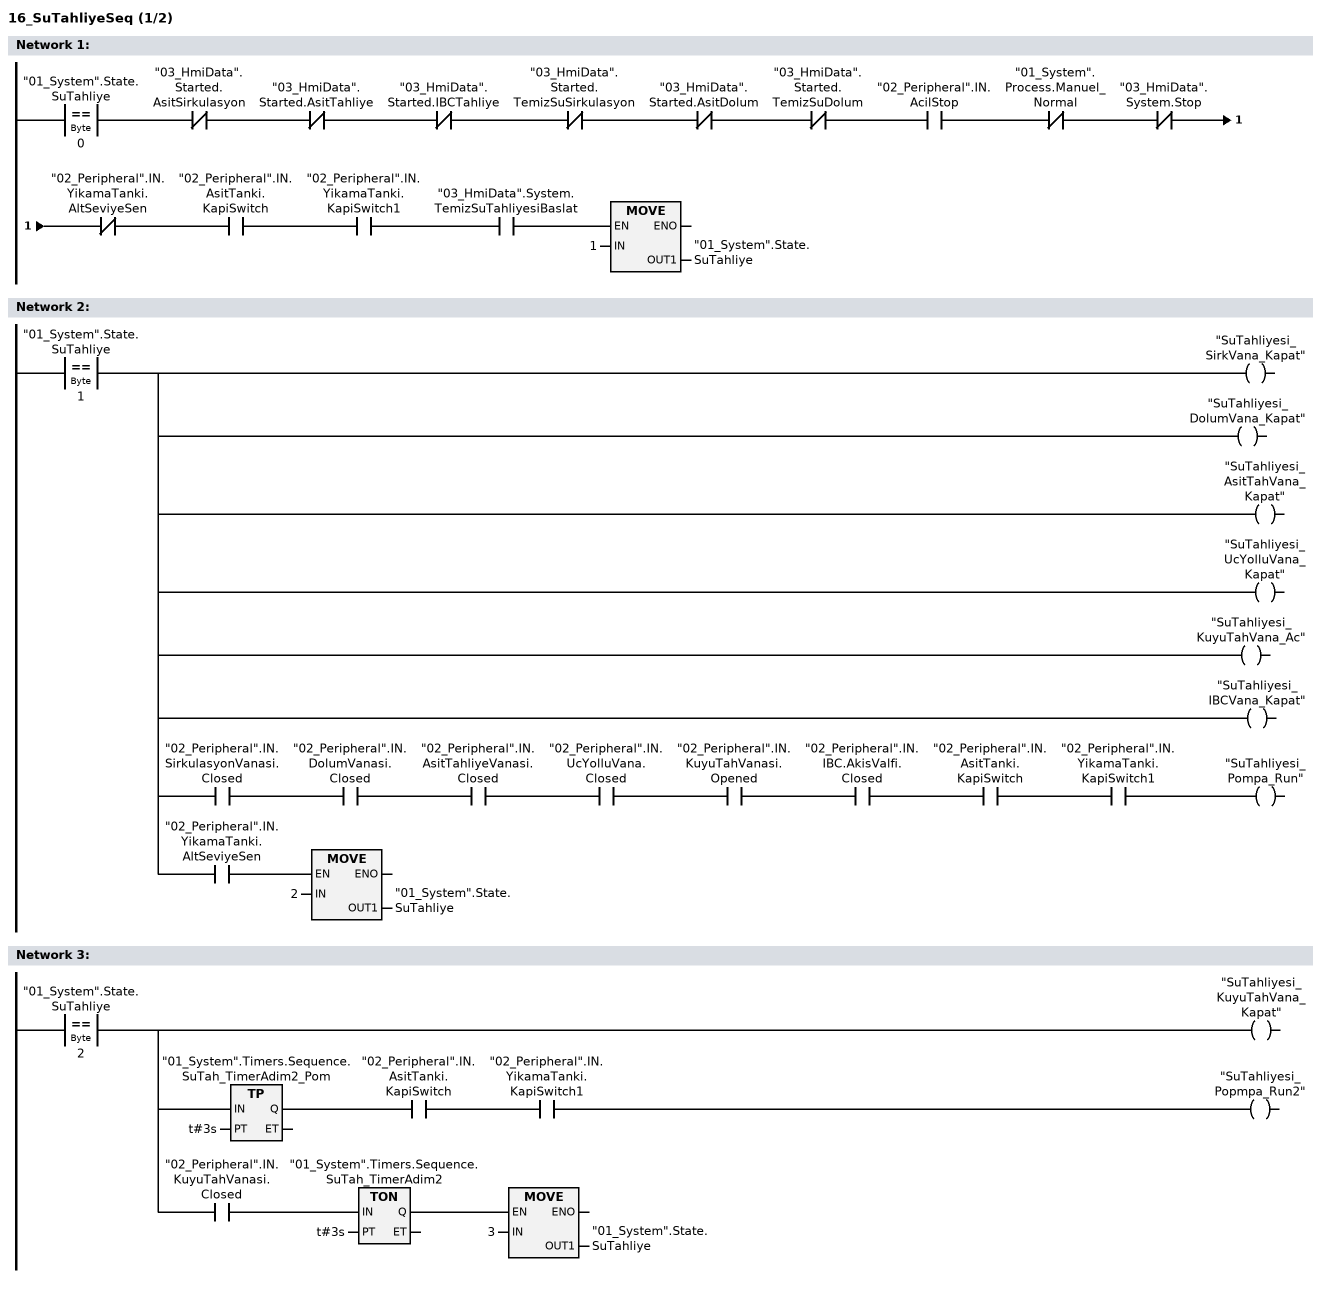
   RUNG wire#powerrail
      { S7_Templates := "SrcType := Byte" } EQ_Contact(in1 := "01_System".State.SuTahliye, in2 := 0)
      I_Contact( "03_HmiData".Started.AsitSirkulasyon )
      I_Contact( "03_HmiData".Started.AsitTahliye )
      I_Contact( "03_HmiData".Started.IBCTahliye )
      I_Contact( "03_HmiData".Started.TemizSuSirkulasyon )
      I_Contact( "03_HmiData".Started.AsitDolum )
      I_Contact( "03_HmiData".Started.TemizSuDolum )
      Contact( "02_Peripheral".IN.AcilStop )
      I_Contact( "01_System".Process.Manuel_Normal )
      I_Contact( "03_HmiData".System.Stop )
      I_Contact( "02_Peripheral".IN.YikamaTanki.AltSeviyeSen )
      Contact( "02_Peripheral".IN.AsitTanki.KapiSwitch )
      Contact( "02_Peripheral".IN.YikamaTanki.KapiSwitch1 )
      Contact( "03_HmiData".System.TemizSuTahliyesiBaslat )
      Move(in := 1, out1 => "01_System".State.SuTahliye)
   END_RUNG
   // the same network as SCL:
   IF ("01_System".State.SuTahliye = 0) AND NOT "03_HmiData".Started.AsitSirkulasyon AND NOT "03_HmiData".Started.AsitTahliye AND NOT "03_HmiData".Started.IBCTahliye AND NOT "03_HmiData".Started.TemizSuSirkulasyon AND NOT "03_HmiData".Started.AsitDolum AND NOT "03_HmiData".Started.TemizSuDolum AND "02_Peripheral".IN.AcilStop AND NOT "01_System".Process.Manuel_Normal AND NOT "03_HmiData".System.Stop AND NOT "02_Peripheral".IN.YikamaTanki.AltSeviyeSen AND "02_Peripheral".IN.AsitTanki.KapiSwitch AND "02_Peripheral".IN.YikamaTanki.KapiSwitch1 AND "03_HmiData".System.TemizSuTahliyesiBaslat THEN
       "01_System".State.SuTahliye := 1;
   END_IF;
END_REGION

REGION Network 2
   RUNG wire#powerrail
      { S7_Templates := "SrcType := Byte" } EQ_Contact(in1 := "01_System".State.SuTahliye, in2 := 1)
      wire#w1
      Coil( "SuTahliyesi_SirkVana_Kapat" )
   END_RUNG
   RUNG wire#w1
      Coil( "SuTahliyesi_DolumVana_Kapat" )
   END_RUNG
   RUNG wire#w1
      Coil( "SuTahliyesi_AsitTahVana_Kapat" )
   END_RUNG
   RUNG wire#w1
      Coil( "SuTahliyesi_UcYolluVana_Kapat" )
   END_RUNG
   RUNG wire#w1
      Coil( "SuTahliyesi_KuyuTahVana_Ac" )
   END_RUNG
   RUNG wire#w1
      Coil( "SuTahliyesi_IBCVana_Kapat" )
   END_RUNG
   RUNG wire#w1
      Contact( "02_Peripheral".IN.SirkulasyonVanasi.Closed )
      Contact( "02_Peripheral".IN.DolumVanasi.Closed )
      Contact( "02_Peripheral".IN.AsitTahliyeVanasi.Closed )
      Contact( "02_Peripheral".IN.UcYolluVana.Closed )
      Contact( "02_Peripheral".IN.KuyuTahVanasi.Opened )
      Contact( "02_Peripheral".IN.IBC.AkisValfi.Closed )
      Contact( "02_Peripheral".IN.AsitTanki.KapiSwitch )
      Contact( "02_Peripheral".IN.YikamaTanki.KapiSwitch1 )
      Coil( "SuTahliyesi_Pompa_Run" )
   END_RUNG
   RUNG wire#w1
      Contact( "02_Peripheral".IN.YikamaTanki.AltSeviyeSen )
      Move(in := 2, out1 => "01_System".State.SuTahliye)
   END_RUNG
   // the same network as SCL:
   "SuTahliyesi_SirkVana_Kapat" := "01_System".State.SuTahliye = 1;
   "SuTahliyesi_DolumVana_Kapat" := "SuTahliyesi_SirkVana_Kapat";
   "SuTahliyesi_AsitTahVana_Kapat" := "SuTahliyesi_SirkVana_Kapat";
   "SuTahliyesi_UcYolluVana_Kapat" := "SuTahliyesi_SirkVana_Kapat";
   "SuTahliyesi_KuyuTahVana_Ac" := "SuTahliyesi_SirkVana_Kapat";
   "SuTahliyesi_IBCVana_Kapat" := "SuTahliyesi_SirkVana_Kapat";
   "SuTahliyesi_Pompa_Run" := "SuTahliyesi_SirkVana_Kapat" AND "02_Peripheral".IN.SirkulasyonVanasi.Closed AND "02_Peripheral".IN.DolumVanasi.Closed AND "02_Peripheral".IN.AsitTahliyeVanasi.Closed AND "02_Peripheral".IN.UcYolluVana.Closed AND "02_Peripheral".IN.KuyuTahVanasi.Opened AND "02_Peripheral".IN.IBC.AkisValfi.Closed AND "02_Peripheral".IN.AsitTanki.KapiSwitch AND "02_Peripheral".IN.YikamaTanki.KapiSwitch1;
   IF "SuTahliyesi_SirkVana_Kapat" AND "02_Peripheral".IN.YikamaTanki.AltSeviyeSen THEN
       "01_System".State.SuTahliye := 2;
   END_IF;
END_REGION

REGION Network 3
   "SuTahliyesi_KuyuTahVana_Kapat" := "01_System".State.SuTahliye = 2;
   "01_System".Timers.Sequence.SuTah_TimerAdim2_Pom.TP(IN := "SuTahliyesi_KuyuTahVana_Kapat", PT := t#3s);
   "SuTahliyesi_Popmpa_Run2" := "01_System".Timers.Sequence.SuTah_TimerAdim2_Pom.Q AND "02_Peripheral".IN.AsitTanki.KapiSwitch AND "02_Peripheral".IN.YikamaTanki.KapiSwitch1;
   "01_System".Timers.Sequence.SuTah_TimerAdim2.TON(IN := "SuTahliyesi_KuyuTahVana_Kapat" AND "02_Peripheral".IN.KuyuTahVanasi.Closed,
                           PT := t#3s);
   IF "01_System".Timers.Sequence.SuTah_TimerAdim2.Q THEN "01_System".State.SuTahliye := 3; END_IF;
END_REGION

REGION Network 4
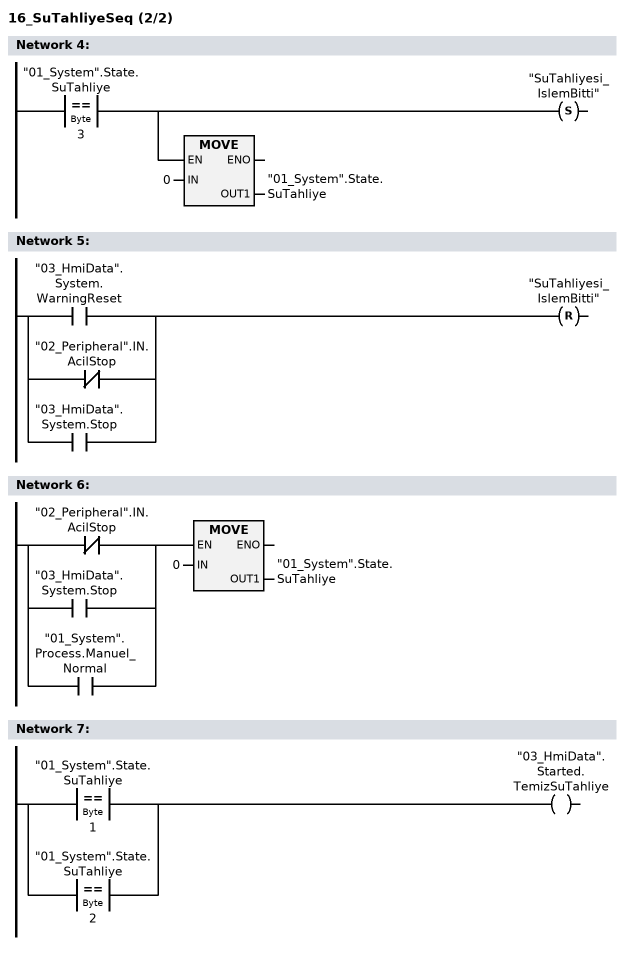
   RUNG wire#powerrail
      { S7_Templates := "SrcType := Byte" } EQ_Contact(in1 := "01_System".State.SuTahliye, in2 := 3)
      wire#w1
      S_Coil( "SuTahliyesi_IslemBitti" )
   END_RUNG
   RUNG wire#w1
      Move(in := 0, out1 => "01_System".State.SuTahliye)
   END_RUNG
   // the same network as SCL:
   IF "01_System".State.SuTahliye = 3 THEN
       "SuTahliyesi_IslemBitti" := TRUE;
       "01_System".State.SuTahliye := 0;
   END_IF;
END_REGION

REGION Network 5
   RUNG wire#powerrail
      Contact( "03_HmiData".System.WarningReset )
      wire#w1
      R_Coil( "SuTahliyesi_IslemBitti" )
   END_RUNG
   RUNG wire#powerrail
      I_Contact( "02_Peripheral".IN.AcilStop )
   END_RUNG wire#w1
   RUNG wire#powerrail
      Contact( "03_HmiData".System.Stop )
   END_RUNG wire#w1
   // the same network as SCL:
   IF "03_HmiData".System.WarningReset OR NOT "02_Peripheral".IN.AcilStop OR "03_HmiData".System.Stop THEN
       "SuTahliyesi_IslemBitti" := FALSE;
   END_IF;
END_REGION

REGION Network 6
   RUNG wire#powerrail
      I_Contact( "02_Peripheral".IN.AcilStop )
      wire#w1
      Move(in := 0, out1 => "01_System".State.SuTahliye)
   END_RUNG
   RUNG wire#powerrail
      Contact( "03_HmiData".System.Stop )
   END_RUNG wire#w1
   RUNG wire#powerrail
      Contact( "01_System".Process.Manuel_Normal )
   END_RUNG wire#w1
   // the same network as SCL:
   IF NOT "02_Peripheral".IN.AcilStop OR "03_HmiData".System.Stop OR "01_System".Process.Manuel_Normal THEN
       "01_System".State.SuTahliye := 0;
   END_IF;
END_REGION

REGION Network 7
   RUNG wire#powerrail
      { S7_Templates := "SrcType := Byte" } EQ_Contact(in1 := "01_System".State.SuTahliye, in2 := 1)
      wire#w1
      Coil( "03_HmiData".Started.TemizSuTahliye )
   END_RUNG
   RUNG wire#powerrail
      { S7_Templates := "SrcType := Byte" } EQ_Contact(in1 := "01_System".State.SuTahliye, in2 := 2)
   END_RUNG wire#w1
   // the same network as SCL:
   "03_HmiData".Started.TemizSuTahliye := ("01_System".State.SuTahliye = 1) OR ("01_System".State.SuTahliye = 2);
END_REGION
END_FUNCTION

FUNCTION "17_IBCTahliyeSeq" : Void   // FC8, LAD
{ S7_Optimized_Access := 'TRUE' }
VERSION : 0.1
BEGIN

REGION Network 1
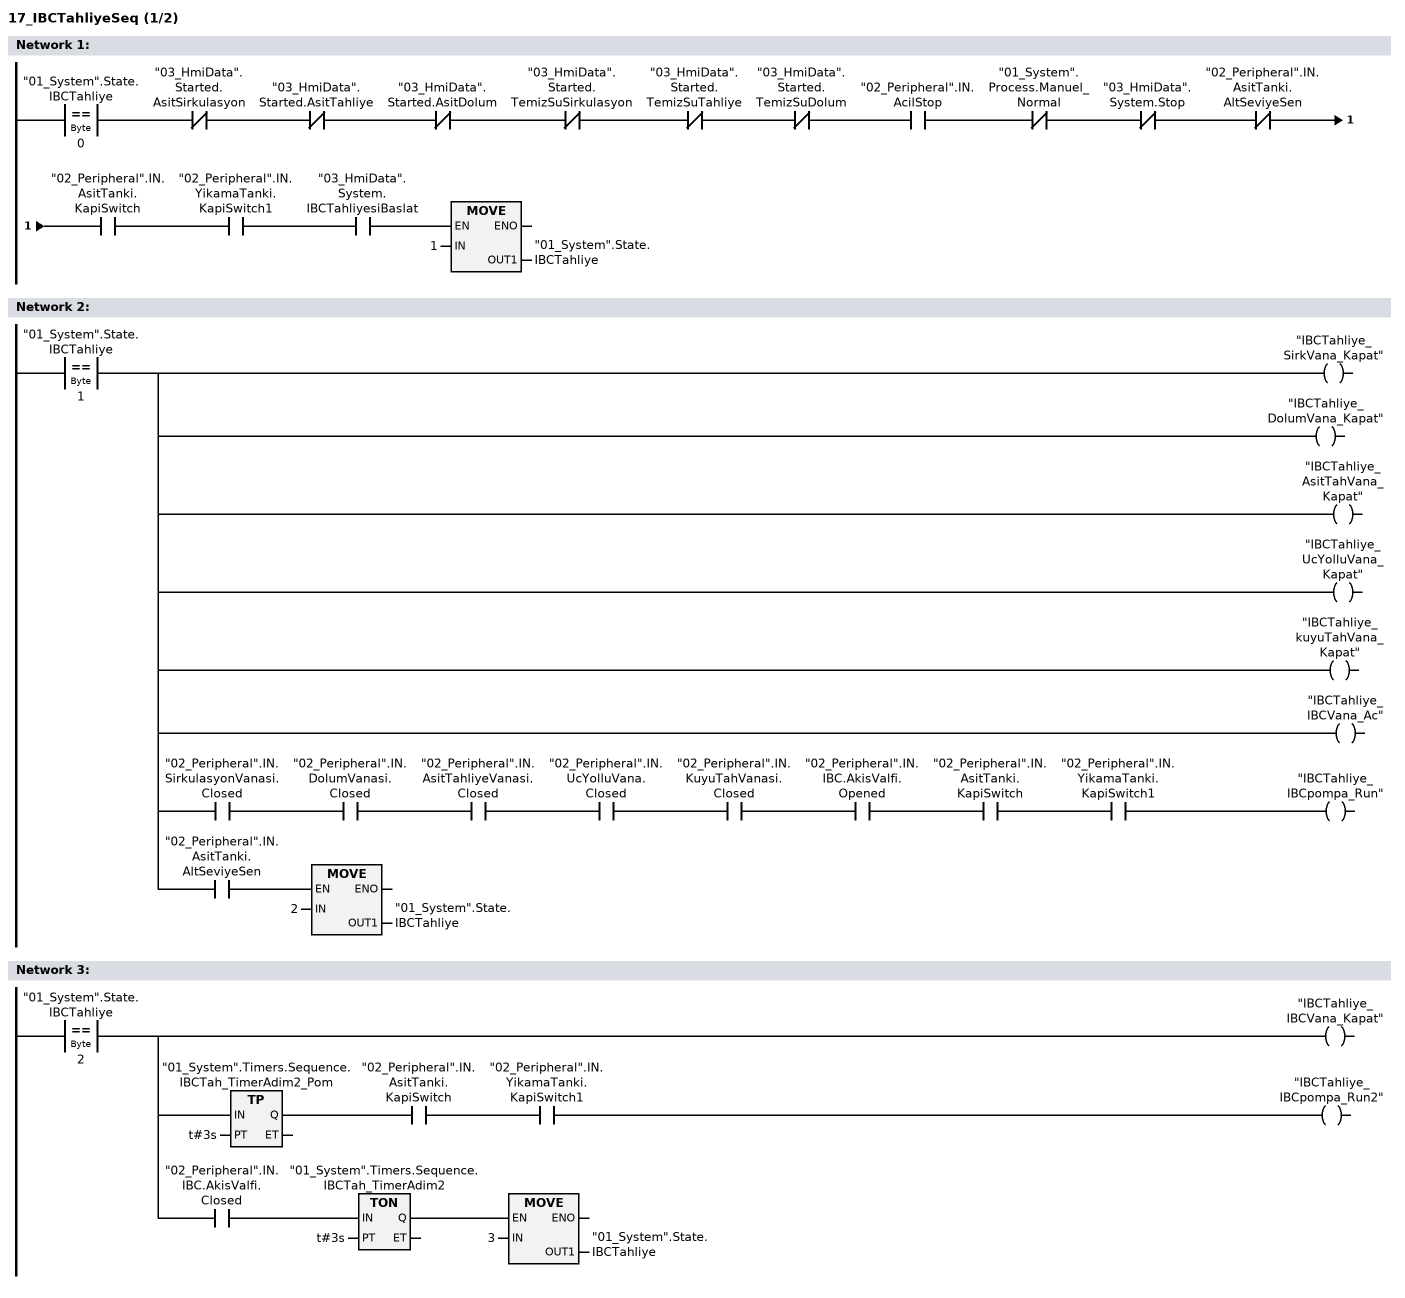
   RUNG wire#powerrail
      { S7_Templates := "SrcType := Byte" } EQ_Contact(in1 := "01_System".State.IBCTahliye, in2 := 0)
      I_Contact( "03_HmiData".Started.AsitSirkulasyon )
      I_Contact( "03_HmiData".Started.AsitTahliye )
      I_Contact( "03_HmiData".Started.AsitDolum )
      I_Contact( "03_HmiData".Started.TemizSuSirkulasyon )
      I_Contact( "03_HmiData".Started.TemizSuTahliye )
      I_Contact( "03_HmiData".Started.TemizSuDolum )
      Contact( "02_Peripheral".IN.AcilStop )
      I_Contact( "01_System".Process.Manuel_Normal )
      I_Contact( "03_HmiData".System.Stop )
      I_Contact( "02_Peripheral".IN.AsitTanki.AltSeviyeSen )
      Contact( "02_Peripheral".IN.AsitTanki.KapiSwitch )
      Contact( "02_Peripheral".IN.YikamaTanki.KapiSwitch1 )
      Contact( "03_HmiData".System.IBCTahliyesiBaslat )
      Move(in := 1, out1 => "01_System".State.IBCTahliye)
   END_RUNG
   // the same network as SCL:
   IF ("01_System".State.IBCTahliye = 0) AND NOT "03_HmiData".Started.AsitSirkulasyon AND NOT "03_HmiData".Started.AsitTahliye AND NOT "03_HmiData".Started.AsitDolum AND NOT "03_HmiData".Started.TemizSuSirkulasyon AND NOT "03_HmiData".Started.TemizSuTahliye AND NOT "03_HmiData".Started.TemizSuDolum AND "02_Peripheral".IN.AcilStop AND NOT "01_System".Process.Manuel_Normal AND NOT "03_HmiData".System.Stop AND NOT "02_Peripheral".IN.AsitTanki.AltSeviyeSen AND "02_Peripheral".IN.AsitTanki.KapiSwitch AND "02_Peripheral".IN.YikamaTanki.KapiSwitch1 AND "03_HmiData".System.IBCTahliyesiBaslat THEN
       "01_System".State.IBCTahliye := 1;
   END_IF;
END_REGION

REGION Network 2
   RUNG wire#powerrail
      { S7_Templates := "SrcType := Byte" } EQ_Contact(in1 := "01_System".State.IBCTahliye, in2 := 1)
      wire#w1
      Coil( "IBCTahliye_SirkVana_Kapat" )
   END_RUNG
   RUNG wire#w1
      Coil( "IBCTahliye_DolumVana_Kapat" )
   END_RUNG
   RUNG wire#w1
      Coil( "IBCTahliye_AsitTahVana_Kapat" )
   END_RUNG
   RUNG wire#w1
      Coil( "IBCTahliye_UcYolluVana_Kapat" )
   END_RUNG
   RUNG wire#w1
      Coil( "IBCTahliye_kuyuTahVana_Kapat" )
   END_RUNG
   RUNG wire#w1
      Coil( "IBCTahliye_IBCVana_Ac" )
   END_RUNG
   RUNG wire#w1
      Contact( "02_Peripheral".IN.SirkulasyonVanasi.Closed )
      Contact( "02_Peripheral".IN.DolumVanasi.Closed )
      Contact( "02_Peripheral".IN.AsitTahliyeVanasi.Closed )
      Contact( "02_Peripheral".IN.UcYolluVana.Closed )
      Contact( "02_Peripheral".IN.KuyuTahVanasi.Closed )
      Contact( "02_Peripheral".IN.IBC.AkisValfi.Opened )
      Contact( "02_Peripheral".IN.AsitTanki.KapiSwitch )
      Contact( "02_Peripheral".IN.YikamaTanki.KapiSwitch1 )
      Coil( "IBCTahliye_IBCpompa_Run" )
   END_RUNG
   RUNG wire#w1
      Contact( "02_Peripheral".IN.AsitTanki.AltSeviyeSen )
      Move(in := 2, out1 => "01_System".State.IBCTahliye)
   END_RUNG
   // the same network as SCL:
   "IBCTahliye_SirkVana_Kapat" := "01_System".State.IBCTahliye = 1;
   "IBCTahliye_DolumVana_Kapat" := "IBCTahliye_SirkVana_Kapat";
   "IBCTahliye_AsitTahVana_Kapat" := "IBCTahliye_SirkVana_Kapat";
   "IBCTahliye_UcYolluVana_Kapat" := "IBCTahliye_SirkVana_Kapat";
   "IBCTahliye_kuyuTahVana_Kapat" := "IBCTahliye_SirkVana_Kapat";
   "IBCTahliye_IBCVana_Ac" := "IBCTahliye_SirkVana_Kapat";
   "IBCTahliye_IBCpompa_Run" := "IBCTahliye_SirkVana_Kapat" AND "02_Peripheral".IN.SirkulasyonVanasi.Closed AND "02_Peripheral".IN.DolumVanasi.Closed AND "02_Peripheral".IN.AsitTahliyeVanasi.Closed AND "02_Peripheral".IN.UcYolluVana.Closed AND "02_Peripheral".IN.KuyuTahVanasi.Closed AND "02_Peripheral".IN.IBC.AkisValfi.Opened AND "02_Peripheral".IN.AsitTanki.KapiSwitch AND "02_Peripheral".IN.YikamaTanki.KapiSwitch1;
   IF "IBCTahliye_SirkVana_Kapat" AND "02_Peripheral".IN.AsitTanki.AltSeviyeSen THEN
       "01_System".State.IBCTahliye := 2;
   END_IF;
END_REGION

REGION Network 3
   "IBCTahliye_IBCVana_Kapat" := "01_System".State.IBCTahliye = 2;
   "01_System".Timers.Sequence.IBCTah_TimerAdim2_Pom.TP(IN := "IBCTahliye_IBCVana_Kapat", PT := t#3s);
   "IBCTahliye_IBCpompa_Run2" := "01_System".Timers.Sequence.IBCTah_TimerAdim2_Pom.Q AND "02_Peripheral".IN.AsitTanki.KapiSwitch AND "02_Peripheral".IN.YikamaTanki.KapiSwitch1;
   "01_System".Timers.Sequence.IBCTah_TimerAdim2.TON(IN := "IBCTahliye_IBCVana_Kapat" AND "02_Peripheral".IN.IBC.AkisValfi.Closed,
                           PT := t#3s);
   IF "01_System".Timers.Sequence.IBCTah_TimerAdim2.Q THEN "01_System".State.IBCTahliye := 3; END_IF;
END_REGION

REGION Network 4
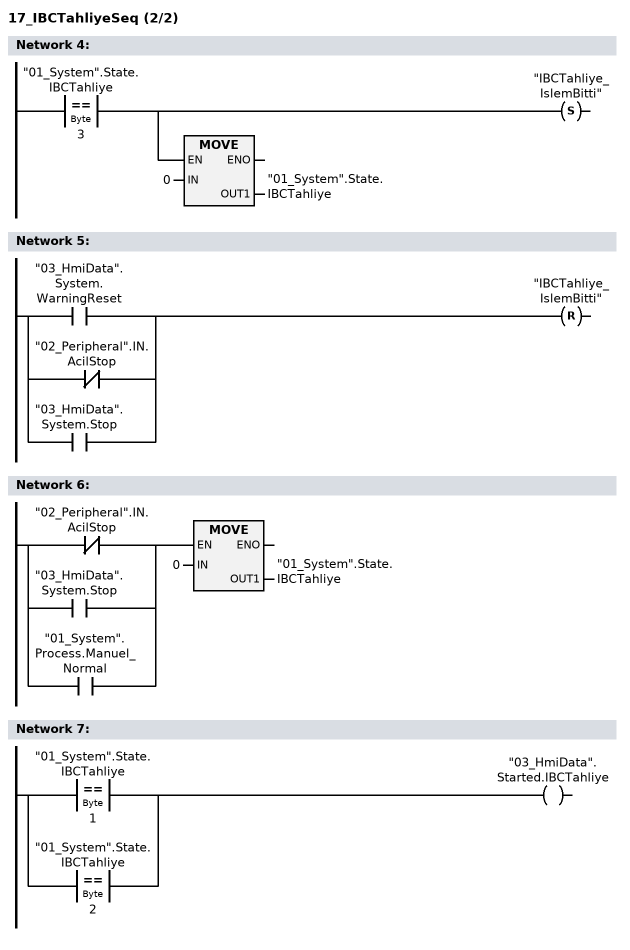
   RUNG wire#powerrail
      { S7_Templates := "SrcType := Byte" } EQ_Contact(in1 := "01_System".State.IBCTahliye, in2 := 3)
      wire#w1
      S_Coil( "IBCTahliye_IslemBitti" )
   END_RUNG
   RUNG wire#w1
      Move(in := 0, out1 => "01_System".State.IBCTahliye)
   END_RUNG
   // the same network as SCL:
   IF "01_System".State.IBCTahliye = 3 THEN
       "IBCTahliye_IslemBitti" := TRUE;
       "01_System".State.IBCTahliye := 0;
   END_IF;
END_REGION

REGION Network 5
   RUNG wire#powerrail
      Contact( "03_HmiData".System.WarningReset )
      wire#w1
      R_Coil( "IBCTahliye_IslemBitti" )
   END_RUNG
   RUNG wire#powerrail
      I_Contact( "02_Peripheral".IN.AcilStop )
   END_RUNG wire#w1
   RUNG wire#powerrail
      Contact( "03_HmiData".System.Stop )
   END_RUNG wire#w1
   // the same network as SCL:
   IF "03_HmiData".System.WarningReset OR NOT "02_Peripheral".IN.AcilStop OR "03_HmiData".System.Stop THEN
       "IBCTahliye_IslemBitti" := FALSE;
   END_IF;
END_REGION

REGION Network 6
   RUNG wire#powerrail
      I_Contact( "02_Peripheral".IN.AcilStop )
      wire#w1
      Move(in := 0, out1 => "01_System".State.IBCTahliye)
   END_RUNG
   RUNG wire#powerrail
      Contact( "03_HmiData".System.Stop )
   END_RUNG wire#w1
   RUNG wire#powerrail
      Contact( "01_System".Process.Manuel_Normal )
   END_RUNG wire#w1
   // the same network as SCL:
   IF NOT "02_Peripheral".IN.AcilStop OR "03_HmiData".System.Stop OR "01_System".Process.Manuel_Normal THEN
       "01_System".State.IBCTahliye := 0;
   END_IF;
END_REGION

REGION Network 7
   RUNG wire#powerrail
      { S7_Templates := "SrcType := Byte" } EQ_Contact(in1 := "01_System".State.IBCTahliye, in2 := 1)
      wire#w1
      Coil( "03_HmiData".Started.IBCTahliye )
   END_RUNG
   RUNG wire#powerrail
      { S7_Templates := "SrcType := Byte" } EQ_Contact(in1 := "01_System".State.IBCTahliye, in2 := 2)
   END_RUNG wire#w1
   // the same network as SCL:
   "03_HmiData".Started.IBCTahliye := ("01_System".State.IBCTahliye = 1) OR ("01_System".State.IBCTahliye = 2);
END_REGION
END_FUNCTION

FUNCTION "23_UyariLambalari" : Void   // FC9, LAD
{ S7_Optimized_Access := 'TRUE' }
VERSION : 0.1
BEGIN

REGION Network 1: Kırmızı lamba
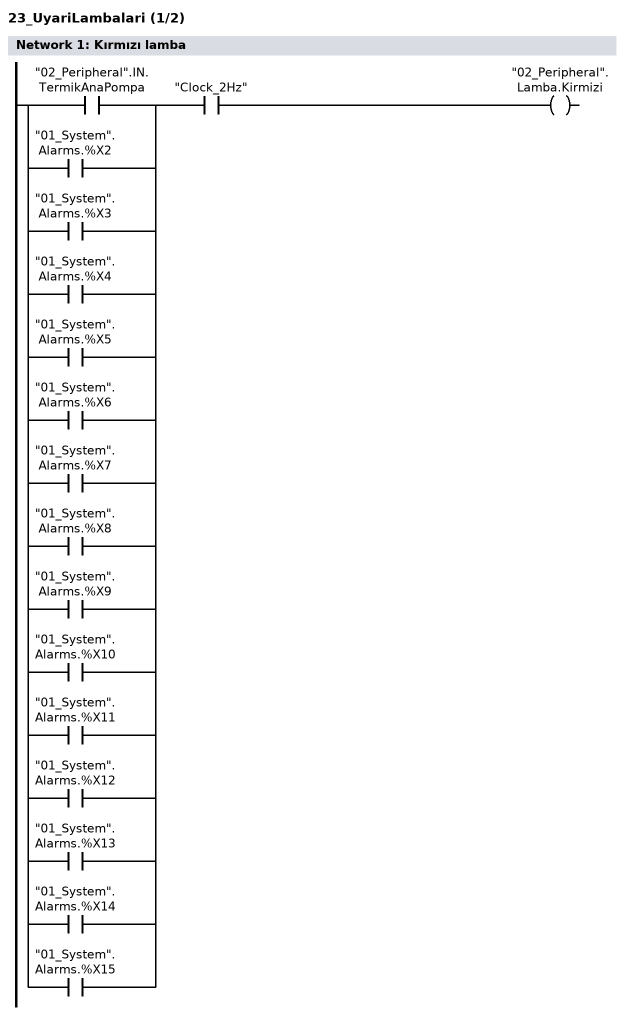
   RUNG wire#powerrail
      Contact( "02_Peripheral".IN.TermikAnaPompa )
      wire#w1
      Contact( "Clock_2Hz" )
      Coil( "02_Peripheral".Lamba.Kirmizi )
   END_RUNG
   RUNG wire#powerrail
      Contact( "01_System".Alarms.%X2 )
   END_RUNG wire#w1
   RUNG wire#powerrail
      Contact( "01_System".Alarms.%X3 )
   END_RUNG wire#w1
   RUNG wire#powerrail
      Contact( "01_System".Alarms.%X4 )
   END_RUNG wire#w1
   RUNG wire#powerrail
      Contact( "01_System".Alarms.%X5 )
   END_RUNG wire#w1
   RUNG wire#powerrail
      Contact( "01_System".Alarms.%X6 )
   END_RUNG wire#w1
   RUNG wire#powerrail
      Contact( "01_System".Alarms.%X7 )
   END_RUNG wire#w1
   RUNG wire#powerrail
      Contact( "01_System".Alarms.%X8 )
   END_RUNG wire#w1
   RUNG wire#powerrail
      Contact( "01_System".Alarms.%X9 )
   END_RUNG wire#w1
   RUNG wire#powerrail
      Contact( "01_System".Alarms.%X10 )
   END_RUNG wire#w1
   RUNG wire#powerrail
      Contact( "01_System".Alarms.%X11 )
   END_RUNG wire#w1
   RUNG wire#powerrail
      Contact( "01_System".Alarms.%X12 )
   END_RUNG wire#w1
   RUNG wire#powerrail
      Contact( "01_System".Alarms.%X13 )
   END_RUNG wire#w1
   RUNG wire#powerrail
      Contact( "01_System".Alarms.%X14 )
   END_RUNG wire#w1
   RUNG wire#powerrail
      Contact( "01_System".Alarms.%X15 )
   END_RUNG wire#w1
   // the same network as SCL:
   "02_Peripheral".Lamba.Kirmizi := ("02_Peripheral".IN.TermikAnaPompa OR "01_System".Alarms.%X2 OR "01_System".Alarms.%X3 OR "01_System".Alarms.%X4 OR "01_System".Alarms.%X5 OR "01_System".Alarms.%X6 OR "01_System".Alarms.%X7 OR "01_System".Alarms.%X8 OR "01_System".Alarms.%X9 OR "01_System".Alarms.%X10 OR "01_System".Alarms.%X11 OR "01_System".Alarms.%X12 OR "01_System".Alarms.%X13 OR "01_System".Alarms.%X14 OR "01_System".Alarms.%X15) AND "Clock_2Hz";
END_REGION

